// TIA Portal V17 export
// export: Created 2025-03-05T07:59:25.1832368Z, ExportSetting WithDefaults, DisplayName Totally Integrated Automation Portal, DisplayVersion V17 Update 8, DisplayName TIA Portal Openness, DisplayVersion V17 Update 8, DisplayName TIA Portal Version Control Interface, DisplayVersion V17, DisplayName SINAMICS Startdrive Advanced, DisplayVersion V17 SP2, DisplayName SINAMICS Startdrive G110M, G120, G120C, G120D, G120P, G115D, DisplayVersion V17 SP2, DisplayName SINAMICS Startdrive G130, G150, S120, S150, SINAMICS MV, S210, DisplayVersion V17 SP2, DisplayName STEP 7 Professional, DisplayVersion V17 Update 8, DisplayName SINUMERIK ONE STEP 7 Toolbox, DisplayVersion V17 Update 12, DisplayName SINUMERIK 840D sl STEP 7 Toolbox, DisplayVersion V17 Update 12, DisplayName STEP 7 Safety, DisplayVersion V17 Update 6, DisplayName WinCC Advanced, DisplayVersion V17 Update 8
FUNCTION "FC8101_MANUAL_LOADING_PART_STATUS_MANAGEMENT" : Void   // FC8101, LAD
{ S7_Optimized_Access := 'FALSE' }
VERSION : 0.1
// stored: AutoNumber false, IsIECCheckEnabled false, SetENOAutomatically false, UDAEnableTagReadback false
   VAR_TEMP
      AUX_STRING : String;
      CNT_CHARS : Int;
      CHARS_ARRAY : Array[0..63] of Char;
      ZERO : Byte;   // ZERO
      STATUS_BLKMOV : Int;   // STATUS BLKMOV
      STATUS_FILL : Int;   // STATUS FILL
   END_VAR
   VAR_TEMP   // added for the SCL form of the ladder/FBD networks
      _w1 : Bool;
      _w2 : Bool;
      _w3 : Bool;
      _w4 : Bool;
      _w5 : Bool;
      _w6 : Bool;
      _w7 : Bool;
      _w8 : Bool;
      _w9 : Bool;
      _w10 : Bool;
      _w11 : Bool;
   END_VAR
BEGIN

REGION Network 1: ZERO
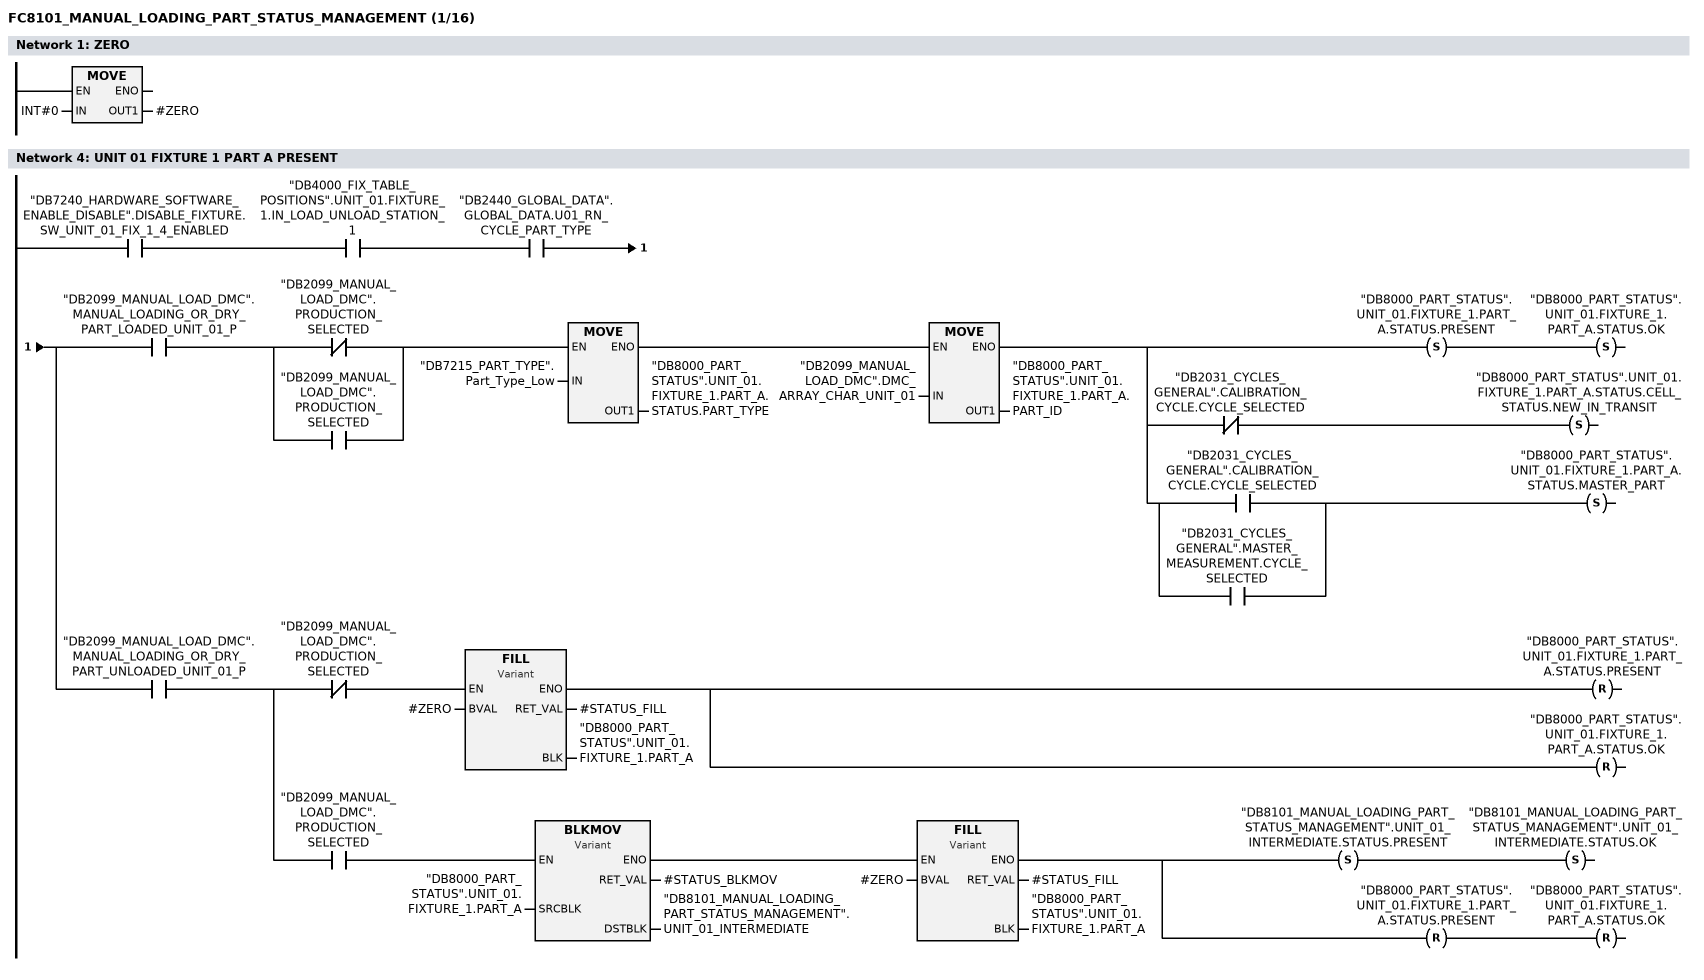
   RUNG wire#powerrail
      { S7_GenerateENO := "TRUE" } Move(in := INT#0, out1 => #ZERO)
   END_RUNG
   // the same network as SCL:
   #ZERO := INT#0;
END_REGION

REGION Network 2: <<<<<<<<<<<<<<<<<<<< RN CYCLE >>>>>>>>>>>>>>>>>>>>
END_REGION

REGION Network 3: <<<<<<<<<<<<<<<<<<<< UNIT 01 >>>>>>>>>>>>>>>>>>>>
END_REGION

REGION Network 4: UNIT 01 FIXTURE 1 PART A PRESENT
   RUNG wire#powerrail
      Contact( "DB7240_HARDWARE_SOFTWARE_ENABLE_DISABLE".DISABLE_FIXTURE.SW_UNIT_01_FIX_1_4_ENABLED )
      Contact( "DB4000_FIX_TABLE_POSITIONS".UNIT_01.FIXTURE_1.IN_LOAD_UNLOAD_STATION_1 )
      Contact( "DB2440_GLOBAL_DATA".GLOBAL_DATA.U01_RN_CYCLE_PART_TYPE )
      wire#w1
      Contact( "DB2099_MANUAL_LOAD_DMC".MANUAL_LOADING_OR_DRY_PART_LOADED_UNIT_01_P )
      wire#w2
      I_Contact( "DB2099_MANUAL_LOAD_DMC".PRODUCTION_SELECTED )
      wire#w3
      { S7_GenerateENO := "TRUE" } Move(in := "DB7215_PART_TYPE".Part_Type_Low, out1 => "DB8000_PART_STATUS".UNIT_01.FIXTURE_1.PART_A.STATUS.PART_TYPE)
      Move(in := "DB2099_MANUAL_LOAD_DMC".DMC_ARRAY_CHAR_UNIT_01, out1 => "DB8000_PART_STATUS".UNIT_01.FIXTURE_1.PART_A.PART_ID)
      wire#w4
      S_Coil( "DB8000_PART_STATUS".UNIT_01.FIXTURE_1.PART_A.STATUS.PRESENT )
      S_Coil( "DB8000_PART_STATUS".UNIT_01.FIXTURE_1.PART_A.STATUS.OK )
   END_RUNG
   RUNG wire#w2
      Contact( "DB2099_MANUAL_LOAD_DMC".PRODUCTION_SELECTED )
   END_RUNG wire#w3
   RUNG wire#w4
      I_Contact( "DB2031_CYCLES_GENERAL".CALIBRATION_CYCLE.CYCLE_SELECTED )
      S_Coil( "DB8000_PART_STATUS".UNIT_01.FIXTURE_1.PART_A.STATUS.CELL_STATUS.NEW_IN_TRANSIT )
   END_RUNG
   RUNG wire#w4
      Contact( "DB2031_CYCLES_GENERAL".CALIBRATION_CYCLE.CYCLE_SELECTED )
      wire#w5
      S_Coil( "DB8000_PART_STATUS".UNIT_01.FIXTURE_1.PART_A.STATUS.MASTER_PART )
   END_RUNG
   RUNG wire#w4
      Contact( "DB2031_CYCLES_GENERAL".MASTER_MEASUREMENT.CYCLE_SELECTED )
   END_RUNG wire#w5
   RUNG wire#w1
      Contact( "DB2099_MANUAL_LOAD_DMC".MANUAL_LOADING_OR_DRY_PART_UNLOADED_UNIT_01_P )
      wire#w6
      I_Contact( "DB2099_MANUAL_LOAD_DMC".PRODUCTION_SELECTED )
      { S7_Templates := "ptr_type := Variant" } FILL(BVAL := #ZERO, RET_VAL => #STATUS_FILL, BLK => "DB8000_PART_STATUS".UNIT_01.FIXTURE_1.PART_A)
      wire#w7
      R_Coil( "DB8000_PART_STATUS".UNIT_01.FIXTURE_1.PART_A.STATUS.PRESENT )
   END_RUNG
   RUNG wire#w7
      R_Coil( "DB8000_PART_STATUS".UNIT_01.FIXTURE_1.PART_A.STATUS.OK )
   END_RUNG
   RUNG wire#w6
      Contact( "DB2099_MANUAL_LOAD_DMC".PRODUCTION_SELECTED )
      { S7_Templates := "blk_type := Variant" } BLKMOV(SRCBLK := "DB8000_PART_STATUS".UNIT_01.FIXTURE_1.PART_A, RET_VAL => #STATUS_BLKMOV, DSTBLK => "DB8101_MANUAL_LOADING_PART_STATUS_MANAGEMENT".UNIT_01_INTERMEDIATE)
      { S7_Templates := "ptr_type := Variant" } FILL(BVAL := #ZERO, RET_VAL => #STATUS_FILL, BLK => "DB8000_PART_STATUS".UNIT_01.FIXTURE_1.PART_A)
      wire#w8
      S_Coil( "DB8101_MANUAL_LOADING_PART_STATUS_MANAGEMENT".UNIT_01_INTERMEDIATE.STATUS.PRESENT )
      S_Coil( "DB8101_MANUAL_LOADING_PART_STATUS_MANAGEMENT".UNIT_01_INTERMEDIATE.STATUS.OK )
   END_RUNG
   RUNG wire#w8
      R_Coil( "DB8000_PART_STATUS".UNIT_01.FIXTURE_1.PART_A.STATUS.PRESENT )
      R_Coil( "DB8000_PART_STATUS".UNIT_01.FIXTURE_1.PART_A.STATUS.OK )
   END_RUNG
   // the same network as SCL:
   // ENO of a box is taken as its EN; it also drops when the box reports an error
   #_w1 := "DB7240_HARDWARE_SOFTWARE_ENABLE_DISABLE".DISABLE_FIXTURE.SW_UNIT_01_FIX_1_4_ENABLED AND "DB4000_FIX_TABLE_POSITIONS".UNIT_01.FIXTURE_1.IN_LOAD_UNLOAD_STATION_1 AND "DB2440_GLOBAL_DATA".GLOBAL_DATA.U01_RN_CYCLE_PART_TYPE;
   #_w2 := #_w1 AND "DB2099_MANUAL_LOAD_DMC".MANUAL_LOADING_OR_DRY_PART_LOADED_UNIT_01_P AND (NOT "DB2099_MANUAL_LOAD_DMC".PRODUCTION_SELECTED OR "DB2099_MANUAL_LOAD_DMC".PRODUCTION_SELECTED);
   IF #_w2 THEN
       "DB8000_PART_STATUS".UNIT_01.FIXTURE_1.PART_A.STATUS.PART_TYPE := "DB7215_PART_TYPE".Part_Type_Low;
       "DB8000_PART_STATUS".UNIT_01.FIXTURE_1.PART_A.PART_ID := "DB2099_MANUAL_LOAD_DMC".DMC_ARRAY_CHAR_UNIT_01;
       "DB8000_PART_STATUS".UNIT_01.FIXTURE_1.PART_A.STATUS.PRESENT := TRUE;
       "DB8000_PART_STATUS".UNIT_01.FIXTURE_1.PART_A.STATUS.OK := TRUE;
   END_IF;
   IF #_w2 AND NOT "DB2031_CYCLES_GENERAL".CALIBRATION_CYCLE.CYCLE_SELECTED THEN
       "DB8000_PART_STATUS".UNIT_01.FIXTURE_1.PART_A.STATUS.CELL_STATUS.NEW_IN_TRANSIT := TRUE;
   END_IF;
   IF #_w2 AND ("DB2031_CYCLES_GENERAL".CALIBRATION_CYCLE.CYCLE_SELECTED OR "DB2031_CYCLES_GENERAL".MASTER_MEASUREMENT.CYCLE_SELECTED) THEN
       "DB8000_PART_STATUS".UNIT_01.FIXTURE_1.PART_A.STATUS.MASTER_PART := TRUE;
   END_IF;
   #_w3 := #_w1 AND "DB2099_MANUAL_LOAD_DMC".MANUAL_LOADING_OR_DRY_PART_UNLOADED_UNIT_01_P;
   #STATUS_FILL := FILL(EN := #_w3 AND NOT "DB2099_MANUAL_LOAD_DMC".PRODUCTION_SELECTED,
                        BVAL := #ZERO,
                        BLK => "DB8000_PART_STATUS".UNIT_01.FIXTURE_1.PART_A,
                        ENO => #_w4);
   IF #_w4 THEN
       "DB8000_PART_STATUS".UNIT_01.FIXTURE_1.PART_A.STATUS.PRESENT := FALSE;
       "DB8000_PART_STATUS".UNIT_01.FIXTURE_1.PART_A.STATUS.OK := FALSE;
   END_IF;
   #STATUS_BLKMOV := BLKMOV(EN := #_w3 AND "DB2099_MANUAL_LOAD_DMC".PRODUCTION_SELECTED,
                           SRCBLK := "DB8000_PART_STATUS".UNIT_01.FIXTURE_1.PART_A,
                           DSTBLK => "DB8101_MANUAL_LOADING_PART_STATUS_MANAGEMENT".UNIT_01_INTERMEDIATE,
                           ENO => #_w5);
   #STATUS_FILL := FILL(EN := #_w5,
                        BVAL := #ZERO,
                        BLK => "DB8000_PART_STATUS".UNIT_01.FIXTURE_1.PART_A,
                        ENO => #_w6);
   IF #_w6 THEN
       "DB8101_MANUAL_LOADING_PART_STATUS_MANAGEMENT".UNIT_01_INTERMEDIATE.STATUS.PRESENT := TRUE;
       "DB8101_MANUAL_LOADING_PART_STATUS_MANAGEMENT".UNIT_01_INTERMEDIATE.STATUS.OK := TRUE;
       "DB8000_PART_STATUS".UNIT_01.FIXTURE_1.PART_A.STATUS.PRESENT := FALSE;
       "DB8000_PART_STATUS".UNIT_01.FIXTURE_1.PART_A.STATUS.OK := FALSE;
   END_IF;
END_REGION

REGION Network 5: UNIT 01 FIXTURE 2 PART A PRESENT
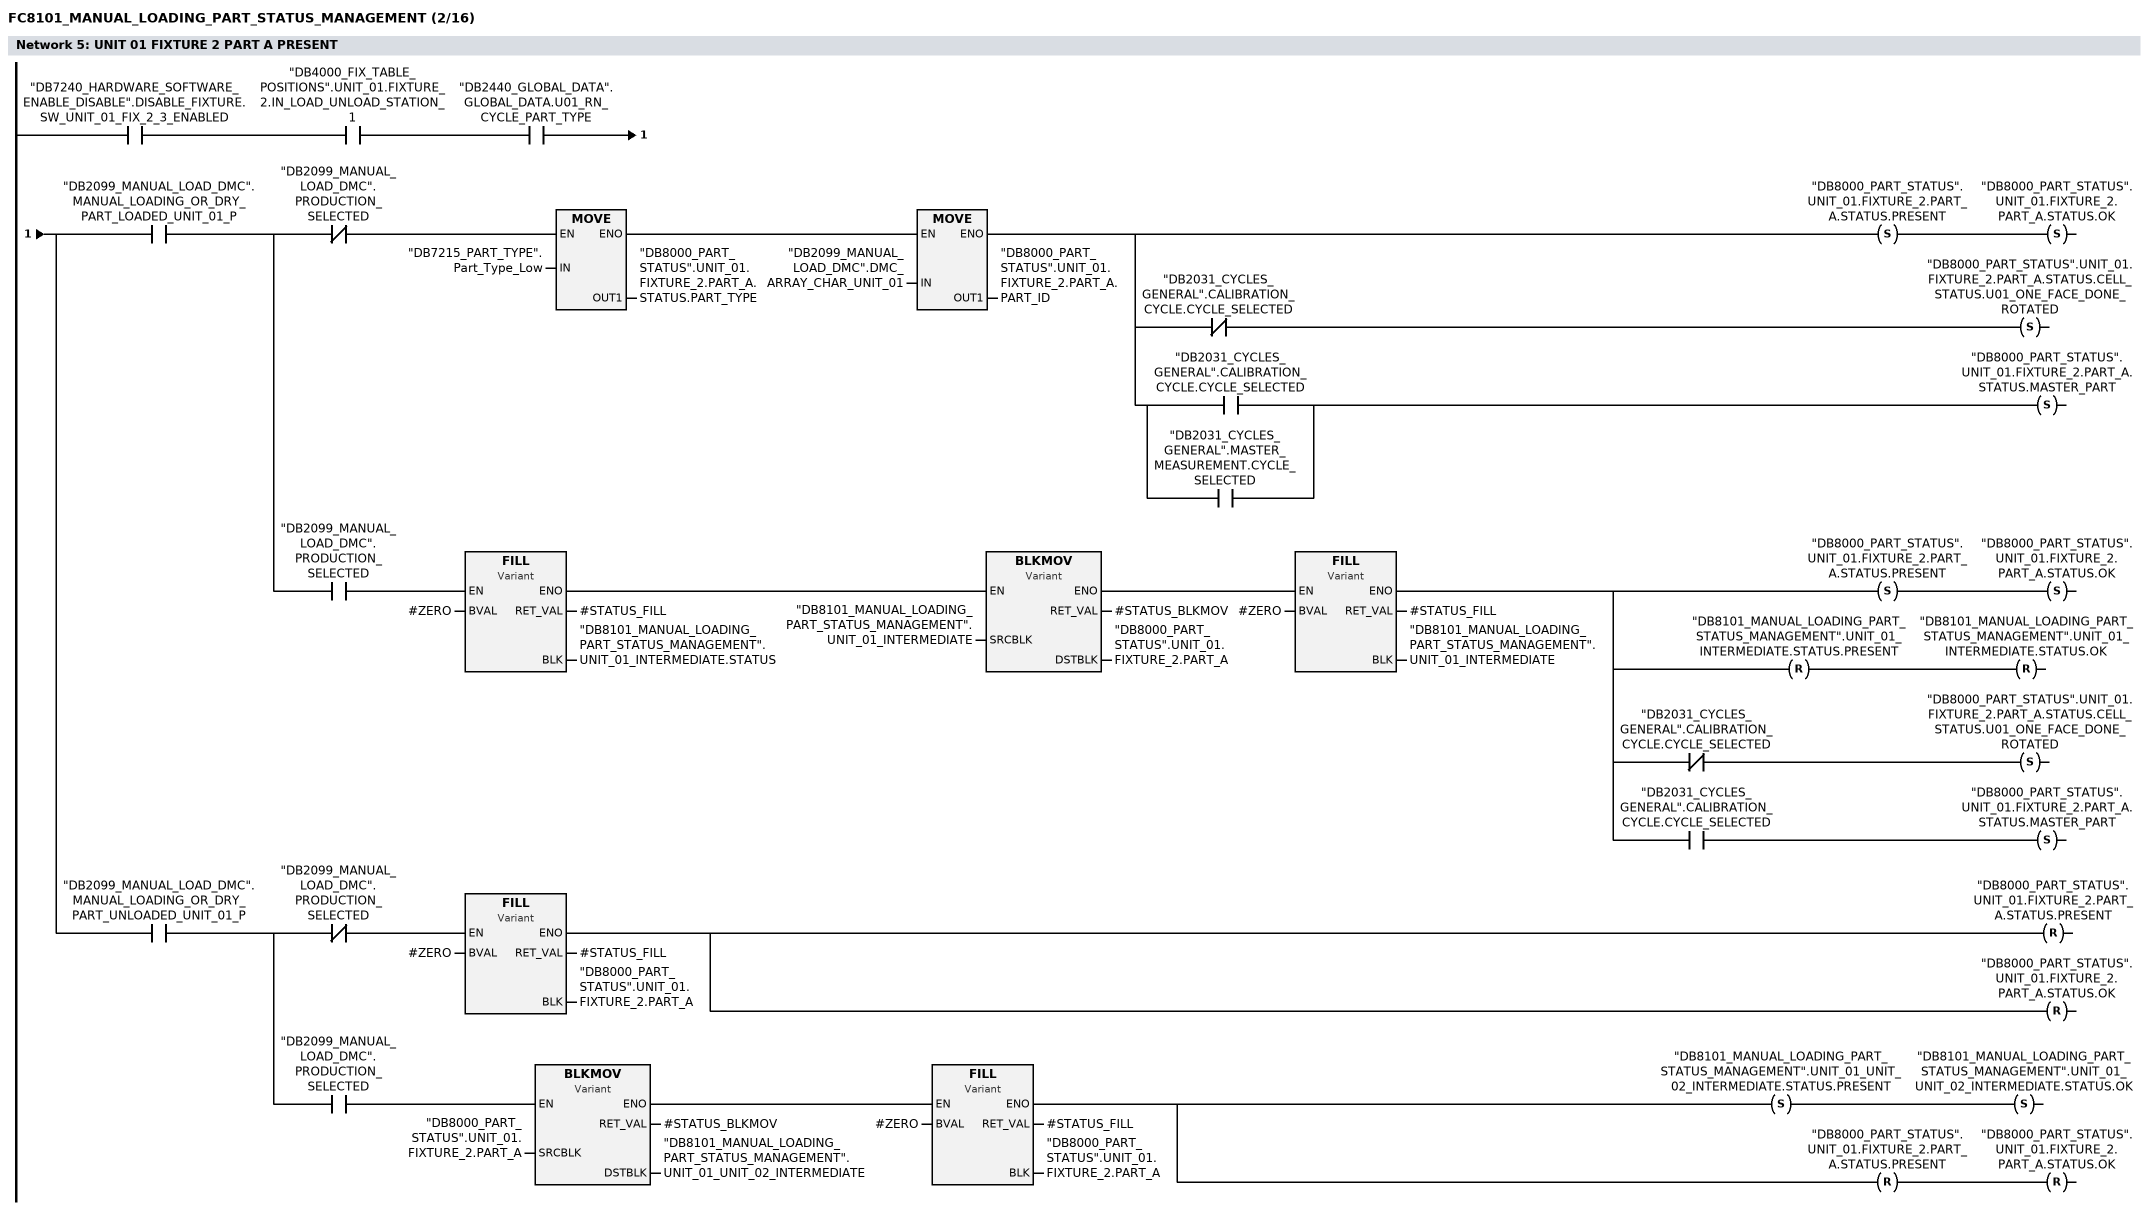
   RUNG wire#powerrail
      Contact( "DB7240_HARDWARE_SOFTWARE_ENABLE_DISABLE".DISABLE_FIXTURE.SW_UNIT_01_FIX_2_3_ENABLED )
      Contact( "DB4000_FIX_TABLE_POSITIONS".UNIT_01.FIXTURE_2.IN_LOAD_UNLOAD_STATION_1 )
      Contact( "DB2440_GLOBAL_DATA".GLOBAL_DATA.U01_RN_CYCLE_PART_TYPE )
      wire#w1
      Contact( "DB2099_MANUAL_LOAD_DMC".MANUAL_LOADING_OR_DRY_PART_LOADED_UNIT_01_P )
      wire#w2
      I_Contact( "DB2099_MANUAL_LOAD_DMC".PRODUCTION_SELECTED )
      { S7_GenerateENO := "TRUE" } Move(in := "DB7215_PART_TYPE".Part_Type_Low, out1 => "DB8000_PART_STATUS".UNIT_01.FIXTURE_2.PART_A.STATUS.PART_TYPE)
      Move(in := "DB2099_MANUAL_LOAD_DMC".DMC_ARRAY_CHAR_UNIT_01, out1 => "DB8000_PART_STATUS".UNIT_01.FIXTURE_2.PART_A.PART_ID)
      wire#w3
      S_Coil( "DB8000_PART_STATUS".UNIT_01.FIXTURE_2.PART_A.STATUS.PRESENT )
      S_Coil( "DB8000_PART_STATUS".UNIT_01.FIXTURE_2.PART_A.STATUS.OK )
   END_RUNG
   RUNG wire#w3
      I_Contact( "DB2031_CYCLES_GENERAL".CALIBRATION_CYCLE.CYCLE_SELECTED )
      S_Coil( "DB8000_PART_STATUS".UNIT_01.FIXTURE_2.PART_A.STATUS.CELL_STATUS.U01_ONE_FACE_DONE_ROTATED )
   END_RUNG
   RUNG wire#w3
      Contact( "DB2031_CYCLES_GENERAL".CALIBRATION_CYCLE.CYCLE_SELECTED )
      wire#w4
      S_Coil( "DB8000_PART_STATUS".UNIT_01.FIXTURE_2.PART_A.STATUS.MASTER_PART )
   END_RUNG
   RUNG wire#w3
      Contact( "DB2031_CYCLES_GENERAL".MASTER_MEASUREMENT.CYCLE_SELECTED )
   END_RUNG wire#w4
   RUNG wire#w2
      Contact( "DB2099_MANUAL_LOAD_DMC".PRODUCTION_SELECTED )
      { S7_Templates := "ptr_type := Variant" } FILL(BVAL := #ZERO, RET_VAL => #STATUS_FILL, BLK => "DB8101_MANUAL_LOADING_PART_STATUS_MANAGEMENT".UNIT_01_INTERMEDIATE.STATUS)
      { S7_Templates := "blk_type := Variant" } BLKMOV(SRCBLK := "DB8101_MANUAL_LOADING_PART_STATUS_MANAGEMENT".UNIT_01_INTERMEDIATE, RET_VAL => #STATUS_BLKMOV, DSTBLK => "DB8000_PART_STATUS".UNIT_01.FIXTURE_2.PART_A)
      { S7_Templates := "ptr_type := Variant" } FILL(BVAL := #ZERO, RET_VAL => #STATUS_FILL, BLK => "DB8101_MANUAL_LOADING_PART_STATUS_MANAGEMENT".UNIT_01_INTERMEDIATE)
      wire#w5
      S_Coil( "DB8000_PART_STATUS".UNIT_01.FIXTURE_2.PART_A.STATUS.PRESENT )
      S_Coil( "DB8000_PART_STATUS".UNIT_01.FIXTURE_2.PART_A.STATUS.OK )
   END_RUNG
   RUNG wire#w5
      R_Coil( "DB8101_MANUAL_LOADING_PART_STATUS_MANAGEMENT".UNIT_01_INTERMEDIATE.STATUS.PRESENT )
      R_Coil( "DB8101_MANUAL_LOADING_PART_STATUS_MANAGEMENT".UNIT_01_INTERMEDIATE.STATUS.OK )
   END_RUNG
   RUNG wire#w5
      I_Contact( "DB2031_CYCLES_GENERAL".CALIBRATION_CYCLE.CYCLE_SELECTED )
      S_Coil( "DB8000_PART_STATUS".UNIT_01.FIXTURE_2.PART_A.STATUS.CELL_STATUS.U01_ONE_FACE_DONE_ROTATED )
   END_RUNG
   RUNG wire#w5
      Contact( "DB2031_CYCLES_GENERAL".CALIBRATION_CYCLE.CYCLE_SELECTED )
      S_Coil( "DB8000_PART_STATUS".UNIT_01.FIXTURE_2.PART_A.STATUS.MASTER_PART )
   END_RUNG
   RUNG wire#w1
      Contact( "DB2099_MANUAL_LOAD_DMC".MANUAL_LOADING_OR_DRY_PART_UNLOADED_UNIT_01_P )
      wire#w6
      I_Contact( "DB2099_MANUAL_LOAD_DMC".PRODUCTION_SELECTED )
      { S7_Templates := "ptr_type := Variant" } FILL(BVAL := #ZERO, RET_VAL => #STATUS_FILL, BLK => "DB8000_PART_STATUS".UNIT_01.FIXTURE_2.PART_A)
      wire#w7
      R_Coil( "DB8000_PART_STATUS".UNIT_01.FIXTURE_2.PART_A.STATUS.PRESENT )
   END_RUNG
   RUNG wire#w7
      R_Coil( "DB8000_PART_STATUS".UNIT_01.FIXTURE_2.PART_A.STATUS.OK )
   END_RUNG
   RUNG wire#w6
      Contact( "DB2099_MANUAL_LOAD_DMC".PRODUCTION_SELECTED )
      { S7_Templates := "blk_type := Variant" } BLKMOV(SRCBLK := "DB8000_PART_STATUS".UNIT_01.FIXTURE_2.PART_A, RET_VAL => #STATUS_BLKMOV, DSTBLK => "DB8101_MANUAL_LOADING_PART_STATUS_MANAGEMENT".UNIT_01_UNIT_02_INTERMEDIATE)
      { S7_Templates := "ptr_type := Variant" } FILL(BVAL := #ZERO, RET_VAL => #STATUS_FILL, BLK => "DB8000_PART_STATUS".UNIT_01.FIXTURE_2.PART_A)
      wire#w8
      S_Coil( "DB8101_MANUAL_LOADING_PART_STATUS_MANAGEMENT".UNIT_01_UNIT_02_INTERMEDIATE.STATUS.PRESENT )
      S_Coil( "DB8101_MANUAL_LOADING_PART_STATUS_MANAGEMENT".UNIT_01_UNIT_02_INTERMEDIATE.STATUS.OK )
   END_RUNG
   RUNG wire#w8
      R_Coil( "DB8000_PART_STATUS".UNIT_01.FIXTURE_2.PART_A.STATUS.PRESENT )
      R_Coil( "DB8000_PART_STATUS".UNIT_01.FIXTURE_2.PART_A.STATUS.OK )
   END_RUNG
   // the same network as SCL:
   // ENO of a box is taken as its EN; it also drops when the box reports an error
   #_w1 := "DB7240_HARDWARE_SOFTWARE_ENABLE_DISABLE".DISABLE_FIXTURE.SW_UNIT_01_FIX_2_3_ENABLED AND "DB4000_FIX_TABLE_POSITIONS".UNIT_01.FIXTURE_2.IN_LOAD_UNLOAD_STATION_1 AND "DB2440_GLOBAL_DATA".GLOBAL_DATA.U01_RN_CYCLE_PART_TYPE;
   #_w2 := #_w1 AND "DB2099_MANUAL_LOAD_DMC".MANUAL_LOADING_OR_DRY_PART_LOADED_UNIT_01_P;
   #_w3 := #_w2 AND NOT "DB2099_MANUAL_LOAD_DMC".PRODUCTION_SELECTED;
   IF #_w3 THEN
       "DB8000_PART_STATUS".UNIT_01.FIXTURE_2.PART_A.STATUS.PART_TYPE := "DB7215_PART_TYPE".Part_Type_Low;
       "DB8000_PART_STATUS".UNIT_01.FIXTURE_2.PART_A.PART_ID := "DB2099_MANUAL_LOAD_DMC".DMC_ARRAY_CHAR_UNIT_01;
       "DB8000_PART_STATUS".UNIT_01.FIXTURE_2.PART_A.STATUS.PRESENT := TRUE;
       "DB8000_PART_STATUS".UNIT_01.FIXTURE_2.PART_A.STATUS.OK := TRUE;
   END_IF;
   IF #_w3 AND NOT "DB2031_CYCLES_GENERAL".CALIBRATION_CYCLE.CYCLE_SELECTED THEN
       "DB8000_PART_STATUS".UNIT_01.FIXTURE_2.PART_A.STATUS.CELL_STATUS.U01_ONE_FACE_DONE_ROTATED := TRUE;
   END_IF;
   IF #_w3 AND ("DB2031_CYCLES_GENERAL".CALIBRATION_CYCLE.CYCLE_SELECTED OR "DB2031_CYCLES_GENERAL".MASTER_MEASUREMENT.CYCLE_SELECTED) THEN
       "DB8000_PART_STATUS".UNIT_01.FIXTURE_2.PART_A.STATUS.MASTER_PART := TRUE;
   END_IF;
   #_w4 := #_w2 AND "DB2099_MANUAL_LOAD_DMC".PRODUCTION_SELECTED;
   #STATUS_FILL := FILL(EN := #_w4,
                        BVAL := #ZERO,
                        BLK => "DB8101_MANUAL_LOADING_PART_STATUS_MANAGEMENT".UNIT_01_INTERMEDIATE.STATUS,
                        ENO => #_w5);
   #STATUS_BLKMOV := BLKMOV(EN := #_w5,
                           SRCBLK := "DB8101_MANUAL_LOADING_PART_STATUS_MANAGEMENT".UNIT_01_INTERMEDIATE,
                           DSTBLK => "DB8000_PART_STATUS".UNIT_01.FIXTURE_2.PART_A,
                           ENO => #_w6);
   #STATUS_FILL := FILL(EN := #_w6,
                        BVAL := #ZERO,
                        BLK => "DB8101_MANUAL_LOADING_PART_STATUS_MANAGEMENT".UNIT_01_INTERMEDIATE,
                        ENO => #_w7);
   IF #_w7 THEN
       "DB8000_PART_STATUS".UNIT_01.FIXTURE_2.PART_A.STATUS.PRESENT := TRUE;
       "DB8000_PART_STATUS".UNIT_01.FIXTURE_2.PART_A.STATUS.OK := TRUE;
       "DB8101_MANUAL_LOADING_PART_STATUS_MANAGEMENT".UNIT_01_INTERMEDIATE.STATUS.PRESENT := FALSE;
       "DB8101_MANUAL_LOADING_PART_STATUS_MANAGEMENT".UNIT_01_INTERMEDIATE.STATUS.OK := FALSE;
   END_IF;
   IF #_w7 AND NOT "DB2031_CYCLES_GENERAL".CALIBRATION_CYCLE.CYCLE_SELECTED THEN
       "DB8000_PART_STATUS".UNIT_01.FIXTURE_2.PART_A.STATUS.CELL_STATUS.U01_ONE_FACE_DONE_ROTATED := TRUE;
   END_IF;
   IF #_w7 AND "DB2031_CYCLES_GENERAL".CALIBRATION_CYCLE.CYCLE_SELECTED THEN
       "DB8000_PART_STATUS".UNIT_01.FIXTURE_2.PART_A.STATUS.MASTER_PART := TRUE;
   END_IF;
   #_w8 := #_w1 AND "DB2099_MANUAL_LOAD_DMC".MANUAL_LOADING_OR_DRY_PART_UNLOADED_UNIT_01_P;
   #STATUS_FILL := FILL(EN := #_w8 AND NOT "DB2099_MANUAL_LOAD_DMC".PRODUCTION_SELECTED,
                        BVAL := #ZERO,
                        BLK => "DB8000_PART_STATUS".UNIT_01.FIXTURE_2.PART_A,
                        ENO => #_w9);
   IF #_w9 THEN
       "DB8000_PART_STATUS".UNIT_01.FIXTURE_2.PART_A.STATUS.PRESENT := FALSE;
       "DB8000_PART_STATUS".UNIT_01.FIXTURE_2.PART_A.STATUS.OK := FALSE;
   END_IF;
   #STATUS_BLKMOV := BLKMOV(EN := #_w8 AND "DB2099_MANUAL_LOAD_DMC".PRODUCTION_SELECTED,
                           SRCBLK := "DB8000_PART_STATUS".UNIT_01.FIXTURE_2.PART_A,
                           DSTBLK => "DB8101_MANUAL_LOADING_PART_STATUS_MANAGEMENT".UNIT_01_UNIT_02_INTERMEDIATE,
                           ENO => #_w10);
   #STATUS_FILL := FILL(EN := #_w10,
                        BVAL := #ZERO,
                        BLK => "DB8000_PART_STATUS".UNIT_01.FIXTURE_2.PART_A,
                        ENO => #_w11);
   IF #_w11 THEN
       "DB8101_MANUAL_LOADING_PART_STATUS_MANAGEMENT".UNIT_01_UNIT_02_INTERMEDIATE.STATUS.PRESENT := TRUE;
       "DB8101_MANUAL_LOADING_PART_STATUS_MANAGEMENT".UNIT_01_UNIT_02_INTERMEDIATE.STATUS.OK := TRUE;
       "DB8000_PART_STATUS".UNIT_01.FIXTURE_2.PART_A.STATUS.PRESENT := FALSE;
       "DB8000_PART_STATUS".UNIT_01.FIXTURE_2.PART_A.STATUS.OK := FALSE;
   END_IF;
END_REGION

REGION Network 6: UNIT 01 FIXTURE 3 PART A PRESENT
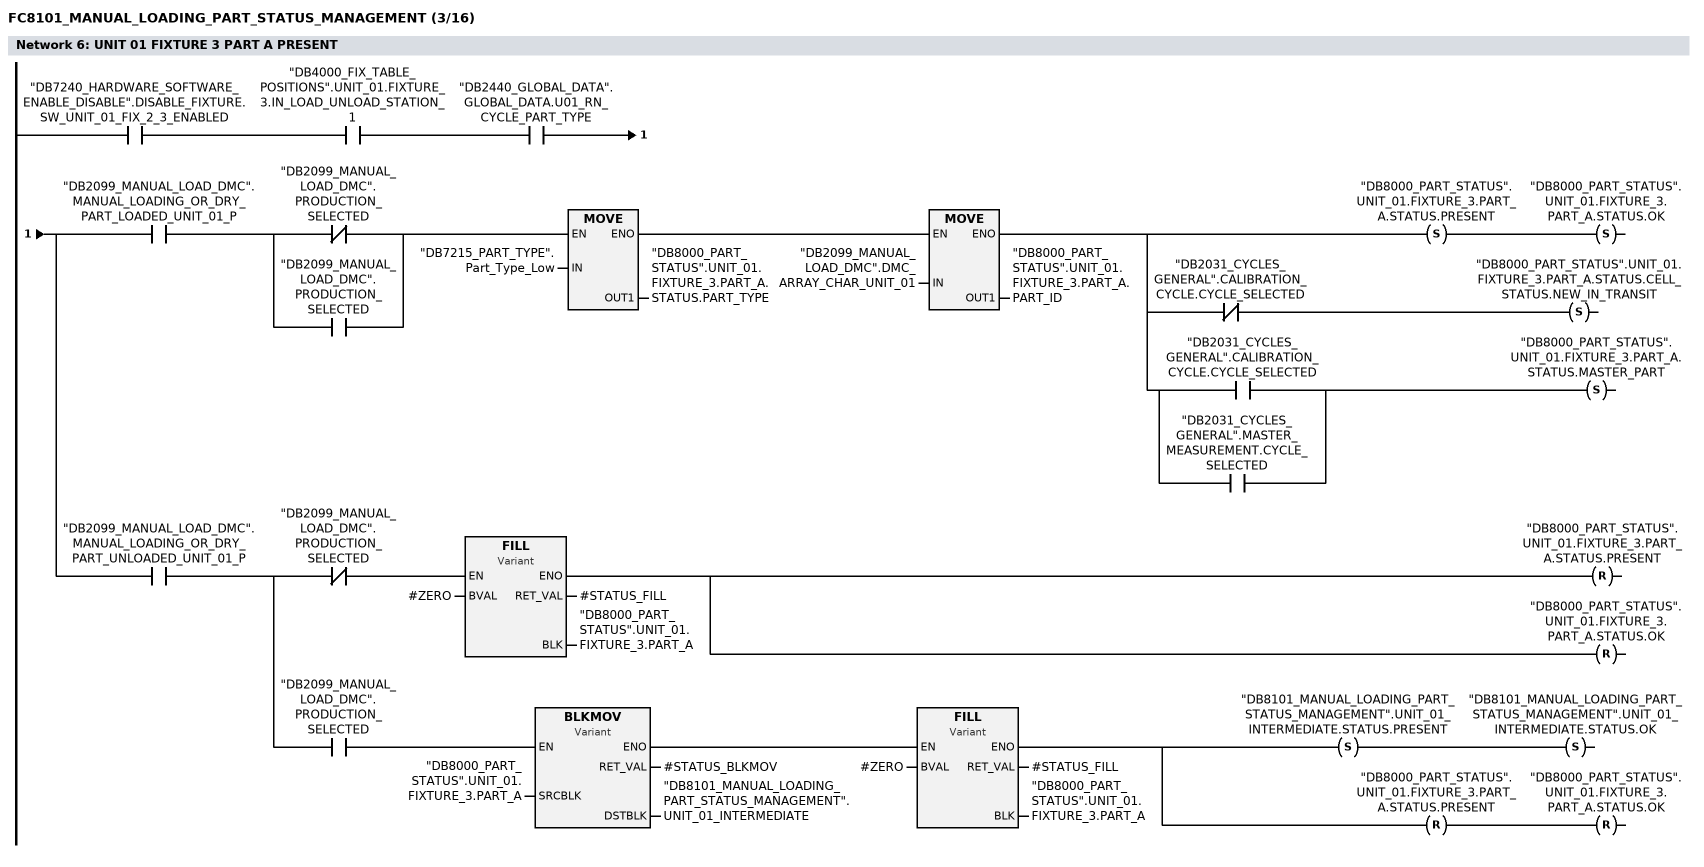
   RUNG wire#powerrail
      Contact( "DB7240_HARDWARE_SOFTWARE_ENABLE_DISABLE".DISABLE_FIXTURE.SW_UNIT_01_FIX_2_3_ENABLED )
      Contact( "DB4000_FIX_TABLE_POSITIONS".UNIT_01.FIXTURE_3.IN_LOAD_UNLOAD_STATION_1 )
      Contact( "DB2440_GLOBAL_DATA".GLOBAL_DATA.U01_RN_CYCLE_PART_TYPE )
      wire#w1
      Contact( "DB2099_MANUAL_LOAD_DMC".MANUAL_LOADING_OR_DRY_PART_LOADED_UNIT_01_P )
      wire#w2
      I_Contact( "DB2099_MANUAL_LOAD_DMC".PRODUCTION_SELECTED )
      wire#w3
      { S7_GenerateENO := "TRUE" } Move(in := "DB7215_PART_TYPE".Part_Type_Low, out1 => "DB8000_PART_STATUS".UNIT_01.FIXTURE_3.PART_A.STATUS.PART_TYPE)
      Move(in := "DB2099_MANUAL_LOAD_DMC".DMC_ARRAY_CHAR_UNIT_01, out1 => "DB8000_PART_STATUS".UNIT_01.FIXTURE_3.PART_A.PART_ID)
      wire#w4
      S_Coil( "DB8000_PART_STATUS".UNIT_01.FIXTURE_3.PART_A.STATUS.PRESENT )
      S_Coil( "DB8000_PART_STATUS".UNIT_01.FIXTURE_3.PART_A.STATUS.OK )
   END_RUNG
   RUNG wire#w2
      Contact( "DB2099_MANUAL_LOAD_DMC".PRODUCTION_SELECTED )
   END_RUNG wire#w3
   RUNG wire#w4
      I_Contact( "DB2031_CYCLES_GENERAL".CALIBRATION_CYCLE.CYCLE_SELECTED )
      S_Coil( "DB8000_PART_STATUS".UNIT_01.FIXTURE_3.PART_A.STATUS.CELL_STATUS.NEW_IN_TRANSIT )
   END_RUNG
   RUNG wire#w4
      Contact( "DB2031_CYCLES_GENERAL".CALIBRATION_CYCLE.CYCLE_SELECTED )
      wire#w5
      S_Coil( "DB8000_PART_STATUS".UNIT_01.FIXTURE_3.PART_A.STATUS.MASTER_PART )
   END_RUNG
   RUNG wire#w4
      Contact( "DB2031_CYCLES_GENERAL".MASTER_MEASUREMENT.CYCLE_SELECTED )
   END_RUNG wire#w5
   RUNG wire#w1
      Contact( "DB2099_MANUAL_LOAD_DMC".MANUAL_LOADING_OR_DRY_PART_UNLOADED_UNIT_01_P )
      wire#w6
      I_Contact( "DB2099_MANUAL_LOAD_DMC".PRODUCTION_SELECTED )
      { S7_Templates := "ptr_type := Variant" } FILL(BVAL := #ZERO, RET_VAL => #STATUS_FILL, BLK => "DB8000_PART_STATUS".UNIT_01.FIXTURE_3.PART_A)
      wire#w7
      R_Coil( "DB8000_PART_STATUS".UNIT_01.FIXTURE_3.PART_A.STATUS.PRESENT )
   END_RUNG
   RUNG wire#w7
      R_Coil( "DB8000_PART_STATUS".UNIT_01.FIXTURE_3.PART_A.STATUS.OK )
   END_RUNG
   RUNG wire#w6
      Contact( "DB2099_MANUAL_LOAD_DMC".PRODUCTION_SELECTED )
      { S7_Templates := "blk_type := Variant" } BLKMOV(SRCBLK := "DB8000_PART_STATUS".UNIT_01.FIXTURE_3.PART_A, RET_VAL => #STATUS_BLKMOV, DSTBLK => "DB8101_MANUAL_LOADING_PART_STATUS_MANAGEMENT".UNIT_01_INTERMEDIATE)
      { S7_Templates := "ptr_type := Variant" } FILL(BVAL := #ZERO, RET_VAL => #STATUS_FILL, BLK => "DB8000_PART_STATUS".UNIT_01.FIXTURE_3.PART_A)
      wire#w8
      S_Coil( "DB8101_MANUAL_LOADING_PART_STATUS_MANAGEMENT".UNIT_01_INTERMEDIATE.STATUS.PRESENT )
      S_Coil( "DB8101_MANUAL_LOADING_PART_STATUS_MANAGEMENT".UNIT_01_INTERMEDIATE.STATUS.OK )
   END_RUNG
   RUNG wire#w8
      R_Coil( "DB8000_PART_STATUS".UNIT_01.FIXTURE_3.PART_A.STATUS.PRESENT )
      R_Coil( "DB8000_PART_STATUS".UNIT_01.FIXTURE_3.PART_A.STATUS.OK )
   END_RUNG
   // the same network as SCL:
   // ENO of a box is taken as its EN; it also drops when the box reports an error
   #_w1 := "DB7240_HARDWARE_SOFTWARE_ENABLE_DISABLE".DISABLE_FIXTURE.SW_UNIT_01_FIX_2_3_ENABLED AND "DB4000_FIX_TABLE_POSITIONS".UNIT_01.FIXTURE_3.IN_LOAD_UNLOAD_STATION_1 AND "DB2440_GLOBAL_DATA".GLOBAL_DATA.U01_RN_CYCLE_PART_TYPE;
   #_w2 := #_w1 AND "DB2099_MANUAL_LOAD_DMC".MANUAL_LOADING_OR_DRY_PART_LOADED_UNIT_01_P AND (NOT "DB2099_MANUAL_LOAD_DMC".PRODUCTION_SELECTED OR "DB2099_MANUAL_LOAD_DMC".PRODUCTION_SELECTED);
   IF #_w2 THEN
       "DB8000_PART_STATUS".UNIT_01.FIXTURE_3.PART_A.STATUS.PART_TYPE := "DB7215_PART_TYPE".Part_Type_Low;
       "DB8000_PART_STATUS".UNIT_01.FIXTURE_3.PART_A.PART_ID := "DB2099_MANUAL_LOAD_DMC".DMC_ARRAY_CHAR_UNIT_01;
       "DB8000_PART_STATUS".UNIT_01.FIXTURE_3.PART_A.STATUS.PRESENT := TRUE;
       "DB8000_PART_STATUS".UNIT_01.FIXTURE_3.PART_A.STATUS.OK := TRUE;
   END_IF;
   IF #_w2 AND NOT "DB2031_CYCLES_GENERAL".CALIBRATION_CYCLE.CYCLE_SELECTED THEN
       "DB8000_PART_STATUS".UNIT_01.FIXTURE_3.PART_A.STATUS.CELL_STATUS.NEW_IN_TRANSIT := TRUE;
   END_IF;
   IF #_w2 AND ("DB2031_CYCLES_GENERAL".CALIBRATION_CYCLE.CYCLE_SELECTED OR "DB2031_CYCLES_GENERAL".MASTER_MEASUREMENT.CYCLE_SELECTED) THEN
       "DB8000_PART_STATUS".UNIT_01.FIXTURE_3.PART_A.STATUS.MASTER_PART := TRUE;
   END_IF;
   #_w3 := #_w1 AND "DB2099_MANUAL_LOAD_DMC".MANUAL_LOADING_OR_DRY_PART_UNLOADED_UNIT_01_P;
   #STATUS_FILL := FILL(EN := #_w3 AND NOT "DB2099_MANUAL_LOAD_DMC".PRODUCTION_SELECTED,
                        BVAL := #ZERO,
                        BLK => "DB8000_PART_STATUS".UNIT_01.FIXTURE_3.PART_A,
                        ENO => #_w4);
   IF #_w4 THEN
       "DB8000_PART_STATUS".UNIT_01.FIXTURE_3.PART_A.STATUS.PRESENT := FALSE;
       "DB8000_PART_STATUS".UNIT_01.FIXTURE_3.PART_A.STATUS.OK := FALSE;
   END_IF;
   #STATUS_BLKMOV := BLKMOV(EN := #_w3 AND "DB2099_MANUAL_LOAD_DMC".PRODUCTION_SELECTED,
                           SRCBLK := "DB8000_PART_STATUS".UNIT_01.FIXTURE_3.PART_A,
                           DSTBLK => "DB8101_MANUAL_LOADING_PART_STATUS_MANAGEMENT".UNIT_01_INTERMEDIATE,
                           ENO => #_w5);
   #STATUS_FILL := FILL(EN := #_w5,
                        BVAL := #ZERO,
                        BLK => "DB8000_PART_STATUS".UNIT_01.FIXTURE_3.PART_A,
                        ENO => #_w6);
   IF #_w6 THEN
       "DB8101_MANUAL_LOADING_PART_STATUS_MANAGEMENT".UNIT_01_INTERMEDIATE.STATUS.PRESENT := TRUE;
       "DB8101_MANUAL_LOADING_PART_STATUS_MANAGEMENT".UNIT_01_INTERMEDIATE.STATUS.OK := TRUE;
       "DB8000_PART_STATUS".UNIT_01.FIXTURE_3.PART_A.STATUS.PRESENT := FALSE;
       "DB8000_PART_STATUS".UNIT_01.FIXTURE_3.PART_A.STATUS.OK := FALSE;
   END_IF;
END_REGION

REGION Network 7: UNIT 01 FIXTURE 4 PART A PRESENT
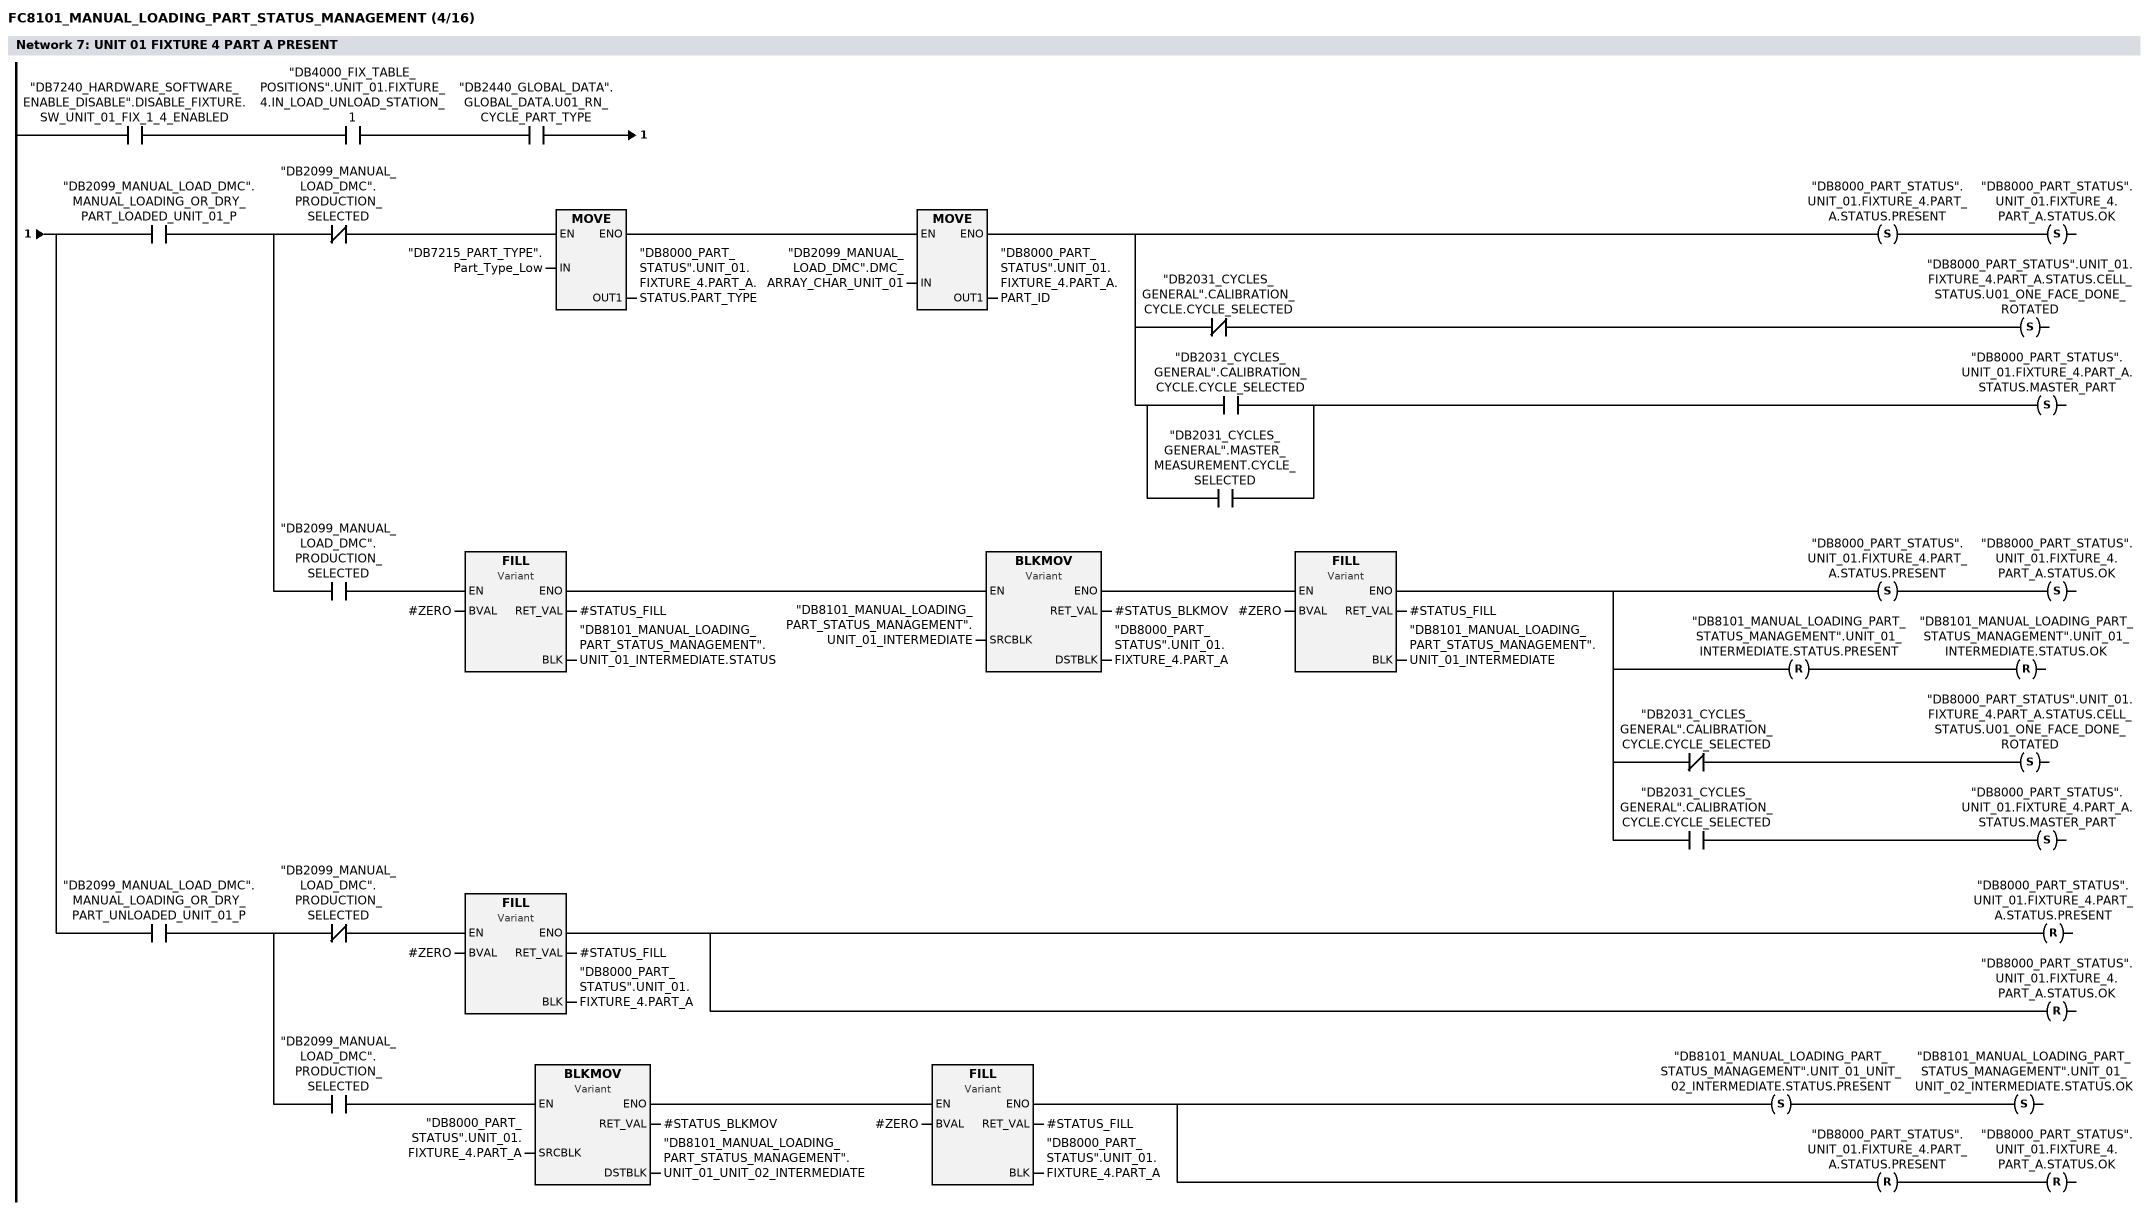
   RUNG wire#powerrail
      Contact( "DB7240_HARDWARE_SOFTWARE_ENABLE_DISABLE".DISABLE_FIXTURE.SW_UNIT_01_FIX_1_4_ENABLED )
      Contact( "DB4000_FIX_TABLE_POSITIONS".UNIT_01.FIXTURE_4.IN_LOAD_UNLOAD_STATION_1 )
      Contact( "DB2440_GLOBAL_DATA".GLOBAL_DATA.U01_RN_CYCLE_PART_TYPE )
      wire#w1
      Contact( "DB2099_MANUAL_LOAD_DMC".MANUAL_LOADING_OR_DRY_PART_LOADED_UNIT_01_P )
      wire#w2
      I_Contact( "DB2099_MANUAL_LOAD_DMC".PRODUCTION_SELECTED )
      { S7_GenerateENO := "TRUE" } Move(in := "DB7215_PART_TYPE".Part_Type_Low, out1 => "DB8000_PART_STATUS".UNIT_01.FIXTURE_4.PART_A.STATUS.PART_TYPE)
      Move(in := "DB2099_MANUAL_LOAD_DMC".DMC_ARRAY_CHAR_UNIT_01, out1 => "DB8000_PART_STATUS".UNIT_01.FIXTURE_4.PART_A.PART_ID)
      wire#w3
      S_Coil( "DB8000_PART_STATUS".UNIT_01.FIXTURE_4.PART_A.STATUS.PRESENT )
      S_Coil( "DB8000_PART_STATUS".UNIT_01.FIXTURE_4.PART_A.STATUS.OK )
   END_RUNG
   RUNG wire#w3
      I_Contact( "DB2031_CYCLES_GENERAL".CALIBRATION_CYCLE.CYCLE_SELECTED )
      S_Coil( "DB8000_PART_STATUS".UNIT_01.FIXTURE_4.PART_A.STATUS.CELL_STATUS.U01_ONE_FACE_DONE_ROTATED )
   END_RUNG
   RUNG wire#w3
      Contact( "DB2031_CYCLES_GENERAL".CALIBRATION_CYCLE.CYCLE_SELECTED )
      wire#w4
      S_Coil( "DB8000_PART_STATUS".UNIT_01.FIXTURE_4.PART_A.STATUS.MASTER_PART )
   END_RUNG
   RUNG wire#w3
      Contact( "DB2031_CYCLES_GENERAL".MASTER_MEASUREMENT.CYCLE_SELECTED )
   END_RUNG wire#w4
   RUNG wire#w2
      Contact( "DB2099_MANUAL_LOAD_DMC".PRODUCTION_SELECTED )
      { S7_Templates := "ptr_type := Variant" } FILL(BVAL := #ZERO, RET_VAL => #STATUS_FILL, BLK => "DB8101_MANUAL_LOADING_PART_STATUS_MANAGEMENT".UNIT_01_INTERMEDIATE.STATUS)
      { S7_Templates := "blk_type := Variant" } BLKMOV(SRCBLK := "DB8101_MANUAL_LOADING_PART_STATUS_MANAGEMENT".UNIT_01_INTERMEDIATE, RET_VAL => #STATUS_BLKMOV, DSTBLK => "DB8000_PART_STATUS".UNIT_01.FIXTURE_4.PART_A)
      { S7_Templates := "ptr_type := Variant" } FILL(BVAL := #ZERO, RET_VAL => #STATUS_FILL, BLK => "DB8101_MANUAL_LOADING_PART_STATUS_MANAGEMENT".UNIT_01_INTERMEDIATE)
      wire#w5
      S_Coil( "DB8000_PART_STATUS".UNIT_01.FIXTURE_4.PART_A.STATUS.PRESENT )
      S_Coil( "DB8000_PART_STATUS".UNIT_01.FIXTURE_4.PART_A.STATUS.OK )
   END_RUNG
   RUNG wire#w5
      R_Coil( "DB8101_MANUAL_LOADING_PART_STATUS_MANAGEMENT".UNIT_01_INTERMEDIATE.STATUS.PRESENT )
      R_Coil( "DB8101_MANUAL_LOADING_PART_STATUS_MANAGEMENT".UNIT_01_INTERMEDIATE.STATUS.OK )
   END_RUNG
   RUNG wire#w5
      I_Contact( "DB2031_CYCLES_GENERAL".CALIBRATION_CYCLE.CYCLE_SELECTED )
      S_Coil( "DB8000_PART_STATUS".UNIT_01.FIXTURE_4.PART_A.STATUS.CELL_STATUS.U01_ONE_FACE_DONE_ROTATED )
   END_RUNG
   RUNG wire#w5
      Contact( "DB2031_CYCLES_GENERAL".CALIBRATION_CYCLE.CYCLE_SELECTED )
      S_Coil( "DB8000_PART_STATUS".UNIT_01.FIXTURE_4.PART_A.STATUS.MASTER_PART )
   END_RUNG
   RUNG wire#w1
      Contact( "DB2099_MANUAL_LOAD_DMC".MANUAL_LOADING_OR_DRY_PART_UNLOADED_UNIT_01_P )
      wire#w6
      I_Contact( "DB2099_MANUAL_LOAD_DMC".PRODUCTION_SELECTED )
      { S7_Templates := "ptr_type := Variant" } FILL(BVAL := #ZERO, RET_VAL => #STATUS_FILL, BLK => "DB8000_PART_STATUS".UNIT_01.FIXTURE_4.PART_A)
      wire#w7
      R_Coil( "DB8000_PART_STATUS".UNIT_01.FIXTURE_4.PART_A.STATUS.PRESENT )
   END_RUNG
   RUNG wire#w7
      R_Coil( "DB8000_PART_STATUS".UNIT_01.FIXTURE_4.PART_A.STATUS.OK )
   END_RUNG
   RUNG wire#w6
      Contact( "DB2099_MANUAL_LOAD_DMC".PRODUCTION_SELECTED )
      { S7_Templates := "blk_type := Variant" } BLKMOV(SRCBLK := "DB8000_PART_STATUS".UNIT_01.FIXTURE_4.PART_A, RET_VAL => #STATUS_BLKMOV, DSTBLK => "DB8101_MANUAL_LOADING_PART_STATUS_MANAGEMENT".UNIT_01_UNIT_02_INTERMEDIATE)
      { S7_Templates := "ptr_type := Variant" } FILL(BVAL := #ZERO, RET_VAL => #STATUS_FILL, BLK => "DB8000_PART_STATUS".UNIT_01.FIXTURE_4.PART_A)
      wire#w8
      S_Coil( "DB8101_MANUAL_LOADING_PART_STATUS_MANAGEMENT".UNIT_01_UNIT_02_INTERMEDIATE.STATUS.PRESENT )
      S_Coil( "DB8101_MANUAL_LOADING_PART_STATUS_MANAGEMENT".UNIT_01_UNIT_02_INTERMEDIATE.STATUS.OK )
   END_RUNG
   RUNG wire#w8
      R_Coil( "DB8000_PART_STATUS".UNIT_01.FIXTURE_4.PART_A.STATUS.PRESENT )
      R_Coil( "DB8000_PART_STATUS".UNIT_01.FIXTURE_4.PART_A.STATUS.OK )
   END_RUNG
   // the same network as SCL:
   // ENO of a box is taken as its EN; it also drops when the box reports an error
   #_w1 := "DB7240_HARDWARE_SOFTWARE_ENABLE_DISABLE".DISABLE_FIXTURE.SW_UNIT_01_FIX_1_4_ENABLED AND "DB4000_FIX_TABLE_POSITIONS".UNIT_01.FIXTURE_4.IN_LOAD_UNLOAD_STATION_1 AND "DB2440_GLOBAL_DATA".GLOBAL_DATA.U01_RN_CYCLE_PART_TYPE;
   #_w2 := #_w1 AND "DB2099_MANUAL_LOAD_DMC".MANUAL_LOADING_OR_DRY_PART_LOADED_UNIT_01_P;
   #_w3 := #_w2 AND NOT "DB2099_MANUAL_LOAD_DMC".PRODUCTION_SELECTED;
   IF #_w3 THEN
       "DB8000_PART_STATUS".UNIT_01.FIXTURE_4.PART_A.STATUS.PART_TYPE := "DB7215_PART_TYPE".Part_Type_Low;
       "DB8000_PART_STATUS".UNIT_01.FIXTURE_4.PART_A.PART_ID := "DB2099_MANUAL_LOAD_DMC".DMC_ARRAY_CHAR_UNIT_01;
       "DB8000_PART_STATUS".UNIT_01.FIXTURE_4.PART_A.STATUS.PRESENT := TRUE;
       "DB8000_PART_STATUS".UNIT_01.FIXTURE_4.PART_A.STATUS.OK := TRUE;
   END_IF;
   IF #_w3 AND NOT "DB2031_CYCLES_GENERAL".CALIBRATION_CYCLE.CYCLE_SELECTED THEN
       "DB8000_PART_STATUS".UNIT_01.FIXTURE_4.PART_A.STATUS.CELL_STATUS.U01_ONE_FACE_DONE_ROTATED := TRUE;
   END_IF;
   IF #_w3 AND ("DB2031_CYCLES_GENERAL".CALIBRATION_CYCLE.CYCLE_SELECTED OR "DB2031_CYCLES_GENERAL".MASTER_MEASUREMENT.CYCLE_SELECTED) THEN
       "DB8000_PART_STATUS".UNIT_01.FIXTURE_4.PART_A.STATUS.MASTER_PART := TRUE;
   END_IF;
   #_w4 := #_w2 AND "DB2099_MANUAL_LOAD_DMC".PRODUCTION_SELECTED;
   #STATUS_FILL := FILL(EN := #_w4,
                        BVAL := #ZERO,
                        BLK => "DB8101_MANUAL_LOADING_PART_STATUS_MANAGEMENT".UNIT_01_INTERMEDIATE.STATUS,
                        ENO => #_w5);
   #STATUS_BLKMOV := BLKMOV(EN := #_w5,
                           SRCBLK := "DB8101_MANUAL_LOADING_PART_STATUS_MANAGEMENT".UNIT_01_INTERMEDIATE,
                           DSTBLK => "DB8000_PART_STATUS".UNIT_01.FIXTURE_4.PART_A,
                           ENO => #_w6);
   #STATUS_FILL := FILL(EN := #_w6,
                        BVAL := #ZERO,
                        BLK => "DB8101_MANUAL_LOADING_PART_STATUS_MANAGEMENT".UNIT_01_INTERMEDIATE,
                        ENO => #_w7);
   IF #_w7 THEN
       "DB8000_PART_STATUS".UNIT_01.FIXTURE_4.PART_A.STATUS.PRESENT := TRUE;
       "DB8000_PART_STATUS".UNIT_01.FIXTURE_4.PART_A.STATUS.OK := TRUE;
       "DB8101_MANUAL_LOADING_PART_STATUS_MANAGEMENT".UNIT_01_INTERMEDIATE.STATUS.PRESENT := FALSE;
       "DB8101_MANUAL_LOADING_PART_STATUS_MANAGEMENT".UNIT_01_INTERMEDIATE.STATUS.OK := FALSE;
   END_IF;
   IF #_w7 AND NOT "DB2031_CYCLES_GENERAL".CALIBRATION_CYCLE.CYCLE_SELECTED THEN
       "DB8000_PART_STATUS".UNIT_01.FIXTURE_4.PART_A.STATUS.CELL_STATUS.U01_ONE_FACE_DONE_ROTATED := TRUE;
   END_IF;
   IF #_w7 AND "DB2031_CYCLES_GENERAL".CALIBRATION_CYCLE.CYCLE_SELECTED THEN
       "DB8000_PART_STATUS".UNIT_01.FIXTURE_4.PART_A.STATUS.MASTER_PART := TRUE;
   END_IF;
   #_w8 := #_w1 AND "DB2099_MANUAL_LOAD_DMC".MANUAL_LOADING_OR_DRY_PART_UNLOADED_UNIT_01_P;
   #STATUS_FILL := FILL(EN := #_w8 AND NOT "DB2099_MANUAL_LOAD_DMC".PRODUCTION_SELECTED,
                        BVAL := #ZERO,
                        BLK => "DB8000_PART_STATUS".UNIT_01.FIXTURE_4.PART_A,
                        ENO => #_w9);
   IF #_w9 THEN
       "DB8000_PART_STATUS".UNIT_01.FIXTURE_4.PART_A.STATUS.PRESENT := FALSE;
       "DB8000_PART_STATUS".UNIT_01.FIXTURE_4.PART_A.STATUS.OK := FALSE;
   END_IF;
   #STATUS_BLKMOV := BLKMOV(EN := #_w8 AND "DB2099_MANUAL_LOAD_DMC".PRODUCTION_SELECTED,
                           SRCBLK := "DB8000_PART_STATUS".UNIT_01.FIXTURE_4.PART_A,
                           DSTBLK => "DB8101_MANUAL_LOADING_PART_STATUS_MANAGEMENT".UNIT_01_UNIT_02_INTERMEDIATE,
                           ENO => #_w10);
   #STATUS_FILL := FILL(EN := #_w10,
                        BVAL := #ZERO,
                        BLK => "DB8000_PART_STATUS".UNIT_01.FIXTURE_4.PART_A,
                        ENO => #_w11);
   IF #_w11 THEN
       "DB8101_MANUAL_LOADING_PART_STATUS_MANAGEMENT".UNIT_01_UNIT_02_INTERMEDIATE.STATUS.PRESENT := TRUE;
       "DB8101_MANUAL_LOADING_PART_STATUS_MANAGEMENT".UNIT_01_UNIT_02_INTERMEDIATE.STATUS.OK := TRUE;
       "DB8000_PART_STATUS".UNIT_01.FIXTURE_4.PART_A.STATUS.PRESENT := FALSE;
       "DB8000_PART_STATUS".UNIT_01.FIXTURE_4.PART_A.STATUS.OK := FALSE;
   END_IF;
END_REGION

REGION Network 8: <<<<<<<<<<<<<<<<<<<< UNIT 02 >>>>>>>>>>>>>>>>>>>>
END_REGION

REGION Network 9: UNIT 02 FIXTURE 1 PART A PRESENT
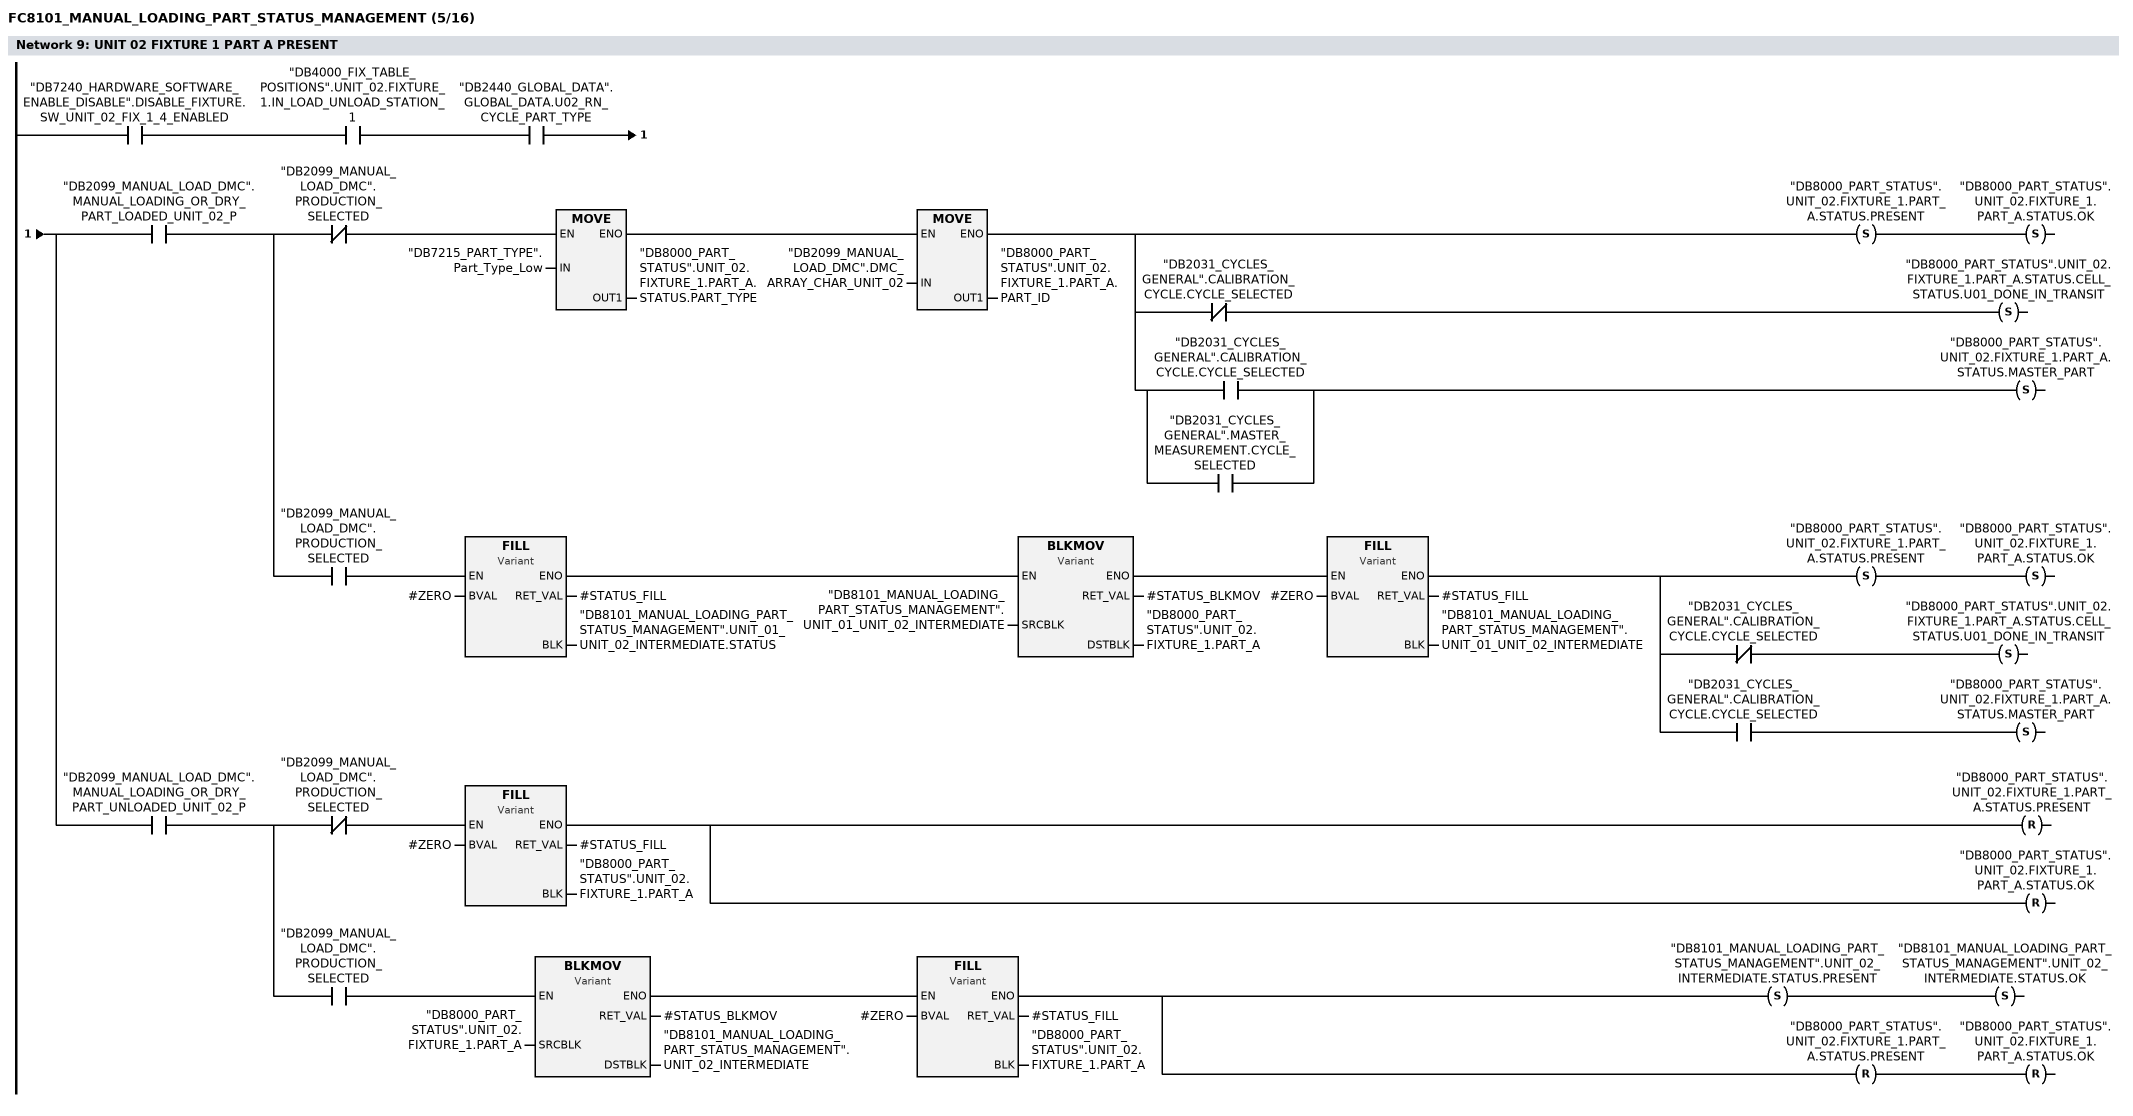
   RUNG wire#powerrail
      Contact( "DB7240_HARDWARE_SOFTWARE_ENABLE_DISABLE".DISABLE_FIXTURE.SW_UNIT_02_FIX_1_4_ENABLED )
      Contact( "DB4000_FIX_TABLE_POSITIONS".UNIT_02.FIXTURE_1.IN_LOAD_UNLOAD_STATION_1 )
      Contact( "DB2440_GLOBAL_DATA".GLOBAL_DATA.U02_RN_CYCLE_PART_TYPE )
      wire#w1
      Contact( "DB2099_MANUAL_LOAD_DMC".MANUAL_LOADING_OR_DRY_PART_LOADED_UNIT_02_P )
      wire#w2
      I_Contact( "DB2099_MANUAL_LOAD_DMC".PRODUCTION_SELECTED )
      { S7_GenerateENO := "TRUE" } Move(in := "DB7215_PART_TYPE".Part_Type_Low, out1 => "DB8000_PART_STATUS".UNIT_02.FIXTURE_1.PART_A.STATUS.PART_TYPE)
      Move(in := "DB2099_MANUAL_LOAD_DMC".DMC_ARRAY_CHAR_UNIT_02, out1 => "DB8000_PART_STATUS".UNIT_02.FIXTURE_1.PART_A.PART_ID)
      wire#w3
      S_Coil( "DB8000_PART_STATUS".UNIT_02.FIXTURE_1.PART_A.STATUS.PRESENT )
      S_Coil( "DB8000_PART_STATUS".UNIT_02.FIXTURE_1.PART_A.STATUS.OK )
   END_RUNG
   RUNG wire#w3
      I_Contact( "DB2031_CYCLES_GENERAL".CALIBRATION_CYCLE.CYCLE_SELECTED )
      S_Coil( "DB8000_PART_STATUS".UNIT_02.FIXTURE_1.PART_A.STATUS.CELL_STATUS.U01_DONE_IN_TRANSIT )
   END_RUNG
   RUNG wire#w3
      Contact( "DB2031_CYCLES_GENERAL".CALIBRATION_CYCLE.CYCLE_SELECTED )
      wire#w4
      S_Coil( "DB8000_PART_STATUS".UNIT_02.FIXTURE_1.PART_A.STATUS.MASTER_PART )
   END_RUNG
   RUNG wire#w3
      Contact( "DB2031_CYCLES_GENERAL".MASTER_MEASUREMENT.CYCLE_SELECTED )
   END_RUNG wire#w4
   RUNG wire#w2
      Contact( "DB2099_MANUAL_LOAD_DMC".PRODUCTION_SELECTED )
      { S7_Templates := "ptr_type := Variant" } FILL(BVAL := #ZERO, RET_VAL => #STATUS_FILL, BLK => "DB8101_MANUAL_LOADING_PART_STATUS_MANAGEMENT".UNIT_01_UNIT_02_INTERMEDIATE.STATUS)
      { S7_Templates := "blk_type := Variant" } BLKMOV(SRCBLK := "DB8101_MANUAL_LOADING_PART_STATUS_MANAGEMENT".UNIT_01_UNIT_02_INTERMEDIATE, RET_VAL => #STATUS_BLKMOV, DSTBLK => "DB8000_PART_STATUS".UNIT_02.FIXTURE_1.PART_A)
      { S7_Templates := "ptr_type := Variant" } FILL(BVAL := #ZERO, RET_VAL => #STATUS_FILL, BLK => "DB8101_MANUAL_LOADING_PART_STATUS_MANAGEMENT".UNIT_01_UNIT_02_INTERMEDIATE)
      wire#w5
      S_Coil( "DB8000_PART_STATUS".UNIT_02.FIXTURE_1.PART_A.STATUS.PRESENT )
      S_Coil( "DB8000_PART_STATUS".UNIT_02.FIXTURE_1.PART_A.STATUS.OK )
   END_RUNG
   RUNG wire#w5
      I_Contact( "DB2031_CYCLES_GENERAL".CALIBRATION_CYCLE.CYCLE_SELECTED )
      S_Coil( "DB8000_PART_STATUS".UNIT_02.FIXTURE_1.PART_A.STATUS.CELL_STATUS.U01_DONE_IN_TRANSIT )
   END_RUNG
   RUNG wire#w5
      Contact( "DB2031_CYCLES_GENERAL".CALIBRATION_CYCLE.CYCLE_SELECTED )
      S_Coil( "DB8000_PART_STATUS".UNIT_02.FIXTURE_1.PART_A.STATUS.MASTER_PART )
   END_RUNG
   RUNG wire#w1
      Contact( "DB2099_MANUAL_LOAD_DMC".MANUAL_LOADING_OR_DRY_PART_UNLOADED_UNIT_02_P )
      wire#w6
      I_Contact( "DB2099_MANUAL_LOAD_DMC".PRODUCTION_SELECTED )
      { S7_Templates := "ptr_type := Variant" } FILL(BVAL := #ZERO, RET_VAL => #STATUS_FILL, BLK => "DB8000_PART_STATUS".UNIT_02.FIXTURE_1.PART_A)
      wire#w7
      R_Coil( "DB8000_PART_STATUS".UNIT_02.FIXTURE_1.PART_A.STATUS.PRESENT )
   END_RUNG
   RUNG wire#w7
      R_Coil( "DB8000_PART_STATUS".UNIT_02.FIXTURE_1.PART_A.STATUS.OK )
   END_RUNG
   RUNG wire#w6
      Contact( "DB2099_MANUAL_LOAD_DMC".PRODUCTION_SELECTED )
      { S7_Templates := "blk_type := Variant" } BLKMOV(SRCBLK := "DB8000_PART_STATUS".UNIT_02.FIXTURE_1.PART_A, RET_VAL => #STATUS_BLKMOV, DSTBLK => "DB8101_MANUAL_LOADING_PART_STATUS_MANAGEMENT".UNIT_02_INTERMEDIATE)
      { S7_Templates := "ptr_type := Variant" } FILL(BVAL := #ZERO, RET_VAL => #STATUS_FILL, BLK => "DB8000_PART_STATUS".UNIT_02.FIXTURE_1.PART_A)
      wire#w8
      S_Coil( "DB8101_MANUAL_LOADING_PART_STATUS_MANAGEMENT".UNIT_02_INTERMEDIATE.STATUS.PRESENT )
      S_Coil( "DB8101_MANUAL_LOADING_PART_STATUS_MANAGEMENT".UNIT_02_INTERMEDIATE.STATUS.OK )
   END_RUNG
   RUNG wire#w8
      R_Coil( "DB8000_PART_STATUS".UNIT_02.FIXTURE_1.PART_A.STATUS.PRESENT )
      R_Coil( "DB8000_PART_STATUS".UNIT_02.FIXTURE_1.PART_A.STATUS.OK )
   END_RUNG
   // the same network as SCL:
   // ENO of a box is taken as its EN; it also drops when the box reports an error
   #_w1 := "DB7240_HARDWARE_SOFTWARE_ENABLE_DISABLE".DISABLE_FIXTURE.SW_UNIT_02_FIX_1_4_ENABLED AND "DB4000_FIX_TABLE_POSITIONS".UNIT_02.FIXTURE_1.IN_LOAD_UNLOAD_STATION_1 AND "DB2440_GLOBAL_DATA".GLOBAL_DATA.U02_RN_CYCLE_PART_TYPE;
   #_w2 := #_w1 AND "DB2099_MANUAL_LOAD_DMC".MANUAL_LOADING_OR_DRY_PART_LOADED_UNIT_02_P;
   #_w3 := #_w2 AND NOT "DB2099_MANUAL_LOAD_DMC".PRODUCTION_SELECTED;
   IF #_w3 THEN
       "DB8000_PART_STATUS".UNIT_02.FIXTURE_1.PART_A.STATUS.PART_TYPE := "DB7215_PART_TYPE".Part_Type_Low;
       "DB8000_PART_STATUS".UNIT_02.FIXTURE_1.PART_A.PART_ID := "DB2099_MANUAL_LOAD_DMC".DMC_ARRAY_CHAR_UNIT_02;
       "DB8000_PART_STATUS".UNIT_02.FIXTURE_1.PART_A.STATUS.PRESENT := TRUE;
       "DB8000_PART_STATUS".UNIT_02.FIXTURE_1.PART_A.STATUS.OK := TRUE;
   END_IF;
   IF #_w3 AND NOT "DB2031_CYCLES_GENERAL".CALIBRATION_CYCLE.CYCLE_SELECTED THEN
       "DB8000_PART_STATUS".UNIT_02.FIXTURE_1.PART_A.STATUS.CELL_STATUS.U01_DONE_IN_TRANSIT := TRUE;
   END_IF;
   IF #_w3 AND ("DB2031_CYCLES_GENERAL".CALIBRATION_CYCLE.CYCLE_SELECTED OR "DB2031_CYCLES_GENERAL".MASTER_MEASUREMENT.CYCLE_SELECTED) THEN
       "DB8000_PART_STATUS".UNIT_02.FIXTURE_1.PART_A.STATUS.MASTER_PART := TRUE;
   END_IF;
   #_w4 := #_w2 AND "DB2099_MANUAL_LOAD_DMC".PRODUCTION_SELECTED;
   #STATUS_FILL := FILL(EN := #_w4,
                        BVAL := #ZERO,
                        BLK => "DB8101_MANUAL_LOADING_PART_STATUS_MANAGEMENT".UNIT_01_UNIT_02_INTERMEDIATE.STATUS,
                        ENO => #_w5);
   #STATUS_BLKMOV := BLKMOV(EN := #_w5,
                           SRCBLK := "DB8101_MANUAL_LOADING_PART_STATUS_MANAGEMENT".UNIT_01_UNIT_02_INTERMEDIATE,
                           DSTBLK => "DB8000_PART_STATUS".UNIT_02.FIXTURE_1.PART_A,
                           ENO => #_w6);
   #STATUS_FILL := FILL(EN := #_w6,
                        BVAL := #ZERO,
                        BLK => "DB8101_MANUAL_LOADING_PART_STATUS_MANAGEMENT".UNIT_01_UNIT_02_INTERMEDIATE,
                        ENO => #_w7);
   IF #_w7 THEN
       "DB8000_PART_STATUS".UNIT_02.FIXTURE_1.PART_A.STATUS.PRESENT := TRUE;
       "DB8000_PART_STATUS".UNIT_02.FIXTURE_1.PART_A.STATUS.OK := TRUE;
   END_IF;
   IF #_w7 AND NOT "DB2031_CYCLES_GENERAL".CALIBRATION_CYCLE.CYCLE_SELECTED THEN
       "DB8000_PART_STATUS".UNIT_02.FIXTURE_1.PART_A.STATUS.CELL_STATUS.U01_DONE_IN_TRANSIT := TRUE;
   END_IF;
   IF #_w7 AND "DB2031_CYCLES_GENERAL".CALIBRATION_CYCLE.CYCLE_SELECTED THEN
       "DB8000_PART_STATUS".UNIT_02.FIXTURE_1.PART_A.STATUS.MASTER_PART := TRUE;
   END_IF;
   #_w8 := #_w1 AND "DB2099_MANUAL_LOAD_DMC".MANUAL_LOADING_OR_DRY_PART_UNLOADED_UNIT_02_P;
   #STATUS_FILL := FILL(EN := #_w8 AND NOT "DB2099_MANUAL_LOAD_DMC".PRODUCTION_SELECTED,
                        BVAL := #ZERO,
                        BLK => "DB8000_PART_STATUS".UNIT_02.FIXTURE_1.PART_A,
                        ENO => #_w9);
   IF #_w9 THEN
       "DB8000_PART_STATUS".UNIT_02.FIXTURE_1.PART_A.STATUS.PRESENT := FALSE;
       "DB8000_PART_STATUS".UNIT_02.FIXTURE_1.PART_A.STATUS.OK := FALSE;
   END_IF;
   #STATUS_BLKMOV := BLKMOV(EN := #_w8 AND "DB2099_MANUAL_LOAD_DMC".PRODUCTION_SELECTED,
                           SRCBLK := "DB8000_PART_STATUS".UNIT_02.FIXTURE_1.PART_A,
                           DSTBLK => "DB8101_MANUAL_LOADING_PART_STATUS_MANAGEMENT".UNIT_02_INTERMEDIATE,
                           ENO => #_w10);
   #STATUS_FILL := FILL(EN := #_w10,
                        BVAL := #ZERO,
                        BLK => "DB8000_PART_STATUS".UNIT_02.FIXTURE_1.PART_A,
                        ENO => #_w11);
   IF #_w11 THEN
       "DB8101_MANUAL_LOADING_PART_STATUS_MANAGEMENT".UNIT_02_INTERMEDIATE.STATUS.PRESENT := TRUE;
       "DB8101_MANUAL_LOADING_PART_STATUS_MANAGEMENT".UNIT_02_INTERMEDIATE.STATUS.OK := TRUE;
       "DB8000_PART_STATUS".UNIT_02.FIXTURE_1.PART_A.STATUS.PRESENT := FALSE;
       "DB8000_PART_STATUS".UNIT_02.FIXTURE_1.PART_A.STATUS.OK := FALSE;
   END_IF;
END_REGION

REGION Network 10: UNIT 02 FIXTURE 2 PART A PRESENT
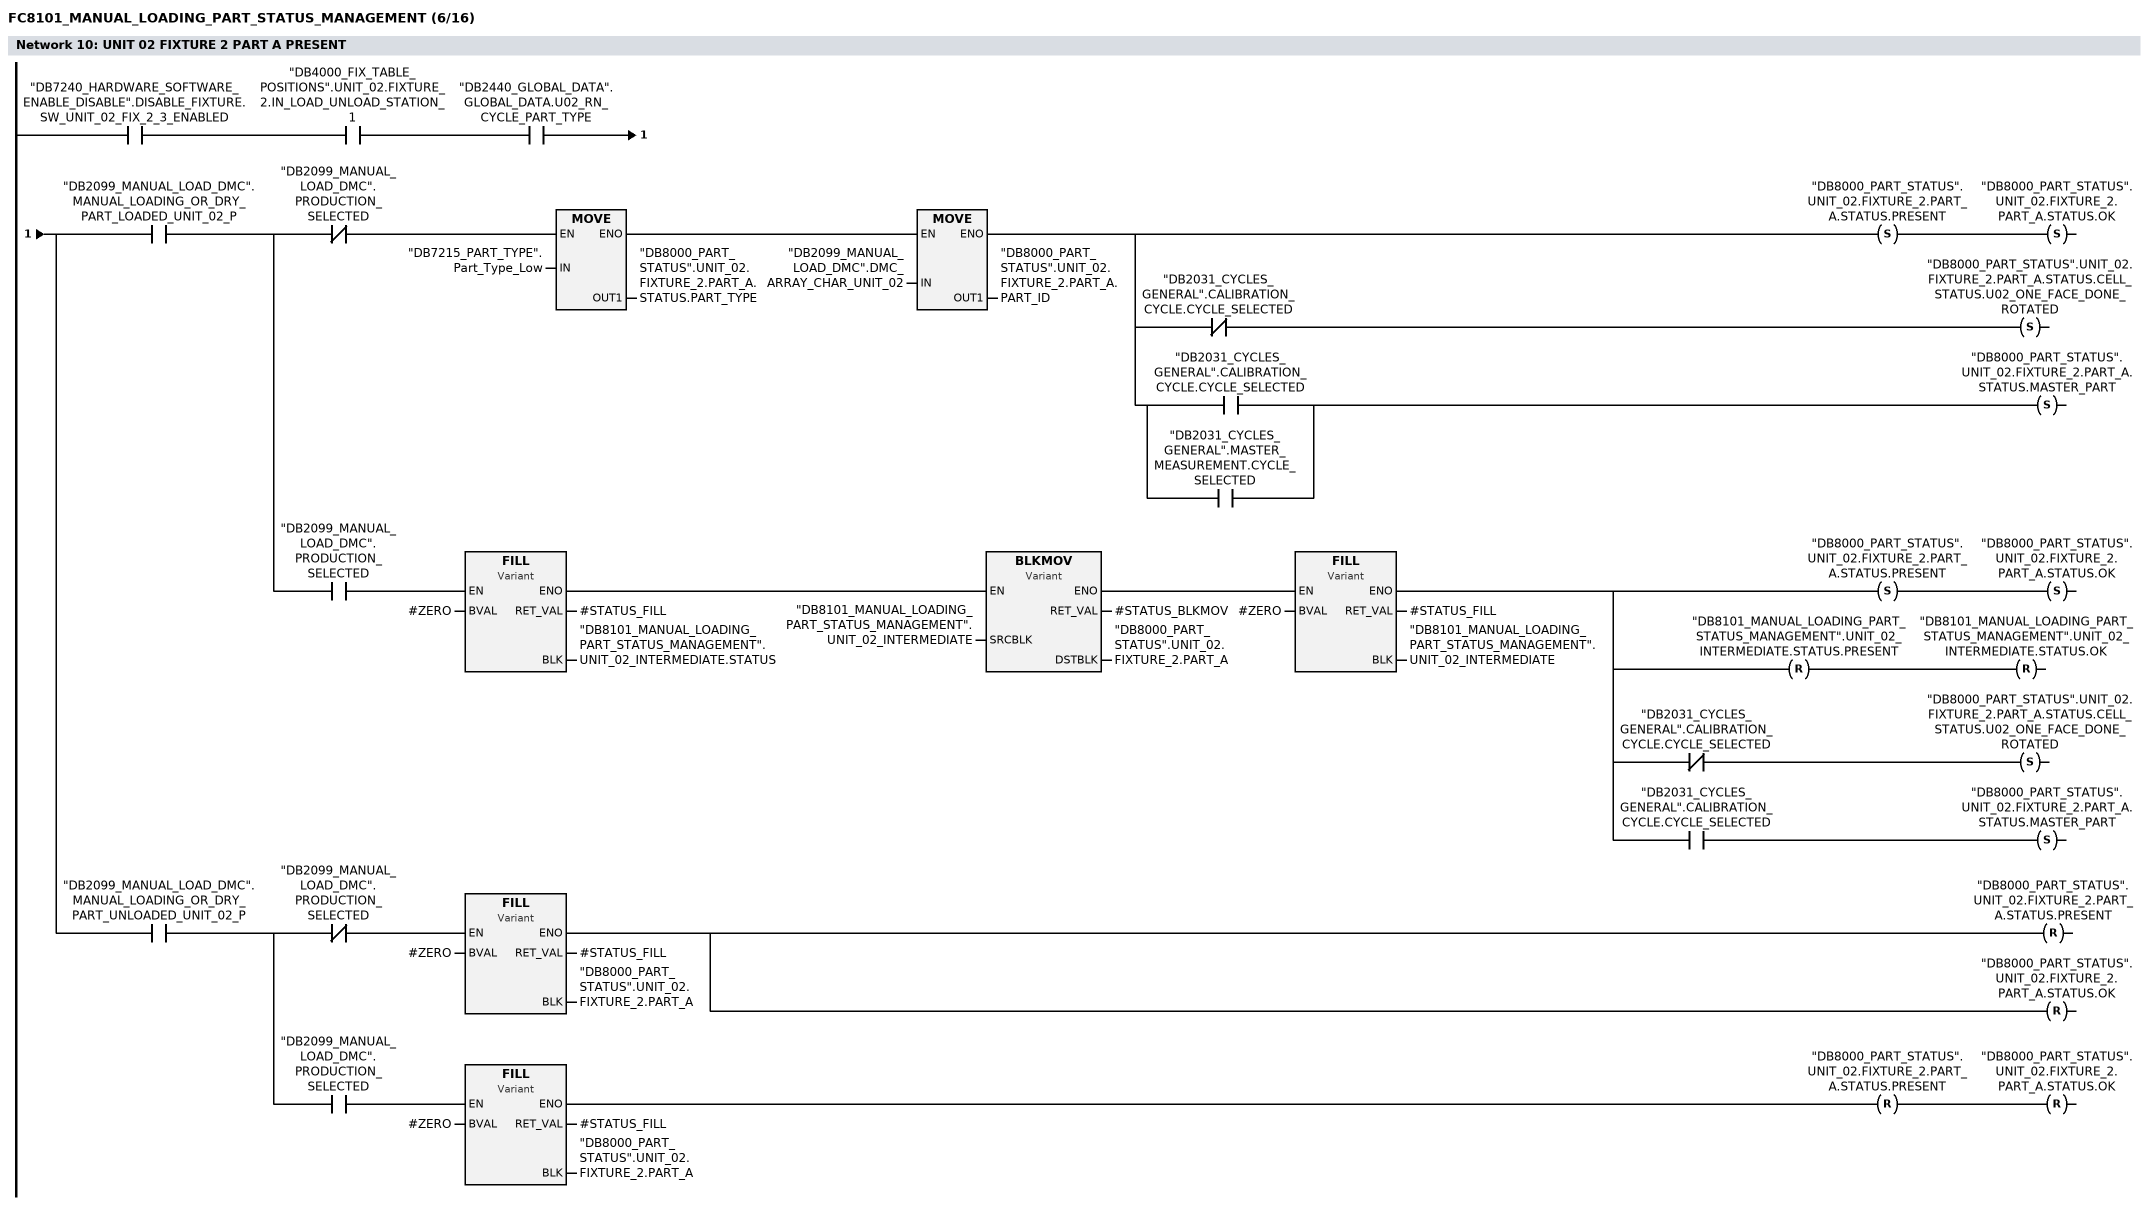
   RUNG wire#powerrail
      Contact( "DB7240_HARDWARE_SOFTWARE_ENABLE_DISABLE".DISABLE_FIXTURE.SW_UNIT_02_FIX_2_3_ENABLED )
      Contact( "DB4000_FIX_TABLE_POSITIONS".UNIT_02.FIXTURE_2.IN_LOAD_UNLOAD_STATION_1 )
      Contact( "DB2440_GLOBAL_DATA".GLOBAL_DATA.U02_RN_CYCLE_PART_TYPE )
      wire#w1
      Contact( "DB2099_MANUAL_LOAD_DMC".MANUAL_LOADING_OR_DRY_PART_LOADED_UNIT_02_P )
      wire#w2
      I_Contact( "DB2099_MANUAL_LOAD_DMC".PRODUCTION_SELECTED )
      { S7_GenerateENO := "TRUE" } Move(in := "DB7215_PART_TYPE".Part_Type_Low, out1 => "DB8000_PART_STATUS".UNIT_02.FIXTURE_2.PART_A.STATUS.PART_TYPE)
      Move(in := "DB2099_MANUAL_LOAD_DMC".DMC_ARRAY_CHAR_UNIT_02, out1 => "DB8000_PART_STATUS".UNIT_02.FIXTURE_2.PART_A.PART_ID)
      wire#w3
      S_Coil( "DB8000_PART_STATUS".UNIT_02.FIXTURE_2.PART_A.STATUS.PRESENT )
      S_Coil( "DB8000_PART_STATUS".UNIT_02.FIXTURE_2.PART_A.STATUS.OK )
   END_RUNG
   RUNG wire#w3
      I_Contact( "DB2031_CYCLES_GENERAL".CALIBRATION_CYCLE.CYCLE_SELECTED )
      S_Coil( "DB8000_PART_STATUS".UNIT_02.FIXTURE_2.PART_A.STATUS.CELL_STATUS.U02_ONE_FACE_DONE_ROTATED )
   END_RUNG
   RUNG wire#w3
      Contact( "DB2031_CYCLES_GENERAL".CALIBRATION_CYCLE.CYCLE_SELECTED )
      wire#w4
      S_Coil( "DB8000_PART_STATUS".UNIT_02.FIXTURE_2.PART_A.STATUS.MASTER_PART )
   END_RUNG
   RUNG wire#w3
      Contact( "DB2031_CYCLES_GENERAL".MASTER_MEASUREMENT.CYCLE_SELECTED )
   END_RUNG wire#w4
   RUNG wire#w2
      Contact( "DB2099_MANUAL_LOAD_DMC".PRODUCTION_SELECTED )
      { S7_Templates := "ptr_type := Variant" } FILL(BVAL := #ZERO, RET_VAL => #STATUS_FILL, BLK => "DB8101_MANUAL_LOADING_PART_STATUS_MANAGEMENT".UNIT_02_INTERMEDIATE.STATUS)
      { S7_Templates := "blk_type := Variant" } BLKMOV(SRCBLK := "DB8101_MANUAL_LOADING_PART_STATUS_MANAGEMENT".UNIT_02_INTERMEDIATE, RET_VAL => #STATUS_BLKMOV, DSTBLK => "DB8000_PART_STATUS".UNIT_02.FIXTURE_2.PART_A)
      { S7_Templates := "ptr_type := Variant" } FILL(BVAL := #ZERO, RET_VAL => #STATUS_FILL, BLK => "DB8101_MANUAL_LOADING_PART_STATUS_MANAGEMENT".UNIT_02_INTERMEDIATE)
      wire#w5
      S_Coil( "DB8000_PART_STATUS".UNIT_02.FIXTURE_2.PART_A.STATUS.PRESENT )
      S_Coil( "DB8000_PART_STATUS".UNIT_02.FIXTURE_2.PART_A.STATUS.OK )
   END_RUNG
   RUNG wire#w5
      R_Coil( "DB8101_MANUAL_LOADING_PART_STATUS_MANAGEMENT".UNIT_02_INTERMEDIATE.STATUS.PRESENT )
      R_Coil( "DB8101_MANUAL_LOADING_PART_STATUS_MANAGEMENT".UNIT_02_INTERMEDIATE.STATUS.OK )
   END_RUNG
   RUNG wire#w5
      I_Contact( "DB2031_CYCLES_GENERAL".CALIBRATION_CYCLE.CYCLE_SELECTED )
      S_Coil( "DB8000_PART_STATUS".UNIT_02.FIXTURE_2.PART_A.STATUS.CELL_STATUS.U02_ONE_FACE_DONE_ROTATED )
   END_RUNG
   RUNG wire#w5
      Contact( "DB2031_CYCLES_GENERAL".CALIBRATION_CYCLE.CYCLE_SELECTED )
      S_Coil( "DB8000_PART_STATUS".UNIT_02.FIXTURE_2.PART_A.STATUS.MASTER_PART )
   END_RUNG
   RUNG wire#w1
      Contact( "DB2099_MANUAL_LOAD_DMC".MANUAL_LOADING_OR_DRY_PART_UNLOADED_UNIT_02_P )
      wire#w6
      I_Contact( "DB2099_MANUAL_LOAD_DMC".PRODUCTION_SELECTED )
      { S7_Templates := "ptr_type := Variant" } FILL(BVAL := #ZERO, RET_VAL => #STATUS_FILL, BLK => "DB8000_PART_STATUS".UNIT_02.FIXTURE_2.PART_A)
      wire#w7
      R_Coil( "DB8000_PART_STATUS".UNIT_02.FIXTURE_2.PART_A.STATUS.PRESENT )
   END_RUNG
   RUNG wire#w7
      R_Coil( "DB8000_PART_STATUS".UNIT_02.FIXTURE_2.PART_A.STATUS.OK )
   END_RUNG
   RUNG wire#w6
      Contact( "DB2099_MANUAL_LOAD_DMC".PRODUCTION_SELECTED )
      { S7_Templates := "ptr_type := Variant" } FILL(BVAL := #ZERO, RET_VAL => #STATUS_FILL, BLK => "DB8000_PART_STATUS".UNIT_02.FIXTURE_2.PART_A)
      R_Coil( "DB8000_PART_STATUS".UNIT_02.FIXTURE_2.PART_A.STATUS.PRESENT )
      R_Coil( "DB8000_PART_STATUS".UNIT_02.FIXTURE_2.PART_A.STATUS.OK )
   END_RUNG
   // the same network as SCL:
   // ENO of a box is taken as its EN; it also drops when the box reports an error
   #_w1 := "DB7240_HARDWARE_SOFTWARE_ENABLE_DISABLE".DISABLE_FIXTURE.SW_UNIT_02_FIX_2_3_ENABLED AND "DB4000_FIX_TABLE_POSITIONS".UNIT_02.FIXTURE_2.IN_LOAD_UNLOAD_STATION_1 AND "DB2440_GLOBAL_DATA".GLOBAL_DATA.U02_RN_CYCLE_PART_TYPE;
   #_w2 := #_w1 AND "DB2099_MANUAL_LOAD_DMC".MANUAL_LOADING_OR_DRY_PART_LOADED_UNIT_02_P;
   #_w3 := #_w2 AND NOT "DB2099_MANUAL_LOAD_DMC".PRODUCTION_SELECTED;
   IF #_w3 THEN
       "DB8000_PART_STATUS".UNIT_02.FIXTURE_2.PART_A.STATUS.PART_TYPE := "DB7215_PART_TYPE".Part_Type_Low;
       "DB8000_PART_STATUS".UNIT_02.FIXTURE_2.PART_A.PART_ID := "DB2099_MANUAL_LOAD_DMC".DMC_ARRAY_CHAR_UNIT_02;
       "DB8000_PART_STATUS".UNIT_02.FIXTURE_2.PART_A.STATUS.PRESENT := TRUE;
       "DB8000_PART_STATUS".UNIT_02.FIXTURE_2.PART_A.STATUS.OK := TRUE;
   END_IF;
   IF #_w3 AND NOT "DB2031_CYCLES_GENERAL".CALIBRATION_CYCLE.CYCLE_SELECTED THEN
       "DB8000_PART_STATUS".UNIT_02.FIXTURE_2.PART_A.STATUS.CELL_STATUS.U02_ONE_FACE_DONE_ROTATED := TRUE;
   END_IF;
   IF #_w3 AND ("DB2031_CYCLES_GENERAL".CALIBRATION_CYCLE.CYCLE_SELECTED OR "DB2031_CYCLES_GENERAL".MASTER_MEASUREMENT.CYCLE_SELECTED) THEN
       "DB8000_PART_STATUS".UNIT_02.FIXTURE_2.PART_A.STATUS.MASTER_PART := TRUE;
   END_IF;
   #_w4 := #_w2 AND "DB2099_MANUAL_LOAD_DMC".PRODUCTION_SELECTED;
   #STATUS_FILL := FILL(EN := #_w4,
                        BVAL := #ZERO,
                        BLK => "DB8101_MANUAL_LOADING_PART_STATUS_MANAGEMENT".UNIT_02_INTERMEDIATE.STATUS,
                        ENO => #_w5);
   #STATUS_BLKMOV := BLKMOV(EN := #_w5,
                           SRCBLK := "DB8101_MANUAL_LOADING_PART_STATUS_MANAGEMENT".UNIT_02_INTERMEDIATE,
                           DSTBLK => "DB8000_PART_STATUS".UNIT_02.FIXTURE_2.PART_A,
                           ENO => #_w6);
   #STATUS_FILL := FILL(EN := #_w6,
                        BVAL := #ZERO,
                        BLK => "DB8101_MANUAL_LOADING_PART_STATUS_MANAGEMENT".UNIT_02_INTERMEDIATE,
                        ENO => #_w7);
   IF #_w7 THEN
       "DB8000_PART_STATUS".UNIT_02.FIXTURE_2.PART_A.STATUS.PRESENT := TRUE;
       "DB8000_PART_STATUS".UNIT_02.FIXTURE_2.PART_A.STATUS.OK := TRUE;
       "DB8101_MANUAL_LOADING_PART_STATUS_MANAGEMENT".UNIT_02_INTERMEDIATE.STATUS.PRESENT := FALSE;
       "DB8101_MANUAL_LOADING_PART_STATUS_MANAGEMENT".UNIT_02_INTERMEDIATE.STATUS.OK := FALSE;
   END_IF;
   IF #_w7 AND NOT "DB2031_CYCLES_GENERAL".CALIBRATION_CYCLE.CYCLE_SELECTED THEN
       "DB8000_PART_STATUS".UNIT_02.FIXTURE_2.PART_A.STATUS.CELL_STATUS.U02_ONE_FACE_DONE_ROTATED := TRUE;
   END_IF;
   IF #_w7 AND "DB2031_CYCLES_GENERAL".CALIBRATION_CYCLE.CYCLE_SELECTED THEN
       "DB8000_PART_STATUS".UNIT_02.FIXTURE_2.PART_A.STATUS.MASTER_PART := TRUE;
   END_IF;
   #_w8 := #_w1 AND "DB2099_MANUAL_LOAD_DMC".MANUAL_LOADING_OR_DRY_PART_UNLOADED_UNIT_02_P;
   #STATUS_FILL := FILL(EN := #_w8 AND NOT "DB2099_MANUAL_LOAD_DMC".PRODUCTION_SELECTED,
                        BVAL := #ZERO,
                        BLK => "DB8000_PART_STATUS".UNIT_02.FIXTURE_2.PART_A,
                        ENO => #_w9);
   IF #_w9 THEN
       "DB8000_PART_STATUS".UNIT_02.FIXTURE_2.PART_A.STATUS.PRESENT := FALSE;
       "DB8000_PART_STATUS".UNIT_02.FIXTURE_2.PART_A.STATUS.OK := FALSE;
   END_IF;
   #STATUS_FILL := FILL(EN := #_w8 AND "DB2099_MANUAL_LOAD_DMC".PRODUCTION_SELECTED,
                        BVAL := #ZERO,
                        BLK => "DB8000_PART_STATUS".UNIT_02.FIXTURE_2.PART_A,
                        ENO => #_w10);
   IF #_w10 THEN
       "DB8000_PART_STATUS".UNIT_02.FIXTURE_2.PART_A.STATUS.PRESENT := FALSE;
       "DB8000_PART_STATUS".UNIT_02.FIXTURE_2.PART_A.STATUS.OK := FALSE;
   END_IF;
END_REGION

REGION Network 11: UNIT 02 FIXTURE 3 PART A PRESENT
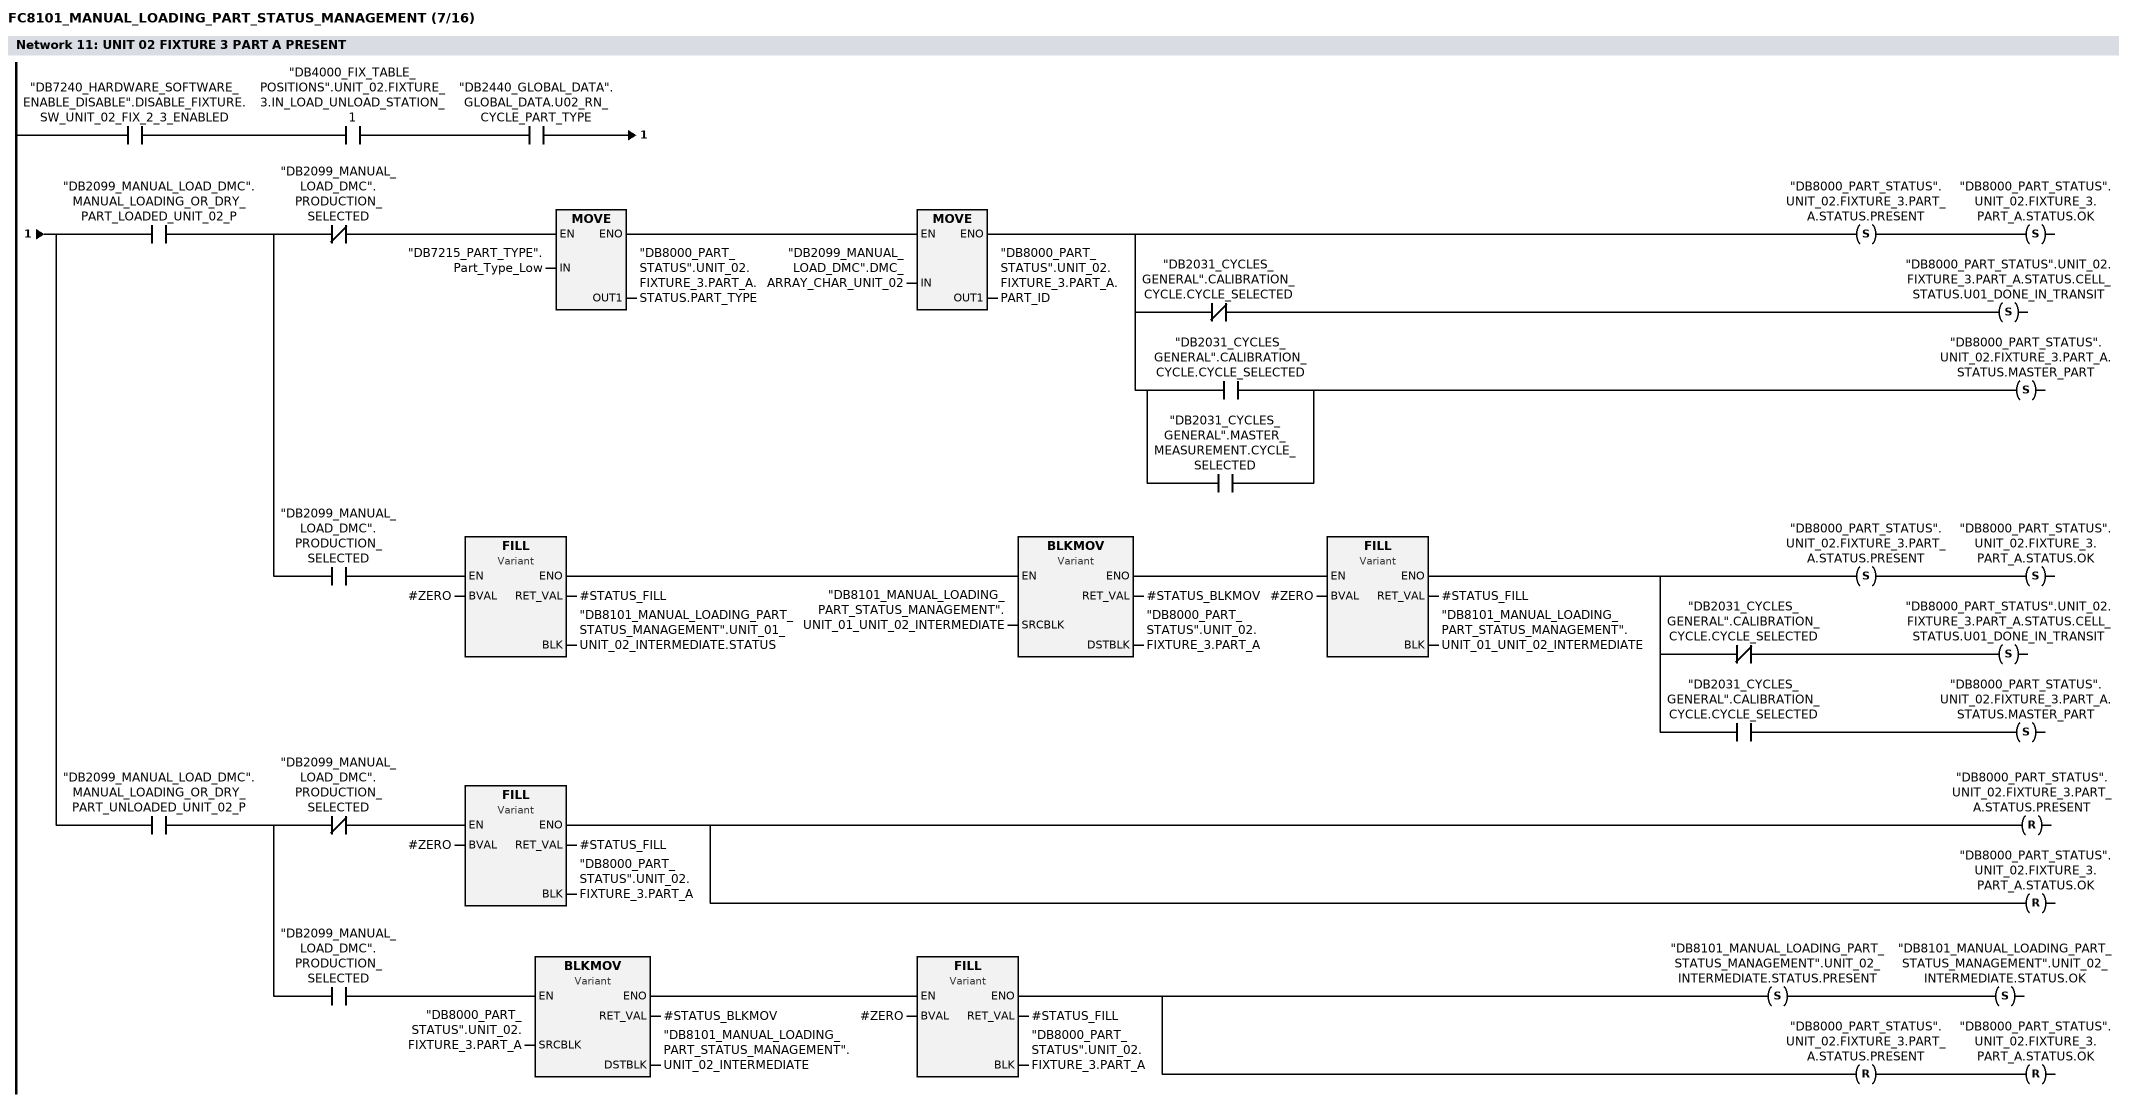
   RUNG wire#powerrail
      Contact( "DB7240_HARDWARE_SOFTWARE_ENABLE_DISABLE".DISABLE_FIXTURE.SW_UNIT_02_FIX_2_3_ENABLED )
      Contact( "DB4000_FIX_TABLE_POSITIONS".UNIT_02.FIXTURE_3.IN_LOAD_UNLOAD_STATION_1 )
      Contact( "DB2440_GLOBAL_DATA".GLOBAL_DATA.U02_RN_CYCLE_PART_TYPE )
      wire#w1
      Contact( "DB2099_MANUAL_LOAD_DMC".MANUAL_LOADING_OR_DRY_PART_LOADED_UNIT_02_P )
      wire#w2
      I_Contact( "DB2099_MANUAL_LOAD_DMC".PRODUCTION_SELECTED )
      { S7_GenerateENO := "TRUE" } Move(in := "DB7215_PART_TYPE".Part_Type_Low, out1 => "DB8000_PART_STATUS".UNIT_02.FIXTURE_3.PART_A.STATUS.PART_TYPE)
      Move(in := "DB2099_MANUAL_LOAD_DMC".DMC_ARRAY_CHAR_UNIT_02, out1 => "DB8000_PART_STATUS".UNIT_02.FIXTURE_3.PART_A.PART_ID)
      wire#w3
      S_Coil( "DB8000_PART_STATUS".UNIT_02.FIXTURE_3.PART_A.STATUS.PRESENT )
      S_Coil( "DB8000_PART_STATUS".UNIT_02.FIXTURE_3.PART_A.STATUS.OK )
   END_RUNG
   RUNG wire#w3
      I_Contact( "DB2031_CYCLES_GENERAL".CALIBRATION_CYCLE.CYCLE_SELECTED )
      S_Coil( "DB8000_PART_STATUS".UNIT_02.FIXTURE_3.PART_A.STATUS.CELL_STATUS.U01_DONE_IN_TRANSIT )
   END_RUNG
   RUNG wire#w3
      Contact( "DB2031_CYCLES_GENERAL".CALIBRATION_CYCLE.CYCLE_SELECTED )
      wire#w4
      S_Coil( "DB8000_PART_STATUS".UNIT_02.FIXTURE_3.PART_A.STATUS.MASTER_PART )
   END_RUNG
   RUNG wire#w3
      Contact( "DB2031_CYCLES_GENERAL".MASTER_MEASUREMENT.CYCLE_SELECTED )
   END_RUNG wire#w4
   RUNG wire#w2
      Contact( "DB2099_MANUAL_LOAD_DMC".PRODUCTION_SELECTED )
      { S7_Templates := "ptr_type := Variant" } FILL(BVAL := #ZERO, RET_VAL => #STATUS_FILL, BLK => "DB8101_MANUAL_LOADING_PART_STATUS_MANAGEMENT".UNIT_01_UNIT_02_INTERMEDIATE.STATUS)
      { S7_Templates := "blk_type := Variant" } BLKMOV(SRCBLK := "DB8101_MANUAL_LOADING_PART_STATUS_MANAGEMENT".UNIT_01_UNIT_02_INTERMEDIATE, RET_VAL => #STATUS_BLKMOV, DSTBLK => "DB8000_PART_STATUS".UNIT_02.FIXTURE_3.PART_A)
      { S7_Templates := "ptr_type := Variant" } FILL(BVAL := #ZERO, RET_VAL => #STATUS_FILL, BLK => "DB8101_MANUAL_LOADING_PART_STATUS_MANAGEMENT".UNIT_01_UNIT_02_INTERMEDIATE)
      wire#w5
      S_Coil( "DB8000_PART_STATUS".UNIT_02.FIXTURE_3.PART_A.STATUS.PRESENT )
      S_Coil( "DB8000_PART_STATUS".UNIT_02.FIXTURE_3.PART_A.STATUS.OK )
   END_RUNG
   RUNG wire#w5
      I_Contact( "DB2031_CYCLES_GENERAL".CALIBRATION_CYCLE.CYCLE_SELECTED )
      S_Coil( "DB8000_PART_STATUS".UNIT_02.FIXTURE_3.PART_A.STATUS.CELL_STATUS.U01_DONE_IN_TRANSIT )
   END_RUNG
   RUNG wire#w5
      Contact( "DB2031_CYCLES_GENERAL".CALIBRATION_CYCLE.CYCLE_SELECTED )
      S_Coil( "DB8000_PART_STATUS".UNIT_02.FIXTURE_3.PART_A.STATUS.MASTER_PART )
   END_RUNG
   RUNG wire#w1
      Contact( "DB2099_MANUAL_LOAD_DMC".MANUAL_LOADING_OR_DRY_PART_UNLOADED_UNIT_02_P )
      wire#w6
      I_Contact( "DB2099_MANUAL_LOAD_DMC".PRODUCTION_SELECTED )
      { S7_Templates := "ptr_type := Variant" } FILL(BVAL := #ZERO, RET_VAL => #STATUS_FILL, BLK => "DB8000_PART_STATUS".UNIT_02.FIXTURE_3.PART_A)
      wire#w7
      R_Coil( "DB8000_PART_STATUS".UNIT_02.FIXTURE_3.PART_A.STATUS.PRESENT )
   END_RUNG
   RUNG wire#w7
      R_Coil( "DB8000_PART_STATUS".UNIT_02.FIXTURE_3.PART_A.STATUS.OK )
   END_RUNG
   RUNG wire#w6
      Contact( "DB2099_MANUAL_LOAD_DMC".PRODUCTION_SELECTED )
      { S7_Templates := "blk_type := Variant" } BLKMOV(SRCBLK := "DB8000_PART_STATUS".UNIT_02.FIXTURE_3.PART_A, RET_VAL => #STATUS_BLKMOV, DSTBLK => "DB8101_MANUAL_LOADING_PART_STATUS_MANAGEMENT".UNIT_02_INTERMEDIATE)
      { S7_Templates := "ptr_type := Variant" } FILL(BVAL := #ZERO, RET_VAL => #STATUS_FILL, BLK => "DB8000_PART_STATUS".UNIT_02.FIXTURE_3.PART_A)
      wire#w8
      S_Coil( "DB8101_MANUAL_LOADING_PART_STATUS_MANAGEMENT".UNIT_02_INTERMEDIATE.STATUS.PRESENT )
      S_Coil( "DB8101_MANUAL_LOADING_PART_STATUS_MANAGEMENT".UNIT_02_INTERMEDIATE.STATUS.OK )
   END_RUNG
   RUNG wire#w8
      R_Coil( "DB8000_PART_STATUS".UNIT_02.FIXTURE_3.PART_A.STATUS.PRESENT )
      R_Coil( "DB8000_PART_STATUS".UNIT_02.FIXTURE_3.PART_A.STATUS.OK )
   END_RUNG
   // the same network as SCL:
   // ENO of a box is taken as its EN; it also drops when the box reports an error
   #_w1 := "DB7240_HARDWARE_SOFTWARE_ENABLE_DISABLE".DISABLE_FIXTURE.SW_UNIT_02_FIX_2_3_ENABLED AND "DB4000_FIX_TABLE_POSITIONS".UNIT_02.FIXTURE_3.IN_LOAD_UNLOAD_STATION_1 AND "DB2440_GLOBAL_DATA".GLOBAL_DATA.U02_RN_CYCLE_PART_TYPE;
   #_w2 := #_w1 AND "DB2099_MANUAL_LOAD_DMC".MANUAL_LOADING_OR_DRY_PART_LOADED_UNIT_02_P;
   #_w3 := #_w2 AND NOT "DB2099_MANUAL_LOAD_DMC".PRODUCTION_SELECTED;
   IF #_w3 THEN
       "DB8000_PART_STATUS".UNIT_02.FIXTURE_3.PART_A.STATUS.PART_TYPE := "DB7215_PART_TYPE".Part_Type_Low;
       "DB8000_PART_STATUS".UNIT_02.FIXTURE_3.PART_A.PART_ID := "DB2099_MANUAL_LOAD_DMC".DMC_ARRAY_CHAR_UNIT_02;
       "DB8000_PART_STATUS".UNIT_02.FIXTURE_3.PART_A.STATUS.PRESENT := TRUE;
       "DB8000_PART_STATUS".UNIT_02.FIXTURE_3.PART_A.STATUS.OK := TRUE;
   END_IF;
   IF #_w3 AND NOT "DB2031_CYCLES_GENERAL".CALIBRATION_CYCLE.CYCLE_SELECTED THEN
       "DB8000_PART_STATUS".UNIT_02.FIXTURE_3.PART_A.STATUS.CELL_STATUS.U01_DONE_IN_TRANSIT := TRUE;
   END_IF;
   IF #_w3 AND ("DB2031_CYCLES_GENERAL".CALIBRATION_CYCLE.CYCLE_SELECTED OR "DB2031_CYCLES_GENERAL".MASTER_MEASUREMENT.CYCLE_SELECTED) THEN
       "DB8000_PART_STATUS".UNIT_02.FIXTURE_3.PART_A.STATUS.MASTER_PART := TRUE;
   END_IF;
   #_w4 := #_w2 AND "DB2099_MANUAL_LOAD_DMC".PRODUCTION_SELECTED;
   #STATUS_FILL := FILL(EN := #_w4,
                        BVAL := #ZERO,
                        BLK => "DB8101_MANUAL_LOADING_PART_STATUS_MANAGEMENT".UNIT_01_UNIT_02_INTERMEDIATE.STATUS,
                        ENO => #_w5);
   #STATUS_BLKMOV := BLKMOV(EN := #_w5,
                           SRCBLK := "DB8101_MANUAL_LOADING_PART_STATUS_MANAGEMENT".UNIT_01_UNIT_02_INTERMEDIATE,
                           DSTBLK => "DB8000_PART_STATUS".UNIT_02.FIXTURE_3.PART_A,
                           ENO => #_w6);
   #STATUS_FILL := FILL(EN := #_w6,
                        BVAL := #ZERO,
                        BLK => "DB8101_MANUAL_LOADING_PART_STATUS_MANAGEMENT".UNIT_01_UNIT_02_INTERMEDIATE,
                        ENO => #_w7);
   IF #_w7 THEN
       "DB8000_PART_STATUS".UNIT_02.FIXTURE_3.PART_A.STATUS.PRESENT := TRUE;
       "DB8000_PART_STATUS".UNIT_02.FIXTURE_3.PART_A.STATUS.OK := TRUE;
   END_IF;
   IF #_w7 AND NOT "DB2031_CYCLES_GENERAL".CALIBRATION_CYCLE.CYCLE_SELECTED THEN
       "DB8000_PART_STATUS".UNIT_02.FIXTURE_3.PART_A.STATUS.CELL_STATUS.U01_DONE_IN_TRANSIT := TRUE;
   END_IF;
   IF #_w7 AND "DB2031_CYCLES_GENERAL".CALIBRATION_CYCLE.CYCLE_SELECTED THEN
       "DB8000_PART_STATUS".UNIT_02.FIXTURE_3.PART_A.STATUS.MASTER_PART := TRUE;
   END_IF;
   #_w8 := #_w1 AND "DB2099_MANUAL_LOAD_DMC".MANUAL_LOADING_OR_DRY_PART_UNLOADED_UNIT_02_P;
   #STATUS_FILL := FILL(EN := #_w8 AND NOT "DB2099_MANUAL_LOAD_DMC".PRODUCTION_SELECTED,
                        BVAL := #ZERO,
                        BLK => "DB8000_PART_STATUS".UNIT_02.FIXTURE_3.PART_A,
                        ENO => #_w9);
   IF #_w9 THEN
       "DB8000_PART_STATUS".UNIT_02.FIXTURE_3.PART_A.STATUS.PRESENT := FALSE;
       "DB8000_PART_STATUS".UNIT_02.FIXTURE_3.PART_A.STATUS.OK := FALSE;
   END_IF;
   #STATUS_BLKMOV := BLKMOV(EN := #_w8 AND "DB2099_MANUAL_LOAD_DMC".PRODUCTION_SELECTED,
                           SRCBLK := "DB8000_PART_STATUS".UNIT_02.FIXTURE_3.PART_A,
                           DSTBLK => "DB8101_MANUAL_LOADING_PART_STATUS_MANAGEMENT".UNIT_02_INTERMEDIATE,
                           ENO => #_w10);
   #STATUS_FILL := FILL(EN := #_w10,
                        BVAL := #ZERO,
                        BLK => "DB8000_PART_STATUS".UNIT_02.FIXTURE_3.PART_A,
                        ENO => #_w11);
   IF #_w11 THEN
       "DB8101_MANUAL_LOADING_PART_STATUS_MANAGEMENT".UNIT_02_INTERMEDIATE.STATUS.PRESENT := TRUE;
       "DB8101_MANUAL_LOADING_PART_STATUS_MANAGEMENT".UNIT_02_INTERMEDIATE.STATUS.OK := TRUE;
       "DB8000_PART_STATUS".UNIT_02.FIXTURE_3.PART_A.STATUS.PRESENT := FALSE;
       "DB8000_PART_STATUS".UNIT_02.FIXTURE_3.PART_A.STATUS.OK := FALSE;
   END_IF;
END_REGION

REGION Network 12: UNIT 02 FIXTURE 4 PART A PRESENT
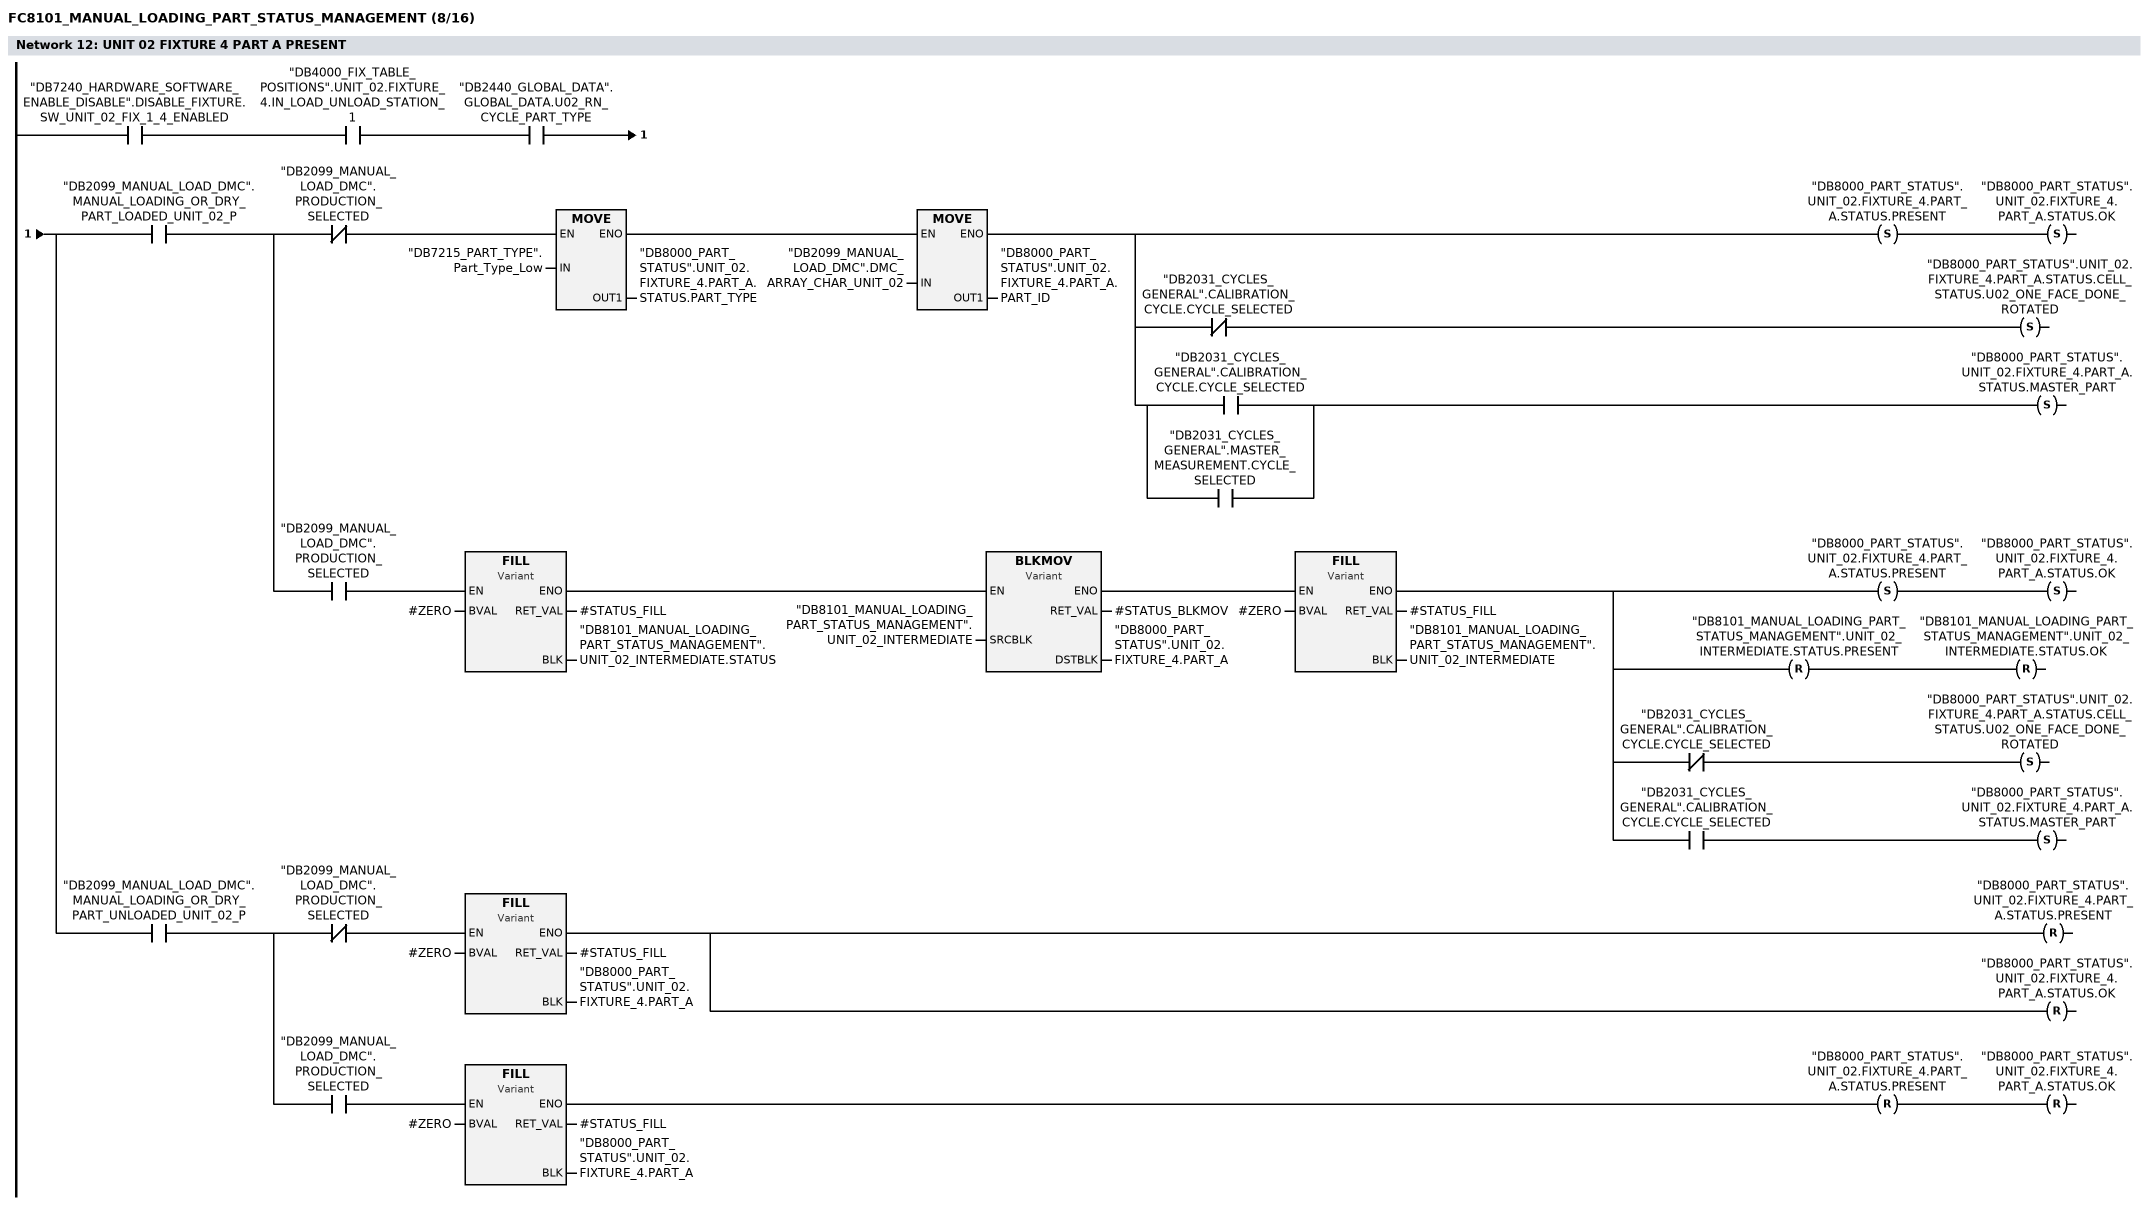
   RUNG wire#powerrail
      Contact( "DB7240_HARDWARE_SOFTWARE_ENABLE_DISABLE".DISABLE_FIXTURE.SW_UNIT_02_FIX_1_4_ENABLED )
      Contact( "DB4000_FIX_TABLE_POSITIONS".UNIT_02.FIXTURE_4.IN_LOAD_UNLOAD_STATION_1 )
      Contact( "DB2440_GLOBAL_DATA".GLOBAL_DATA.U02_RN_CYCLE_PART_TYPE )
      wire#w1
      Contact( "DB2099_MANUAL_LOAD_DMC".MANUAL_LOADING_OR_DRY_PART_LOADED_UNIT_02_P )
      wire#w2
      I_Contact( "DB2099_MANUAL_LOAD_DMC".PRODUCTION_SELECTED )
      { S7_GenerateENO := "TRUE" } Move(in := "DB7215_PART_TYPE".Part_Type_Low, out1 => "DB8000_PART_STATUS".UNIT_02.FIXTURE_4.PART_A.STATUS.PART_TYPE)
      Move(in := "DB2099_MANUAL_LOAD_DMC".DMC_ARRAY_CHAR_UNIT_02, out1 => "DB8000_PART_STATUS".UNIT_02.FIXTURE_4.PART_A.PART_ID)
      wire#w3
      S_Coil( "DB8000_PART_STATUS".UNIT_02.FIXTURE_4.PART_A.STATUS.PRESENT )
      S_Coil( "DB8000_PART_STATUS".UNIT_02.FIXTURE_4.PART_A.STATUS.OK )
   END_RUNG
   RUNG wire#w3
      I_Contact( "DB2031_CYCLES_GENERAL".CALIBRATION_CYCLE.CYCLE_SELECTED )
      S_Coil( "DB8000_PART_STATUS".UNIT_02.FIXTURE_4.PART_A.STATUS.CELL_STATUS.U02_ONE_FACE_DONE_ROTATED )
   END_RUNG
   RUNG wire#w3
      Contact( "DB2031_CYCLES_GENERAL".CALIBRATION_CYCLE.CYCLE_SELECTED )
      wire#w4
      S_Coil( "DB8000_PART_STATUS".UNIT_02.FIXTURE_4.PART_A.STATUS.MASTER_PART )
   END_RUNG
   RUNG wire#w3
      Contact( "DB2031_CYCLES_GENERAL".MASTER_MEASUREMENT.CYCLE_SELECTED )
   END_RUNG wire#w4
   RUNG wire#w2
      Contact( "DB2099_MANUAL_LOAD_DMC".PRODUCTION_SELECTED )
      { S7_Templates := "ptr_type := Variant" } FILL(BVAL := #ZERO, RET_VAL => #STATUS_FILL, BLK => "DB8101_MANUAL_LOADING_PART_STATUS_MANAGEMENT".UNIT_02_INTERMEDIATE.STATUS)
      { S7_Templates := "blk_type := Variant" } BLKMOV(SRCBLK := "DB8101_MANUAL_LOADING_PART_STATUS_MANAGEMENT".UNIT_02_INTERMEDIATE, RET_VAL => #STATUS_BLKMOV, DSTBLK => "DB8000_PART_STATUS".UNIT_02.FIXTURE_4.PART_A)
      { S7_Templates := "ptr_type := Variant" } FILL(BVAL := #ZERO, RET_VAL => #STATUS_FILL, BLK => "DB8101_MANUAL_LOADING_PART_STATUS_MANAGEMENT".UNIT_02_INTERMEDIATE)
      wire#w5
      S_Coil( "DB8000_PART_STATUS".UNIT_02.FIXTURE_4.PART_A.STATUS.PRESENT )
      S_Coil( "DB8000_PART_STATUS".UNIT_02.FIXTURE_4.PART_A.STATUS.OK )
   END_RUNG
   RUNG wire#w5
      R_Coil( "DB8101_MANUAL_LOADING_PART_STATUS_MANAGEMENT".UNIT_02_INTERMEDIATE.STATUS.PRESENT )
      R_Coil( "DB8101_MANUAL_LOADING_PART_STATUS_MANAGEMENT".UNIT_02_INTERMEDIATE.STATUS.OK )
   END_RUNG
   RUNG wire#w5
      I_Contact( "DB2031_CYCLES_GENERAL".CALIBRATION_CYCLE.CYCLE_SELECTED )
      S_Coil( "DB8000_PART_STATUS".UNIT_02.FIXTURE_4.PART_A.STATUS.CELL_STATUS.U02_ONE_FACE_DONE_ROTATED )
   END_RUNG
   RUNG wire#w5
      Contact( "DB2031_CYCLES_GENERAL".CALIBRATION_CYCLE.CYCLE_SELECTED )
      S_Coil( "DB8000_PART_STATUS".UNIT_02.FIXTURE_4.PART_A.STATUS.MASTER_PART )
   END_RUNG
   RUNG wire#w1
      Contact( "DB2099_MANUAL_LOAD_DMC".MANUAL_LOADING_OR_DRY_PART_UNLOADED_UNIT_02_P )
      wire#w6
      I_Contact( "DB2099_MANUAL_LOAD_DMC".PRODUCTION_SELECTED )
      { S7_Templates := "ptr_type := Variant" } FILL(BVAL := #ZERO, RET_VAL => #STATUS_FILL, BLK => "DB8000_PART_STATUS".UNIT_02.FIXTURE_4.PART_A)
      wire#w7
      R_Coil( "DB8000_PART_STATUS".UNIT_02.FIXTURE_4.PART_A.STATUS.PRESENT )
   END_RUNG
   RUNG wire#w7
      R_Coil( "DB8000_PART_STATUS".UNIT_02.FIXTURE_4.PART_A.STATUS.OK )
   END_RUNG
   RUNG wire#w6
      Contact( "DB2099_MANUAL_LOAD_DMC".PRODUCTION_SELECTED )
      { S7_Templates := "ptr_type := Variant" } FILL(BVAL := #ZERO, RET_VAL => #STATUS_FILL, BLK => "DB8000_PART_STATUS".UNIT_02.FIXTURE_4.PART_A)
      R_Coil( "DB8000_PART_STATUS".UNIT_02.FIXTURE_4.PART_A.STATUS.PRESENT )
      R_Coil( "DB8000_PART_STATUS".UNIT_02.FIXTURE_4.PART_A.STATUS.OK )
   END_RUNG
   // the same network as SCL:
   // ENO of a box is taken as its EN; it also drops when the box reports an error
   #_w1 := "DB7240_HARDWARE_SOFTWARE_ENABLE_DISABLE".DISABLE_FIXTURE.SW_UNIT_02_FIX_1_4_ENABLED AND "DB4000_FIX_TABLE_POSITIONS".UNIT_02.FIXTURE_4.IN_LOAD_UNLOAD_STATION_1 AND "DB2440_GLOBAL_DATA".GLOBAL_DATA.U02_RN_CYCLE_PART_TYPE;
   #_w2 := #_w1 AND "DB2099_MANUAL_LOAD_DMC".MANUAL_LOADING_OR_DRY_PART_LOADED_UNIT_02_P;
   #_w3 := #_w2 AND NOT "DB2099_MANUAL_LOAD_DMC".PRODUCTION_SELECTED;
   IF #_w3 THEN
       "DB8000_PART_STATUS".UNIT_02.FIXTURE_4.PART_A.STATUS.PART_TYPE := "DB7215_PART_TYPE".Part_Type_Low;
       "DB8000_PART_STATUS".UNIT_02.FIXTURE_4.PART_A.PART_ID := "DB2099_MANUAL_LOAD_DMC".DMC_ARRAY_CHAR_UNIT_02;
       "DB8000_PART_STATUS".UNIT_02.FIXTURE_4.PART_A.STATUS.PRESENT := TRUE;
       "DB8000_PART_STATUS".UNIT_02.FIXTURE_4.PART_A.STATUS.OK := TRUE;
   END_IF;
   IF #_w3 AND NOT "DB2031_CYCLES_GENERAL".CALIBRATION_CYCLE.CYCLE_SELECTED THEN
       "DB8000_PART_STATUS".UNIT_02.FIXTURE_4.PART_A.STATUS.CELL_STATUS.U02_ONE_FACE_DONE_ROTATED := TRUE;
   END_IF;
   IF #_w3 AND ("DB2031_CYCLES_GENERAL".CALIBRATION_CYCLE.CYCLE_SELECTED OR "DB2031_CYCLES_GENERAL".MASTER_MEASUREMENT.CYCLE_SELECTED) THEN
       "DB8000_PART_STATUS".UNIT_02.FIXTURE_4.PART_A.STATUS.MASTER_PART := TRUE;
   END_IF;
   #_w4 := #_w2 AND "DB2099_MANUAL_LOAD_DMC".PRODUCTION_SELECTED;
   #STATUS_FILL := FILL(EN := #_w4,
                        BVAL := #ZERO,
                        BLK => "DB8101_MANUAL_LOADING_PART_STATUS_MANAGEMENT".UNIT_02_INTERMEDIATE.STATUS,
                        ENO => #_w5);
   #STATUS_BLKMOV := BLKMOV(EN := #_w5,
                           SRCBLK := "DB8101_MANUAL_LOADING_PART_STATUS_MANAGEMENT".UNIT_02_INTERMEDIATE,
                           DSTBLK => "DB8000_PART_STATUS".UNIT_02.FIXTURE_4.PART_A,
                           ENO => #_w6);
   #STATUS_FILL := FILL(EN := #_w6,
                        BVAL := #ZERO,
                        BLK => "DB8101_MANUAL_LOADING_PART_STATUS_MANAGEMENT".UNIT_02_INTERMEDIATE,
                        ENO => #_w7);
   IF #_w7 THEN
       "DB8000_PART_STATUS".UNIT_02.FIXTURE_4.PART_A.STATUS.PRESENT := TRUE;
       "DB8000_PART_STATUS".UNIT_02.FIXTURE_4.PART_A.STATUS.OK := TRUE;
       "DB8101_MANUAL_LOADING_PART_STATUS_MANAGEMENT".UNIT_02_INTERMEDIATE.STATUS.PRESENT := FALSE;
       "DB8101_MANUAL_LOADING_PART_STATUS_MANAGEMENT".UNIT_02_INTERMEDIATE.STATUS.OK := FALSE;
   END_IF;
   IF #_w7 AND NOT "DB2031_CYCLES_GENERAL".CALIBRATION_CYCLE.CYCLE_SELECTED THEN
       "DB8000_PART_STATUS".UNIT_02.FIXTURE_4.PART_A.STATUS.CELL_STATUS.U02_ONE_FACE_DONE_ROTATED := TRUE;
   END_IF;
   IF #_w7 AND "DB2031_CYCLES_GENERAL".CALIBRATION_CYCLE.CYCLE_SELECTED THEN
       "DB8000_PART_STATUS".UNIT_02.FIXTURE_4.PART_A.STATUS.MASTER_PART := TRUE;
   END_IF;
   #_w8 := #_w1 AND "DB2099_MANUAL_LOAD_DMC".MANUAL_LOADING_OR_DRY_PART_UNLOADED_UNIT_02_P;
   #STATUS_FILL := FILL(EN := #_w8 AND NOT "DB2099_MANUAL_LOAD_DMC".PRODUCTION_SELECTED,
                        BVAL := #ZERO,
                        BLK => "DB8000_PART_STATUS".UNIT_02.FIXTURE_4.PART_A,
                        ENO => #_w9);
   IF #_w9 THEN
       "DB8000_PART_STATUS".UNIT_02.FIXTURE_4.PART_A.STATUS.PRESENT := FALSE;
       "DB8000_PART_STATUS".UNIT_02.FIXTURE_4.PART_A.STATUS.OK := FALSE;
   END_IF;
   #STATUS_FILL := FILL(EN := #_w8 AND "DB2099_MANUAL_LOAD_DMC".PRODUCTION_SELECTED,
                        BVAL := #ZERO,
                        BLK => "DB8000_PART_STATUS".UNIT_02.FIXTURE_4.PART_A,
                        ENO => #_w10);
   IF #_w10 THEN
       "DB8000_PART_STATUS".UNIT_02.FIXTURE_4.PART_A.STATUS.PRESENT := FALSE;
       "DB8000_PART_STATUS".UNIT_02.FIXTURE_4.PART_A.STATUS.OK := FALSE;
   END_IF;
END_REGION

REGION Network 13: <<<<<<<<<<<<<<<<<<<< NR CYCLE >>>>>>>>>>>>>>>>>>>>
END_REGION

REGION Network 14: <<<<<<<<<<<<<<<<<<<< UNIT 01 >>>>>>>>>>>>>>>>>>>>
END_REGION

REGION Network 15: UNIT 01 FIXTURE 1 PART A PRESENT
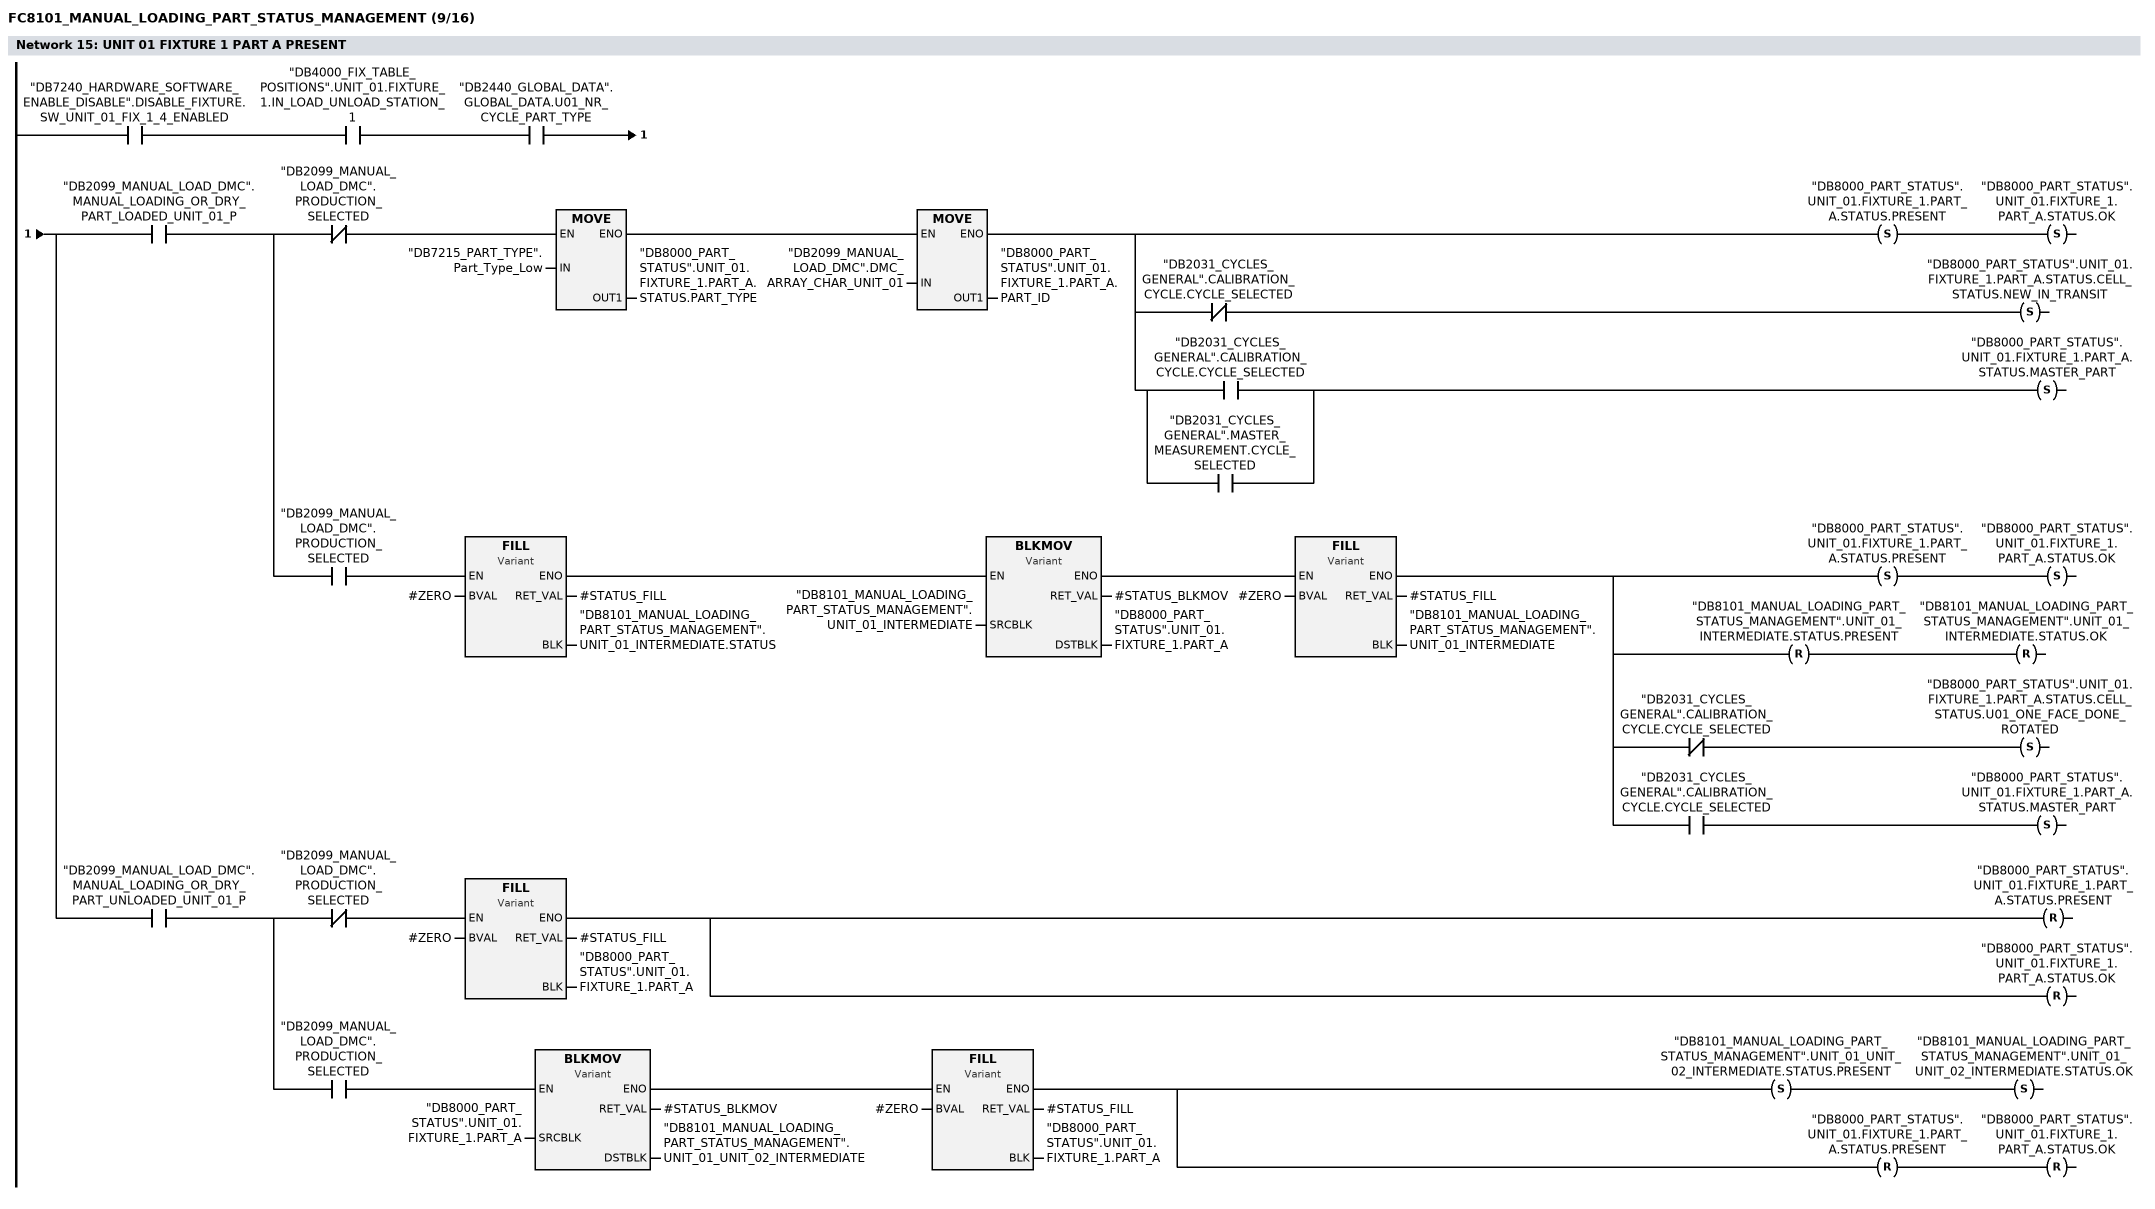
   RUNG wire#powerrail
      Contact( "DB7240_HARDWARE_SOFTWARE_ENABLE_DISABLE".DISABLE_FIXTURE.SW_UNIT_01_FIX_1_4_ENABLED )
      Contact( "DB4000_FIX_TABLE_POSITIONS".UNIT_01.FIXTURE_1.IN_LOAD_UNLOAD_STATION_1 )
      Contact( "DB2440_GLOBAL_DATA".GLOBAL_DATA.U01_NR_CYCLE_PART_TYPE )
      wire#w1
      Contact( "DB2099_MANUAL_LOAD_DMC".MANUAL_LOADING_OR_DRY_PART_LOADED_UNIT_01_P )
      wire#w2
      I_Contact( "DB2099_MANUAL_LOAD_DMC".PRODUCTION_SELECTED )
      { S7_GenerateENO := "TRUE" } Move(in := "DB7215_PART_TYPE".Part_Type_Low, out1 => "DB8000_PART_STATUS".UNIT_01.FIXTURE_1.PART_A.STATUS.PART_TYPE)
      Move(in := "DB2099_MANUAL_LOAD_DMC".DMC_ARRAY_CHAR_UNIT_01, out1 => "DB8000_PART_STATUS".UNIT_01.FIXTURE_1.PART_A.PART_ID)
      wire#w3
      S_Coil( "DB8000_PART_STATUS".UNIT_01.FIXTURE_1.PART_A.STATUS.PRESENT )
      S_Coil( "DB8000_PART_STATUS".UNIT_01.FIXTURE_1.PART_A.STATUS.OK )
   END_RUNG
   RUNG wire#w3
      I_Contact( "DB2031_CYCLES_GENERAL".CALIBRATION_CYCLE.CYCLE_SELECTED )
      S_Coil( "DB8000_PART_STATUS".UNIT_01.FIXTURE_1.PART_A.STATUS.CELL_STATUS.NEW_IN_TRANSIT )
   END_RUNG
   RUNG wire#w3
      Contact( "DB2031_CYCLES_GENERAL".CALIBRATION_CYCLE.CYCLE_SELECTED )
      wire#w4
      S_Coil( "DB8000_PART_STATUS".UNIT_01.FIXTURE_1.PART_A.STATUS.MASTER_PART )
   END_RUNG
   RUNG wire#w3
      Contact( "DB2031_CYCLES_GENERAL".MASTER_MEASUREMENT.CYCLE_SELECTED )
   END_RUNG wire#w4
   RUNG wire#w2
      Contact( "DB2099_MANUAL_LOAD_DMC".PRODUCTION_SELECTED )
      { S7_Templates := "ptr_type := Variant" } FILL(BVAL := #ZERO, RET_VAL => #STATUS_FILL, BLK => "DB8101_MANUAL_LOADING_PART_STATUS_MANAGEMENT".UNIT_01_INTERMEDIATE.STATUS)
      { S7_Templates := "blk_type := Variant" } BLKMOV(SRCBLK := "DB8101_MANUAL_LOADING_PART_STATUS_MANAGEMENT".UNIT_01_INTERMEDIATE, RET_VAL => #STATUS_BLKMOV, DSTBLK => "DB8000_PART_STATUS".UNIT_01.FIXTURE_1.PART_A)
      { S7_Templates := "ptr_type := Variant" } FILL(BVAL := #ZERO, RET_VAL => #STATUS_FILL, BLK => "DB8101_MANUAL_LOADING_PART_STATUS_MANAGEMENT".UNIT_01_INTERMEDIATE)
      wire#w5
      S_Coil( "DB8000_PART_STATUS".UNIT_01.FIXTURE_1.PART_A.STATUS.PRESENT )
      S_Coil( "DB8000_PART_STATUS".UNIT_01.FIXTURE_1.PART_A.STATUS.OK )
   END_RUNG
   RUNG wire#w5
      R_Coil( "DB8101_MANUAL_LOADING_PART_STATUS_MANAGEMENT".UNIT_01_INTERMEDIATE.STATUS.PRESENT )
      R_Coil( "DB8101_MANUAL_LOADING_PART_STATUS_MANAGEMENT".UNIT_01_INTERMEDIATE.STATUS.OK )
   END_RUNG
   RUNG wire#w5
      I_Contact( "DB2031_CYCLES_GENERAL".CALIBRATION_CYCLE.CYCLE_SELECTED )
      S_Coil( "DB8000_PART_STATUS".UNIT_01.FIXTURE_1.PART_A.STATUS.CELL_STATUS.U01_ONE_FACE_DONE_ROTATED )
   END_RUNG
   RUNG wire#w5
      Contact( "DB2031_CYCLES_GENERAL".CALIBRATION_CYCLE.CYCLE_SELECTED )
      S_Coil( "DB8000_PART_STATUS".UNIT_01.FIXTURE_1.PART_A.STATUS.MASTER_PART )
   END_RUNG
   RUNG wire#w1
      Contact( "DB2099_MANUAL_LOAD_DMC".MANUAL_LOADING_OR_DRY_PART_UNLOADED_UNIT_01_P )
      wire#w6
      I_Contact( "DB2099_MANUAL_LOAD_DMC".PRODUCTION_SELECTED )
      { S7_Templates := "ptr_type := Variant" } FILL(BVAL := #ZERO, RET_VAL => #STATUS_FILL, BLK => "DB8000_PART_STATUS".UNIT_01.FIXTURE_1.PART_A)
      wire#w7
      R_Coil( "DB8000_PART_STATUS".UNIT_01.FIXTURE_1.PART_A.STATUS.PRESENT )
   END_RUNG
   RUNG wire#w7
      R_Coil( "DB8000_PART_STATUS".UNIT_01.FIXTURE_1.PART_A.STATUS.OK )
   END_RUNG
   RUNG wire#w6
      Contact( "DB2099_MANUAL_LOAD_DMC".PRODUCTION_SELECTED )
      { S7_Templates := "blk_type := Variant" } BLKMOV(SRCBLK := "DB8000_PART_STATUS".UNIT_01.FIXTURE_1.PART_A, RET_VAL => #STATUS_BLKMOV, DSTBLK => "DB8101_MANUAL_LOADING_PART_STATUS_MANAGEMENT".UNIT_01_UNIT_02_INTERMEDIATE)
      { S7_Templates := "ptr_type := Variant" } FILL(BVAL := #ZERO, RET_VAL => #STATUS_FILL, BLK => "DB8000_PART_STATUS".UNIT_01.FIXTURE_1.PART_A)
      wire#w8
      S_Coil( "DB8101_MANUAL_LOADING_PART_STATUS_MANAGEMENT".UNIT_01_UNIT_02_INTERMEDIATE.STATUS.PRESENT )
      S_Coil( "DB8101_MANUAL_LOADING_PART_STATUS_MANAGEMENT".UNIT_01_UNIT_02_INTERMEDIATE.STATUS.OK )
   END_RUNG
   RUNG wire#w8
      R_Coil( "DB8000_PART_STATUS".UNIT_01.FIXTURE_1.PART_A.STATUS.PRESENT )
      R_Coil( "DB8000_PART_STATUS".UNIT_01.FIXTURE_1.PART_A.STATUS.OK )
   END_RUNG
   // the same network as SCL:
   // ENO of a box is taken as its EN; it also drops when the box reports an error
   #_w1 := "DB7240_HARDWARE_SOFTWARE_ENABLE_DISABLE".DISABLE_FIXTURE.SW_UNIT_01_FIX_1_4_ENABLED AND "DB4000_FIX_TABLE_POSITIONS".UNIT_01.FIXTURE_1.IN_LOAD_UNLOAD_STATION_1 AND "DB2440_GLOBAL_DATA".GLOBAL_DATA.U01_NR_CYCLE_PART_TYPE;
   #_w2 := #_w1 AND "DB2099_MANUAL_LOAD_DMC".MANUAL_LOADING_OR_DRY_PART_LOADED_UNIT_01_P;
   #_w3 := #_w2 AND NOT "DB2099_MANUAL_LOAD_DMC".PRODUCTION_SELECTED;
   IF #_w3 THEN
       "DB8000_PART_STATUS".UNIT_01.FIXTURE_1.PART_A.STATUS.PART_TYPE := "DB7215_PART_TYPE".Part_Type_Low;
       "DB8000_PART_STATUS".UNIT_01.FIXTURE_1.PART_A.PART_ID := "DB2099_MANUAL_LOAD_DMC".DMC_ARRAY_CHAR_UNIT_01;
       "DB8000_PART_STATUS".UNIT_01.FIXTURE_1.PART_A.STATUS.PRESENT := TRUE;
       "DB8000_PART_STATUS".UNIT_01.FIXTURE_1.PART_A.STATUS.OK := TRUE;
   END_IF;
   IF #_w3 AND NOT "DB2031_CYCLES_GENERAL".CALIBRATION_CYCLE.CYCLE_SELECTED THEN
       "DB8000_PART_STATUS".UNIT_01.FIXTURE_1.PART_A.STATUS.CELL_STATUS.NEW_IN_TRANSIT := TRUE;
   END_IF;
   IF #_w3 AND ("DB2031_CYCLES_GENERAL".CALIBRATION_CYCLE.CYCLE_SELECTED OR "DB2031_CYCLES_GENERAL".MASTER_MEASUREMENT.CYCLE_SELECTED) THEN
       "DB8000_PART_STATUS".UNIT_01.FIXTURE_1.PART_A.STATUS.MASTER_PART := TRUE;
   END_IF;
   #_w4 := #_w2 AND "DB2099_MANUAL_LOAD_DMC".PRODUCTION_SELECTED;
   #STATUS_FILL := FILL(EN := #_w4,
                        BVAL := #ZERO,
                        BLK => "DB8101_MANUAL_LOADING_PART_STATUS_MANAGEMENT".UNIT_01_INTERMEDIATE.STATUS,
                        ENO => #_w5);
   #STATUS_BLKMOV := BLKMOV(EN := #_w5,
                           SRCBLK := "DB8101_MANUAL_LOADING_PART_STATUS_MANAGEMENT".UNIT_01_INTERMEDIATE,
                           DSTBLK => "DB8000_PART_STATUS".UNIT_01.FIXTURE_1.PART_A,
                           ENO => #_w6);
   #STATUS_FILL := FILL(EN := #_w6,
                        BVAL := #ZERO,
                        BLK => "DB8101_MANUAL_LOADING_PART_STATUS_MANAGEMENT".UNIT_01_INTERMEDIATE,
                        ENO => #_w7);
   IF #_w7 THEN
       "DB8000_PART_STATUS".UNIT_01.FIXTURE_1.PART_A.STATUS.PRESENT := TRUE;
       "DB8000_PART_STATUS".UNIT_01.FIXTURE_1.PART_A.STATUS.OK := TRUE;
       "DB8101_MANUAL_LOADING_PART_STATUS_MANAGEMENT".UNIT_01_INTERMEDIATE.STATUS.PRESENT := FALSE;
       "DB8101_MANUAL_LOADING_PART_STATUS_MANAGEMENT".UNIT_01_INTERMEDIATE.STATUS.OK := FALSE;
   END_IF;
   IF #_w7 AND NOT "DB2031_CYCLES_GENERAL".CALIBRATION_CYCLE.CYCLE_SELECTED THEN
       "DB8000_PART_STATUS".UNIT_01.FIXTURE_1.PART_A.STATUS.CELL_STATUS.U01_ONE_FACE_DONE_ROTATED := TRUE;
   END_IF;
   IF #_w7 AND "DB2031_CYCLES_GENERAL".CALIBRATION_CYCLE.CYCLE_SELECTED THEN
       "DB8000_PART_STATUS".UNIT_01.FIXTURE_1.PART_A.STATUS.MASTER_PART := TRUE;
   END_IF;
   #_w8 := #_w1 AND "DB2099_MANUAL_LOAD_DMC".MANUAL_LOADING_OR_DRY_PART_UNLOADED_UNIT_01_P;
   #STATUS_FILL := FILL(EN := #_w8 AND NOT "DB2099_MANUAL_LOAD_DMC".PRODUCTION_SELECTED,
                        BVAL := #ZERO,
                        BLK => "DB8000_PART_STATUS".UNIT_01.FIXTURE_1.PART_A,
                        ENO => #_w9);
   IF #_w9 THEN
       "DB8000_PART_STATUS".UNIT_01.FIXTURE_1.PART_A.STATUS.PRESENT := FALSE;
       "DB8000_PART_STATUS".UNIT_01.FIXTURE_1.PART_A.STATUS.OK := FALSE;
   END_IF;
   #STATUS_BLKMOV := BLKMOV(EN := #_w8 AND "DB2099_MANUAL_LOAD_DMC".PRODUCTION_SELECTED,
                           SRCBLK := "DB8000_PART_STATUS".UNIT_01.FIXTURE_1.PART_A,
                           DSTBLK => "DB8101_MANUAL_LOADING_PART_STATUS_MANAGEMENT".UNIT_01_UNIT_02_INTERMEDIATE,
                           ENO => #_w10);
   #STATUS_FILL := FILL(EN := #_w10,
                        BVAL := #ZERO,
                        BLK => "DB8000_PART_STATUS".UNIT_01.FIXTURE_1.PART_A,
                        ENO => #_w11);
   IF #_w11 THEN
       "DB8101_MANUAL_LOADING_PART_STATUS_MANAGEMENT".UNIT_01_UNIT_02_INTERMEDIATE.STATUS.PRESENT := TRUE;
       "DB8101_MANUAL_LOADING_PART_STATUS_MANAGEMENT".UNIT_01_UNIT_02_INTERMEDIATE.STATUS.OK := TRUE;
       "DB8000_PART_STATUS".UNIT_01.FIXTURE_1.PART_A.STATUS.PRESENT := FALSE;
       "DB8000_PART_STATUS".UNIT_01.FIXTURE_1.PART_A.STATUS.OK := FALSE;
   END_IF;
END_REGION

REGION Network 16: UNIT 01 FIXTURE 2 PART A PRESENT
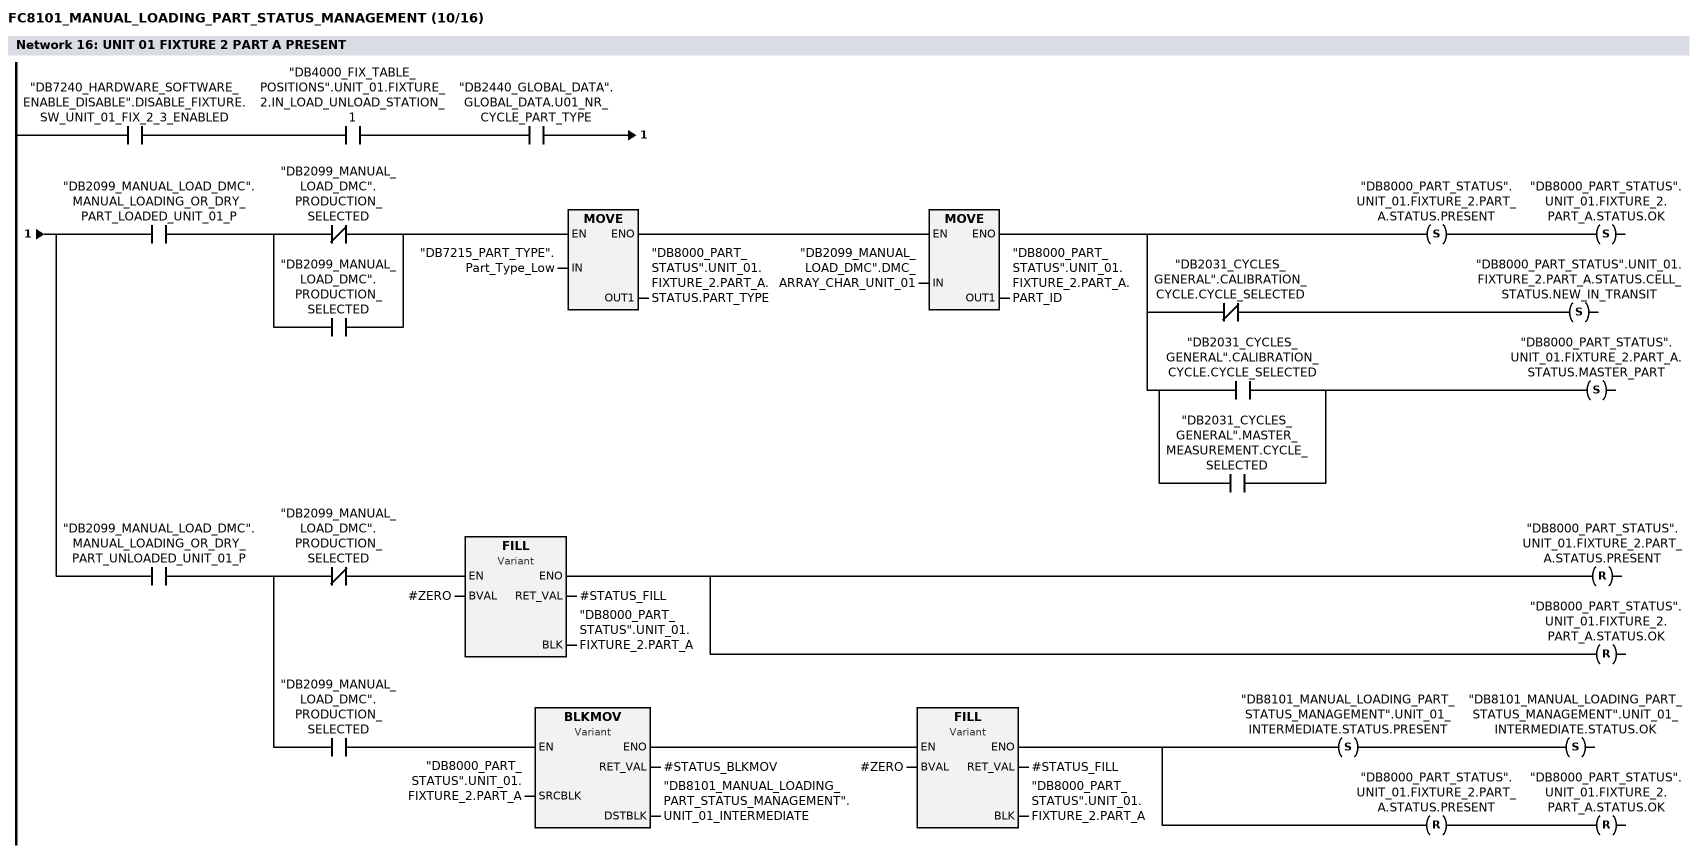
   RUNG wire#powerrail
      Contact( "DB7240_HARDWARE_SOFTWARE_ENABLE_DISABLE".DISABLE_FIXTURE.SW_UNIT_01_FIX_2_3_ENABLED )
      Contact( "DB4000_FIX_TABLE_POSITIONS".UNIT_01.FIXTURE_2.IN_LOAD_UNLOAD_STATION_1 )
      Contact( "DB2440_GLOBAL_DATA".GLOBAL_DATA.U01_NR_CYCLE_PART_TYPE )
      wire#w1
      Contact( "DB2099_MANUAL_LOAD_DMC".MANUAL_LOADING_OR_DRY_PART_LOADED_UNIT_01_P )
      wire#w2
      I_Contact( "DB2099_MANUAL_LOAD_DMC".PRODUCTION_SELECTED )
      wire#w3
      { S7_GenerateENO := "TRUE" } Move(in := "DB7215_PART_TYPE".Part_Type_Low, out1 => "DB8000_PART_STATUS".UNIT_01.FIXTURE_2.PART_A.STATUS.PART_TYPE)
      Move(in := "DB2099_MANUAL_LOAD_DMC".DMC_ARRAY_CHAR_UNIT_01, out1 => "DB8000_PART_STATUS".UNIT_01.FIXTURE_2.PART_A.PART_ID)
      wire#w4
      S_Coil( "DB8000_PART_STATUS".UNIT_01.FIXTURE_2.PART_A.STATUS.PRESENT )
      S_Coil( "DB8000_PART_STATUS".UNIT_01.FIXTURE_2.PART_A.STATUS.OK )
   END_RUNG
   RUNG wire#w2
      Contact( "DB2099_MANUAL_LOAD_DMC".PRODUCTION_SELECTED )
   END_RUNG wire#w3
   RUNG wire#w4
      I_Contact( "DB2031_CYCLES_GENERAL".CALIBRATION_CYCLE.CYCLE_SELECTED )
      S_Coil( "DB8000_PART_STATUS".UNIT_01.FIXTURE_2.PART_A.STATUS.CELL_STATUS.NEW_IN_TRANSIT )
   END_RUNG
   RUNG wire#w4
      Contact( "DB2031_CYCLES_GENERAL".CALIBRATION_CYCLE.CYCLE_SELECTED )
      wire#w5
      S_Coil( "DB8000_PART_STATUS".UNIT_01.FIXTURE_2.PART_A.STATUS.MASTER_PART )
   END_RUNG
   RUNG wire#w4
      Contact( "DB2031_CYCLES_GENERAL".MASTER_MEASUREMENT.CYCLE_SELECTED )
   END_RUNG wire#w5
   RUNG wire#w1
      Contact( "DB2099_MANUAL_LOAD_DMC".MANUAL_LOADING_OR_DRY_PART_UNLOADED_UNIT_01_P )
      wire#w6
      I_Contact( "DB2099_MANUAL_LOAD_DMC".PRODUCTION_SELECTED )
      { S7_Templates := "ptr_type := Variant" } FILL(BVAL := #ZERO, RET_VAL => #STATUS_FILL, BLK => "DB8000_PART_STATUS".UNIT_01.FIXTURE_2.PART_A)
      wire#w7
      R_Coil( "DB8000_PART_STATUS".UNIT_01.FIXTURE_2.PART_A.STATUS.PRESENT )
   END_RUNG
   RUNG wire#w7
      R_Coil( "DB8000_PART_STATUS".UNIT_01.FIXTURE_2.PART_A.STATUS.OK )
   END_RUNG
   RUNG wire#w6
      Contact( "DB2099_MANUAL_LOAD_DMC".PRODUCTION_SELECTED )
      { S7_Templates := "blk_type := Variant" } BLKMOV(SRCBLK := "DB8000_PART_STATUS".UNIT_01.FIXTURE_2.PART_A, RET_VAL => #STATUS_BLKMOV, DSTBLK => "DB8101_MANUAL_LOADING_PART_STATUS_MANAGEMENT".UNIT_01_INTERMEDIATE)
      { S7_Templates := "ptr_type := Variant" } FILL(BVAL := #ZERO, RET_VAL => #STATUS_FILL, BLK => "DB8000_PART_STATUS".UNIT_01.FIXTURE_2.PART_A)
      wire#w8
      S_Coil( "DB8101_MANUAL_LOADING_PART_STATUS_MANAGEMENT".UNIT_01_INTERMEDIATE.STATUS.PRESENT )
      S_Coil( "DB8101_MANUAL_LOADING_PART_STATUS_MANAGEMENT".UNIT_01_INTERMEDIATE.STATUS.OK )
   END_RUNG
   RUNG wire#w8
      R_Coil( "DB8000_PART_STATUS".UNIT_01.FIXTURE_2.PART_A.STATUS.PRESENT )
      R_Coil( "DB8000_PART_STATUS".UNIT_01.FIXTURE_2.PART_A.STATUS.OK )
   END_RUNG
   // the same network as SCL:
   // ENO of a box is taken as its EN; it also drops when the box reports an error
   #_w1 := "DB7240_HARDWARE_SOFTWARE_ENABLE_DISABLE".DISABLE_FIXTURE.SW_UNIT_01_FIX_2_3_ENABLED AND "DB4000_FIX_TABLE_POSITIONS".UNIT_01.FIXTURE_2.IN_LOAD_UNLOAD_STATION_1 AND "DB2440_GLOBAL_DATA".GLOBAL_DATA.U01_NR_CYCLE_PART_TYPE;
   #_w2 := #_w1 AND "DB2099_MANUAL_LOAD_DMC".MANUAL_LOADING_OR_DRY_PART_LOADED_UNIT_01_P AND (NOT "DB2099_MANUAL_LOAD_DMC".PRODUCTION_SELECTED OR "DB2099_MANUAL_LOAD_DMC".PRODUCTION_SELECTED);
   IF #_w2 THEN
       "DB8000_PART_STATUS".UNIT_01.FIXTURE_2.PART_A.STATUS.PART_TYPE := "DB7215_PART_TYPE".Part_Type_Low;
       "DB8000_PART_STATUS".UNIT_01.FIXTURE_2.PART_A.PART_ID := "DB2099_MANUAL_LOAD_DMC".DMC_ARRAY_CHAR_UNIT_01;
       "DB8000_PART_STATUS".UNIT_01.FIXTURE_2.PART_A.STATUS.PRESENT := TRUE;
       "DB8000_PART_STATUS".UNIT_01.FIXTURE_2.PART_A.STATUS.OK := TRUE;
   END_IF;
   IF #_w2 AND NOT "DB2031_CYCLES_GENERAL".CALIBRATION_CYCLE.CYCLE_SELECTED THEN
       "DB8000_PART_STATUS".UNIT_01.FIXTURE_2.PART_A.STATUS.CELL_STATUS.NEW_IN_TRANSIT := TRUE;
   END_IF;
   IF #_w2 AND ("DB2031_CYCLES_GENERAL".CALIBRATION_CYCLE.CYCLE_SELECTED OR "DB2031_CYCLES_GENERAL".MASTER_MEASUREMENT.CYCLE_SELECTED) THEN
       "DB8000_PART_STATUS".UNIT_01.FIXTURE_2.PART_A.STATUS.MASTER_PART := TRUE;
   END_IF;
   #_w3 := #_w1 AND "DB2099_MANUAL_LOAD_DMC".MANUAL_LOADING_OR_DRY_PART_UNLOADED_UNIT_01_P;
   #STATUS_FILL := FILL(EN := #_w3 AND NOT "DB2099_MANUAL_LOAD_DMC".PRODUCTION_SELECTED,
                        BVAL := #ZERO,
                        BLK => "DB8000_PART_STATUS".UNIT_01.FIXTURE_2.PART_A,
                        ENO => #_w4);
   IF #_w4 THEN
       "DB8000_PART_STATUS".UNIT_01.FIXTURE_2.PART_A.STATUS.PRESENT := FALSE;
       "DB8000_PART_STATUS".UNIT_01.FIXTURE_2.PART_A.STATUS.OK := FALSE;
   END_IF;
   #STATUS_BLKMOV := BLKMOV(EN := #_w3 AND "DB2099_MANUAL_LOAD_DMC".PRODUCTION_SELECTED,
                           SRCBLK := "DB8000_PART_STATUS".UNIT_01.FIXTURE_2.PART_A,
                           DSTBLK => "DB8101_MANUAL_LOADING_PART_STATUS_MANAGEMENT".UNIT_01_INTERMEDIATE,
                           ENO => #_w5);
   #STATUS_FILL := FILL(EN := #_w5,
                        BVAL := #ZERO,
                        BLK => "DB8000_PART_STATUS".UNIT_01.FIXTURE_2.PART_A,
                        ENO => #_w6);
   IF #_w6 THEN
       "DB8101_MANUAL_LOADING_PART_STATUS_MANAGEMENT".UNIT_01_INTERMEDIATE.STATUS.PRESENT := TRUE;
       "DB8101_MANUAL_LOADING_PART_STATUS_MANAGEMENT".UNIT_01_INTERMEDIATE.STATUS.OK := TRUE;
       "DB8000_PART_STATUS".UNIT_01.FIXTURE_2.PART_A.STATUS.PRESENT := FALSE;
       "DB8000_PART_STATUS".UNIT_01.FIXTURE_2.PART_A.STATUS.OK := FALSE;
   END_IF;
END_REGION

REGION Network 17: UNIT 01 FIXTURE 3 PART A PRESENT
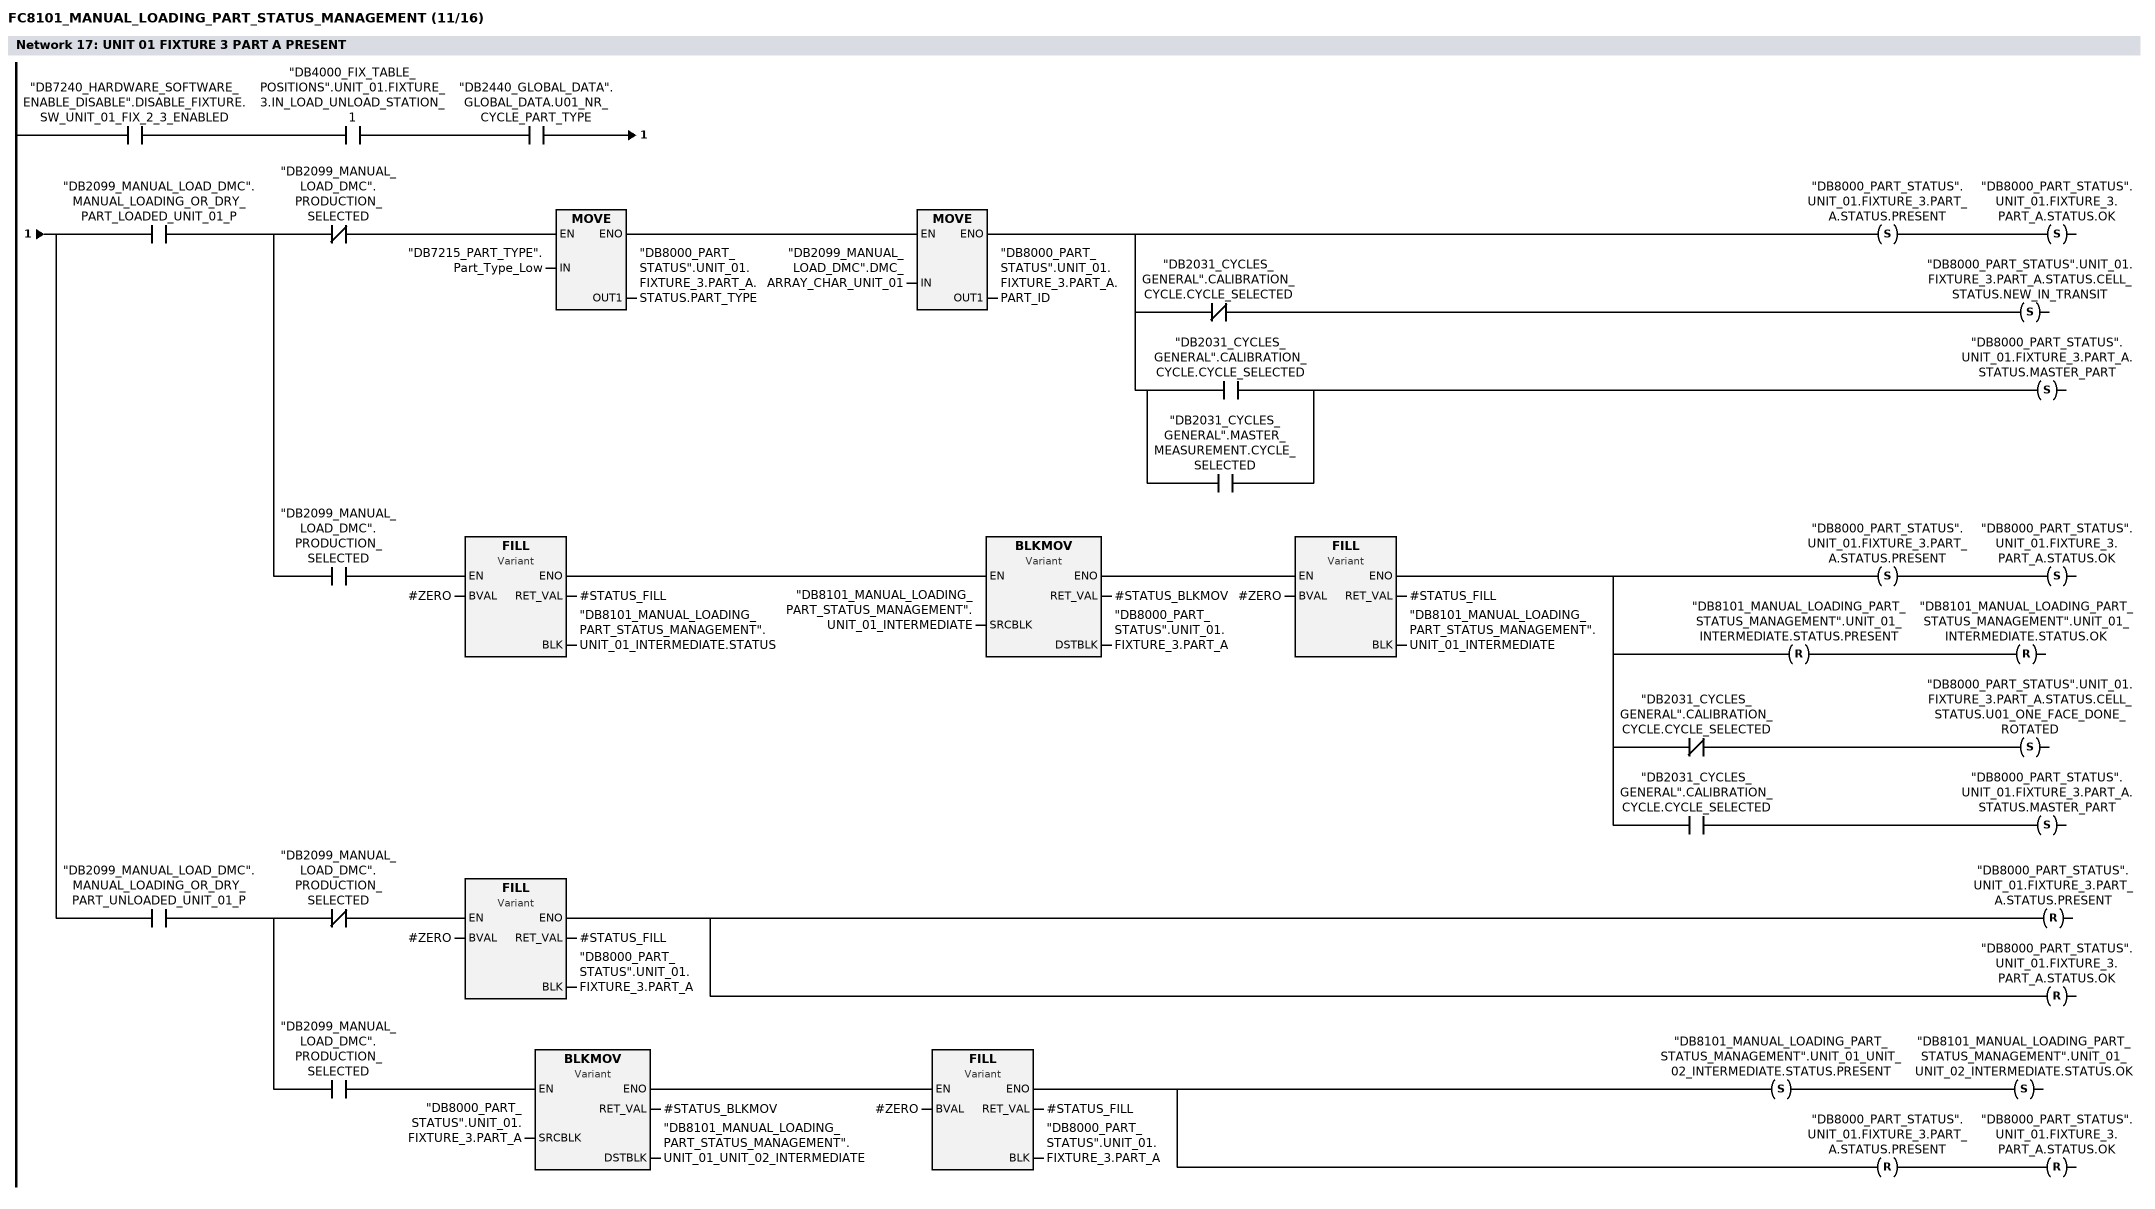
   RUNG wire#powerrail
      Contact( "DB7240_HARDWARE_SOFTWARE_ENABLE_DISABLE".DISABLE_FIXTURE.SW_UNIT_01_FIX_2_3_ENABLED )
      Contact( "DB4000_FIX_TABLE_POSITIONS".UNIT_01.FIXTURE_3.IN_LOAD_UNLOAD_STATION_1 )
      Contact( "DB2440_GLOBAL_DATA".GLOBAL_DATA.U01_NR_CYCLE_PART_TYPE )
      wire#w1
      Contact( "DB2099_MANUAL_LOAD_DMC".MANUAL_LOADING_OR_DRY_PART_LOADED_UNIT_01_P )
      wire#w2
      I_Contact( "DB2099_MANUAL_LOAD_DMC".PRODUCTION_SELECTED )
      { S7_GenerateENO := "TRUE" } Move(in := "DB7215_PART_TYPE".Part_Type_Low, out1 => "DB8000_PART_STATUS".UNIT_01.FIXTURE_3.PART_A.STATUS.PART_TYPE)
      Move(in := "DB2099_MANUAL_LOAD_DMC".DMC_ARRAY_CHAR_UNIT_01, out1 => "DB8000_PART_STATUS".UNIT_01.FIXTURE_3.PART_A.PART_ID)
      wire#w3
      S_Coil( "DB8000_PART_STATUS".UNIT_01.FIXTURE_3.PART_A.STATUS.PRESENT )
      S_Coil( "DB8000_PART_STATUS".UNIT_01.FIXTURE_3.PART_A.STATUS.OK )
   END_RUNG
   RUNG wire#w3
      I_Contact( "DB2031_CYCLES_GENERAL".CALIBRATION_CYCLE.CYCLE_SELECTED )
      S_Coil( "DB8000_PART_STATUS".UNIT_01.FIXTURE_3.PART_A.STATUS.CELL_STATUS.NEW_IN_TRANSIT )
   END_RUNG
   RUNG wire#w3
      Contact( "DB2031_CYCLES_GENERAL".CALIBRATION_CYCLE.CYCLE_SELECTED )
      wire#w4
      S_Coil( "DB8000_PART_STATUS".UNIT_01.FIXTURE_3.PART_A.STATUS.MASTER_PART )
   END_RUNG
   RUNG wire#w3
      Contact( "DB2031_CYCLES_GENERAL".MASTER_MEASUREMENT.CYCLE_SELECTED )
   END_RUNG wire#w4
   RUNG wire#w2
      Contact( "DB2099_MANUAL_LOAD_DMC".PRODUCTION_SELECTED )
      { S7_Templates := "ptr_type := Variant" } FILL(BVAL := #ZERO, RET_VAL => #STATUS_FILL, BLK => "DB8101_MANUAL_LOADING_PART_STATUS_MANAGEMENT".UNIT_01_INTERMEDIATE.STATUS)
      { S7_Templates := "blk_type := Variant" } BLKMOV(SRCBLK := "DB8101_MANUAL_LOADING_PART_STATUS_MANAGEMENT".UNIT_01_INTERMEDIATE, RET_VAL => #STATUS_BLKMOV, DSTBLK => "DB8000_PART_STATUS".UNIT_01.FIXTURE_3.PART_A)
      { S7_Templates := "ptr_type := Variant" } FILL(BVAL := #ZERO, RET_VAL => #STATUS_FILL, BLK => "DB8101_MANUAL_LOADING_PART_STATUS_MANAGEMENT".UNIT_01_INTERMEDIATE)
      wire#w5
      S_Coil( "DB8000_PART_STATUS".UNIT_01.FIXTURE_3.PART_A.STATUS.PRESENT )
      S_Coil( "DB8000_PART_STATUS".UNIT_01.FIXTURE_3.PART_A.STATUS.OK )
   END_RUNG
   RUNG wire#w5
      R_Coil( "DB8101_MANUAL_LOADING_PART_STATUS_MANAGEMENT".UNIT_01_INTERMEDIATE.STATUS.PRESENT )
      R_Coil( "DB8101_MANUAL_LOADING_PART_STATUS_MANAGEMENT".UNIT_01_INTERMEDIATE.STATUS.OK )
   END_RUNG
   RUNG wire#w5
      I_Contact( "DB2031_CYCLES_GENERAL".CALIBRATION_CYCLE.CYCLE_SELECTED )
      S_Coil( "DB8000_PART_STATUS".UNIT_01.FIXTURE_3.PART_A.STATUS.CELL_STATUS.U01_ONE_FACE_DONE_ROTATED )
   END_RUNG
   RUNG wire#w5
      Contact( "DB2031_CYCLES_GENERAL".CALIBRATION_CYCLE.CYCLE_SELECTED )
      S_Coil( "DB8000_PART_STATUS".UNIT_01.FIXTURE_3.PART_A.STATUS.MASTER_PART )
   END_RUNG
   RUNG wire#w1
      Contact( "DB2099_MANUAL_LOAD_DMC".MANUAL_LOADING_OR_DRY_PART_UNLOADED_UNIT_01_P )
      wire#w6
      I_Contact( "DB2099_MANUAL_LOAD_DMC".PRODUCTION_SELECTED )
      { S7_Templates := "ptr_type := Variant" } FILL(BVAL := #ZERO, RET_VAL => #STATUS_FILL, BLK => "DB8000_PART_STATUS".UNIT_01.FIXTURE_3.PART_A)
      wire#w7
      R_Coil( "DB8000_PART_STATUS".UNIT_01.FIXTURE_3.PART_A.STATUS.PRESENT )
   END_RUNG
   RUNG wire#w7
      R_Coil( "DB8000_PART_STATUS".UNIT_01.FIXTURE_3.PART_A.STATUS.OK )
   END_RUNG
   RUNG wire#w6
      Contact( "DB2099_MANUAL_LOAD_DMC".PRODUCTION_SELECTED )
      { S7_Templates := "blk_type := Variant" } BLKMOV(SRCBLK := "DB8000_PART_STATUS".UNIT_01.FIXTURE_3.PART_A, RET_VAL => #STATUS_BLKMOV, DSTBLK => "DB8101_MANUAL_LOADING_PART_STATUS_MANAGEMENT".UNIT_01_UNIT_02_INTERMEDIATE)
      { S7_Templates := "ptr_type := Variant" } FILL(BVAL := #ZERO, RET_VAL => #STATUS_FILL, BLK => "DB8000_PART_STATUS".UNIT_01.FIXTURE_3.PART_A)
      wire#w8
      S_Coil( "DB8101_MANUAL_LOADING_PART_STATUS_MANAGEMENT".UNIT_01_UNIT_02_INTERMEDIATE.STATUS.PRESENT )
      S_Coil( "DB8101_MANUAL_LOADING_PART_STATUS_MANAGEMENT".UNIT_01_UNIT_02_INTERMEDIATE.STATUS.OK )
   END_RUNG
   RUNG wire#w8
      R_Coil( "DB8000_PART_STATUS".UNIT_01.FIXTURE_3.PART_A.STATUS.PRESENT )
      R_Coil( "DB8000_PART_STATUS".UNIT_01.FIXTURE_3.PART_A.STATUS.OK )
   END_RUNG
   // the same network as SCL:
   // ENO of a box is taken as its EN; it also drops when the box reports an error
   #_w1 := "DB7240_HARDWARE_SOFTWARE_ENABLE_DISABLE".DISABLE_FIXTURE.SW_UNIT_01_FIX_2_3_ENABLED AND "DB4000_FIX_TABLE_POSITIONS".UNIT_01.FIXTURE_3.IN_LOAD_UNLOAD_STATION_1 AND "DB2440_GLOBAL_DATA".GLOBAL_DATA.U01_NR_CYCLE_PART_TYPE;
   #_w2 := #_w1 AND "DB2099_MANUAL_LOAD_DMC".MANUAL_LOADING_OR_DRY_PART_LOADED_UNIT_01_P;
   #_w3 := #_w2 AND NOT "DB2099_MANUAL_LOAD_DMC".PRODUCTION_SELECTED;
   IF #_w3 THEN
       "DB8000_PART_STATUS".UNIT_01.FIXTURE_3.PART_A.STATUS.PART_TYPE := "DB7215_PART_TYPE".Part_Type_Low;
       "DB8000_PART_STATUS".UNIT_01.FIXTURE_3.PART_A.PART_ID := "DB2099_MANUAL_LOAD_DMC".DMC_ARRAY_CHAR_UNIT_01;
       "DB8000_PART_STATUS".UNIT_01.FIXTURE_3.PART_A.STATUS.PRESENT := TRUE;
       "DB8000_PART_STATUS".UNIT_01.FIXTURE_3.PART_A.STATUS.OK := TRUE;
   END_IF;
   IF #_w3 AND NOT "DB2031_CYCLES_GENERAL".CALIBRATION_CYCLE.CYCLE_SELECTED THEN
       "DB8000_PART_STATUS".UNIT_01.FIXTURE_3.PART_A.STATUS.CELL_STATUS.NEW_IN_TRANSIT := TRUE;
   END_IF;
   IF #_w3 AND ("DB2031_CYCLES_GENERAL".CALIBRATION_CYCLE.CYCLE_SELECTED OR "DB2031_CYCLES_GENERAL".MASTER_MEASUREMENT.CYCLE_SELECTED) THEN
       "DB8000_PART_STATUS".UNIT_01.FIXTURE_3.PART_A.STATUS.MASTER_PART := TRUE;
   END_IF;
   #_w4 := #_w2 AND "DB2099_MANUAL_LOAD_DMC".PRODUCTION_SELECTED;
   #STATUS_FILL := FILL(EN := #_w4,
                        BVAL := #ZERO,
                        BLK => "DB8101_MANUAL_LOADING_PART_STATUS_MANAGEMENT".UNIT_01_INTERMEDIATE.STATUS,
                        ENO => #_w5);
   #STATUS_BLKMOV := BLKMOV(EN := #_w5,
                           SRCBLK := "DB8101_MANUAL_LOADING_PART_STATUS_MANAGEMENT".UNIT_01_INTERMEDIATE,
                           DSTBLK => "DB8000_PART_STATUS".UNIT_01.FIXTURE_3.PART_A,
                           ENO => #_w6);
   #STATUS_FILL := FILL(EN := #_w6,
                        BVAL := #ZERO,
                        BLK => "DB8101_MANUAL_LOADING_PART_STATUS_MANAGEMENT".UNIT_01_INTERMEDIATE,
                        ENO => #_w7);
   IF #_w7 THEN
       "DB8000_PART_STATUS".UNIT_01.FIXTURE_3.PART_A.STATUS.PRESENT := TRUE;
       "DB8000_PART_STATUS".UNIT_01.FIXTURE_3.PART_A.STATUS.OK := TRUE;
       "DB8101_MANUAL_LOADING_PART_STATUS_MANAGEMENT".UNIT_01_INTERMEDIATE.STATUS.PRESENT := FALSE;
       "DB8101_MANUAL_LOADING_PART_STATUS_MANAGEMENT".UNIT_01_INTERMEDIATE.STATUS.OK := FALSE;
   END_IF;
   IF #_w7 AND NOT "DB2031_CYCLES_GENERAL".CALIBRATION_CYCLE.CYCLE_SELECTED THEN
       "DB8000_PART_STATUS".UNIT_01.FIXTURE_3.PART_A.STATUS.CELL_STATUS.U01_ONE_FACE_DONE_ROTATED := TRUE;
   END_IF;
   IF #_w7 AND "DB2031_CYCLES_GENERAL".CALIBRATION_CYCLE.CYCLE_SELECTED THEN
       "DB8000_PART_STATUS".UNIT_01.FIXTURE_3.PART_A.STATUS.MASTER_PART := TRUE;
   END_IF;
   #_w8 := #_w1 AND "DB2099_MANUAL_LOAD_DMC".MANUAL_LOADING_OR_DRY_PART_UNLOADED_UNIT_01_P;
   #STATUS_FILL := FILL(EN := #_w8 AND NOT "DB2099_MANUAL_LOAD_DMC".PRODUCTION_SELECTED,
                        BVAL := #ZERO,
                        BLK => "DB8000_PART_STATUS".UNIT_01.FIXTURE_3.PART_A,
                        ENO => #_w9);
   IF #_w9 THEN
       "DB8000_PART_STATUS".UNIT_01.FIXTURE_3.PART_A.STATUS.PRESENT := FALSE;
       "DB8000_PART_STATUS".UNIT_01.FIXTURE_3.PART_A.STATUS.OK := FALSE;
   END_IF;
   #STATUS_BLKMOV := BLKMOV(EN := #_w8 AND "DB2099_MANUAL_LOAD_DMC".PRODUCTION_SELECTED,
                           SRCBLK := "DB8000_PART_STATUS".UNIT_01.FIXTURE_3.PART_A,
                           DSTBLK => "DB8101_MANUAL_LOADING_PART_STATUS_MANAGEMENT".UNIT_01_UNIT_02_INTERMEDIATE,
                           ENO => #_w10);
   #STATUS_FILL := FILL(EN := #_w10,
                        BVAL := #ZERO,
                        BLK => "DB8000_PART_STATUS".UNIT_01.FIXTURE_3.PART_A,
                        ENO => #_w11);
   IF #_w11 THEN
       "DB8101_MANUAL_LOADING_PART_STATUS_MANAGEMENT".UNIT_01_UNIT_02_INTERMEDIATE.STATUS.PRESENT := TRUE;
       "DB8101_MANUAL_LOADING_PART_STATUS_MANAGEMENT".UNIT_01_UNIT_02_INTERMEDIATE.STATUS.OK := TRUE;
       "DB8000_PART_STATUS".UNIT_01.FIXTURE_3.PART_A.STATUS.PRESENT := FALSE;
       "DB8000_PART_STATUS".UNIT_01.FIXTURE_3.PART_A.STATUS.OK := FALSE;
   END_IF;
END_REGION

REGION Network 18: UNIT 01 FIXTURE 4 PART A PRESENT
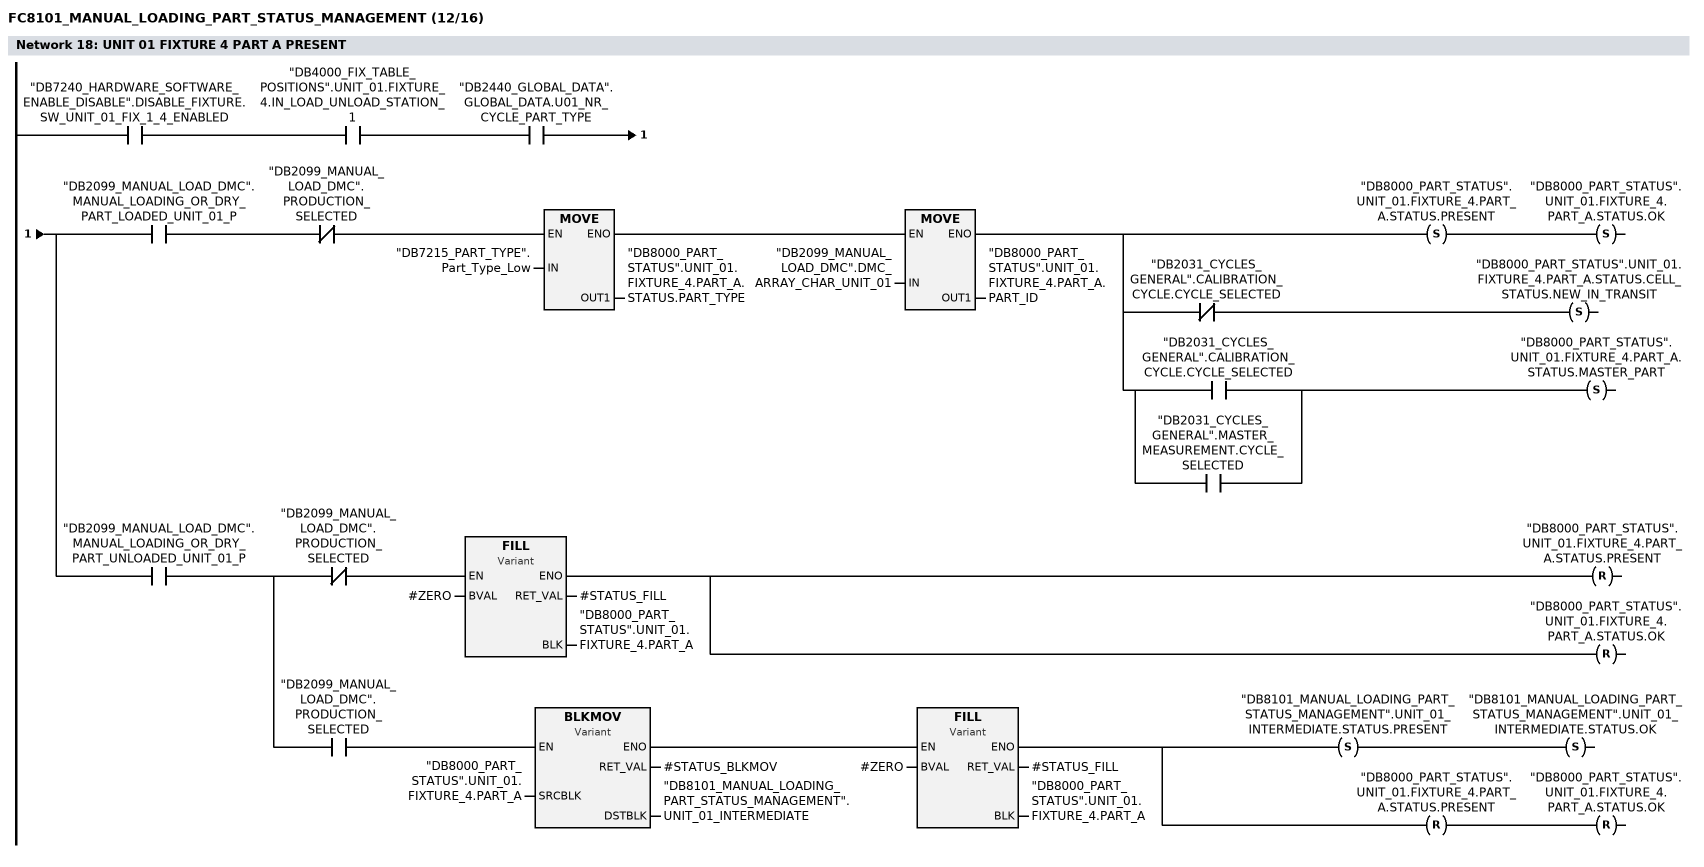
   RUNG wire#powerrail
      Contact( "DB7240_HARDWARE_SOFTWARE_ENABLE_DISABLE".DISABLE_FIXTURE.SW_UNIT_01_FIX_1_4_ENABLED )
      Contact( "DB4000_FIX_TABLE_POSITIONS".UNIT_01.FIXTURE_4.IN_LOAD_UNLOAD_STATION_1 )
      Contact( "DB2440_GLOBAL_DATA".GLOBAL_DATA.U01_NR_CYCLE_PART_TYPE )
      wire#w1
      Contact( "DB2099_MANUAL_LOAD_DMC".MANUAL_LOADING_OR_DRY_PART_LOADED_UNIT_01_P )
      I_Contact( "DB2099_MANUAL_LOAD_DMC".PRODUCTION_SELECTED )
      { S7_GenerateENO := "TRUE" } Move(in := "DB7215_PART_TYPE".Part_Type_Low, out1 => "DB8000_PART_STATUS".UNIT_01.FIXTURE_4.PART_A.STATUS.PART_TYPE)
      Move(in := "DB2099_MANUAL_LOAD_DMC".DMC_ARRAY_CHAR_UNIT_01, out1 => "DB8000_PART_STATUS".UNIT_01.FIXTURE_4.PART_A.PART_ID)
      wire#w2
      S_Coil( "DB8000_PART_STATUS".UNIT_01.FIXTURE_4.PART_A.STATUS.PRESENT )
      S_Coil( "DB8000_PART_STATUS".UNIT_01.FIXTURE_4.PART_A.STATUS.OK )
   END_RUNG
   RUNG wire#w2
      I_Contact( "DB2031_CYCLES_GENERAL".CALIBRATION_CYCLE.CYCLE_SELECTED )
      S_Coil( "DB8000_PART_STATUS".UNIT_01.FIXTURE_4.PART_A.STATUS.CELL_STATUS.NEW_IN_TRANSIT )
   END_RUNG
   RUNG wire#w2
      Contact( "DB2031_CYCLES_GENERAL".CALIBRATION_CYCLE.CYCLE_SELECTED )
      wire#w3
      S_Coil( "DB8000_PART_STATUS".UNIT_01.FIXTURE_4.PART_A.STATUS.MASTER_PART )
   END_RUNG
   RUNG wire#w2
      Contact( "DB2031_CYCLES_GENERAL".MASTER_MEASUREMENT.CYCLE_SELECTED )
   END_RUNG wire#w3
   RUNG wire#w1
      Contact( "DB2099_MANUAL_LOAD_DMC".MANUAL_LOADING_OR_DRY_PART_UNLOADED_UNIT_01_P )
      wire#w4
      I_Contact( "DB2099_MANUAL_LOAD_DMC".PRODUCTION_SELECTED )
      { S7_Templates := "ptr_type := Variant" } FILL(BVAL := #ZERO, RET_VAL => #STATUS_FILL, BLK => "DB8000_PART_STATUS".UNIT_01.FIXTURE_4.PART_A)
      wire#w5
      R_Coil( "DB8000_PART_STATUS".UNIT_01.FIXTURE_4.PART_A.STATUS.PRESENT )
   END_RUNG
   RUNG wire#w5
      R_Coil( "DB8000_PART_STATUS".UNIT_01.FIXTURE_4.PART_A.STATUS.OK )
   END_RUNG
   RUNG wire#w4
      Contact( "DB2099_MANUAL_LOAD_DMC".PRODUCTION_SELECTED )
      { S7_Templates := "blk_type := Variant" } BLKMOV(SRCBLK := "DB8000_PART_STATUS".UNIT_01.FIXTURE_4.PART_A, RET_VAL => #STATUS_BLKMOV, DSTBLK => "DB8101_MANUAL_LOADING_PART_STATUS_MANAGEMENT".UNIT_01_INTERMEDIATE)
      { S7_Templates := "ptr_type := Variant" } FILL(BVAL := #ZERO, RET_VAL => #STATUS_FILL, BLK => "DB8000_PART_STATUS".UNIT_01.FIXTURE_4.PART_A)
      wire#w6
      S_Coil( "DB8101_MANUAL_LOADING_PART_STATUS_MANAGEMENT".UNIT_01_INTERMEDIATE.STATUS.PRESENT )
      S_Coil( "DB8101_MANUAL_LOADING_PART_STATUS_MANAGEMENT".UNIT_01_INTERMEDIATE.STATUS.OK )
   END_RUNG
   RUNG wire#w6
      R_Coil( "DB8000_PART_STATUS".UNIT_01.FIXTURE_4.PART_A.STATUS.PRESENT )
      R_Coil( "DB8000_PART_STATUS".UNIT_01.FIXTURE_4.PART_A.STATUS.OK )
   END_RUNG
   // the same network as SCL:
   // ENO of a box is taken as its EN; it also drops when the box reports an error
   #_w1 := "DB7240_HARDWARE_SOFTWARE_ENABLE_DISABLE".DISABLE_FIXTURE.SW_UNIT_01_FIX_1_4_ENABLED AND "DB4000_FIX_TABLE_POSITIONS".UNIT_01.FIXTURE_4.IN_LOAD_UNLOAD_STATION_1 AND "DB2440_GLOBAL_DATA".GLOBAL_DATA.U01_NR_CYCLE_PART_TYPE;
   #_w2 := #_w1 AND "DB2099_MANUAL_LOAD_DMC".MANUAL_LOADING_OR_DRY_PART_LOADED_UNIT_01_P AND NOT "DB2099_MANUAL_LOAD_DMC".PRODUCTION_SELECTED;
   IF #_w2 THEN
       "DB8000_PART_STATUS".UNIT_01.FIXTURE_4.PART_A.STATUS.PART_TYPE := "DB7215_PART_TYPE".Part_Type_Low;
       "DB8000_PART_STATUS".UNIT_01.FIXTURE_4.PART_A.PART_ID := "DB2099_MANUAL_LOAD_DMC".DMC_ARRAY_CHAR_UNIT_01;
       "DB8000_PART_STATUS".UNIT_01.FIXTURE_4.PART_A.STATUS.PRESENT := TRUE;
       "DB8000_PART_STATUS".UNIT_01.FIXTURE_4.PART_A.STATUS.OK := TRUE;
   END_IF;
   IF #_w2 AND NOT "DB2031_CYCLES_GENERAL".CALIBRATION_CYCLE.CYCLE_SELECTED THEN
       "DB8000_PART_STATUS".UNIT_01.FIXTURE_4.PART_A.STATUS.CELL_STATUS.NEW_IN_TRANSIT := TRUE;
   END_IF;
   IF #_w2 AND ("DB2031_CYCLES_GENERAL".CALIBRATION_CYCLE.CYCLE_SELECTED OR "DB2031_CYCLES_GENERAL".MASTER_MEASUREMENT.CYCLE_SELECTED) THEN
       "DB8000_PART_STATUS".UNIT_01.FIXTURE_4.PART_A.STATUS.MASTER_PART := TRUE;
   END_IF;
   #_w3 := #_w1 AND "DB2099_MANUAL_LOAD_DMC".MANUAL_LOADING_OR_DRY_PART_UNLOADED_UNIT_01_P;
   #STATUS_FILL := FILL(EN := #_w3 AND NOT "DB2099_MANUAL_LOAD_DMC".PRODUCTION_SELECTED,
                        BVAL := #ZERO,
                        BLK => "DB8000_PART_STATUS".UNIT_01.FIXTURE_4.PART_A,
                        ENO => #_w4);
   IF #_w4 THEN
       "DB8000_PART_STATUS".UNIT_01.FIXTURE_4.PART_A.STATUS.PRESENT := FALSE;
       "DB8000_PART_STATUS".UNIT_01.FIXTURE_4.PART_A.STATUS.OK := FALSE;
   END_IF;
   #STATUS_BLKMOV := BLKMOV(EN := #_w3 AND "DB2099_MANUAL_LOAD_DMC".PRODUCTION_SELECTED,
                           SRCBLK := "DB8000_PART_STATUS".UNIT_01.FIXTURE_4.PART_A,
                           DSTBLK => "DB8101_MANUAL_LOADING_PART_STATUS_MANAGEMENT".UNIT_01_INTERMEDIATE,
                           ENO => #_w5);
   #STATUS_FILL := FILL(EN := #_w5,
                        BVAL := #ZERO,
                        BLK => "DB8000_PART_STATUS".UNIT_01.FIXTURE_4.PART_A,
                        ENO => #_w6);
   IF #_w6 THEN
       "DB8101_MANUAL_LOADING_PART_STATUS_MANAGEMENT".UNIT_01_INTERMEDIATE.STATUS.PRESENT := TRUE;
       "DB8101_MANUAL_LOADING_PART_STATUS_MANAGEMENT".UNIT_01_INTERMEDIATE.STATUS.OK := TRUE;
       "DB8000_PART_STATUS".UNIT_01.FIXTURE_4.PART_A.STATUS.PRESENT := FALSE;
       "DB8000_PART_STATUS".UNIT_01.FIXTURE_4.PART_A.STATUS.OK := FALSE;
   END_IF;
END_REGION

REGION Network 19: <<<<<<<<<<<<<<<<<<<< UNIT 02 >>>>>>>>>>>>>>>>>>>>
END_REGION

REGION Network 20: UNIT 02 FIXTURE 1 PART A PRESENT
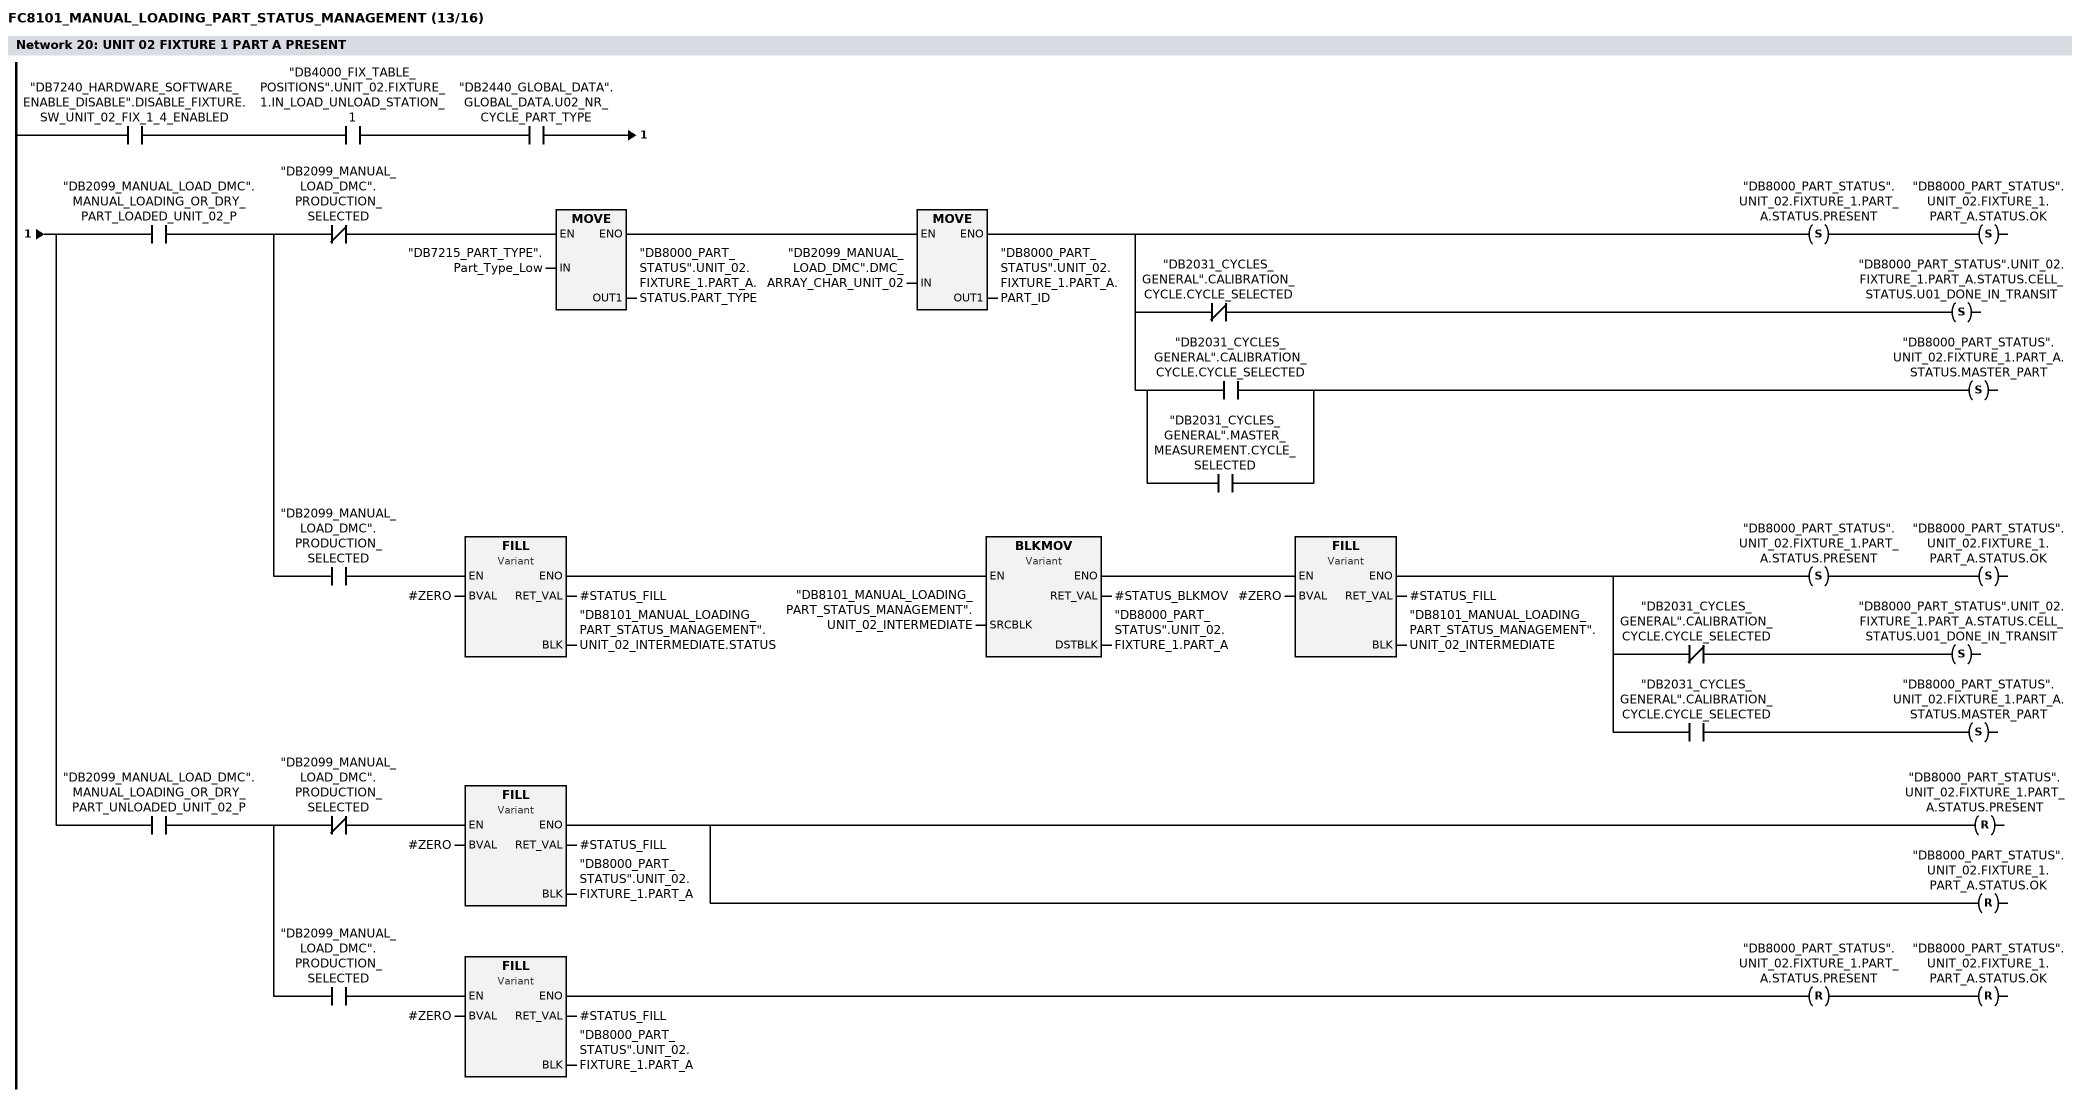
   RUNG wire#powerrail
      Contact( "DB7240_HARDWARE_SOFTWARE_ENABLE_DISABLE".DISABLE_FIXTURE.SW_UNIT_02_FIX_1_4_ENABLED )
      Contact( "DB4000_FIX_TABLE_POSITIONS".UNIT_02.FIXTURE_1.IN_LOAD_UNLOAD_STATION_1 )
      Contact( "DB2440_GLOBAL_DATA".GLOBAL_DATA.U02_NR_CYCLE_PART_TYPE )
      wire#w1
      Contact( "DB2099_MANUAL_LOAD_DMC".MANUAL_LOADING_OR_DRY_PART_LOADED_UNIT_02_P )
      wire#w2
      I_Contact( "DB2099_MANUAL_LOAD_DMC".PRODUCTION_SELECTED )
      { S7_GenerateENO := "TRUE" } Move(in := "DB7215_PART_TYPE".Part_Type_Low, out1 => "DB8000_PART_STATUS".UNIT_02.FIXTURE_1.PART_A.STATUS.PART_TYPE)
      Move(in := "DB2099_MANUAL_LOAD_DMC".DMC_ARRAY_CHAR_UNIT_02, out1 => "DB8000_PART_STATUS".UNIT_02.FIXTURE_1.PART_A.PART_ID)
      wire#w3
      S_Coil( "DB8000_PART_STATUS".UNIT_02.FIXTURE_1.PART_A.STATUS.PRESENT )
      S_Coil( "DB8000_PART_STATUS".UNIT_02.FIXTURE_1.PART_A.STATUS.OK )
   END_RUNG
   RUNG wire#w3
      I_Contact( "DB2031_CYCLES_GENERAL".CALIBRATION_CYCLE.CYCLE_SELECTED )
      S_Coil( "DB8000_PART_STATUS".UNIT_02.FIXTURE_1.PART_A.STATUS.CELL_STATUS.U01_DONE_IN_TRANSIT )
   END_RUNG
   RUNG wire#w3
      Contact( "DB2031_CYCLES_GENERAL".CALIBRATION_CYCLE.CYCLE_SELECTED )
      wire#w4
      S_Coil( "DB8000_PART_STATUS".UNIT_02.FIXTURE_1.PART_A.STATUS.MASTER_PART )
   END_RUNG
   RUNG wire#w3
      Contact( "DB2031_CYCLES_GENERAL".MASTER_MEASUREMENT.CYCLE_SELECTED )
   END_RUNG wire#w4
   RUNG wire#w2
      Contact( "DB2099_MANUAL_LOAD_DMC".PRODUCTION_SELECTED )
      { S7_Templates := "ptr_type := Variant" } FILL(BVAL := #ZERO, RET_VAL => #STATUS_FILL, BLK => "DB8101_MANUAL_LOADING_PART_STATUS_MANAGEMENT".UNIT_02_INTERMEDIATE.STATUS)
      { S7_Templates := "blk_type := Variant" } BLKMOV(SRCBLK := "DB8101_MANUAL_LOADING_PART_STATUS_MANAGEMENT".UNIT_02_INTERMEDIATE, RET_VAL => #STATUS_BLKMOV, DSTBLK => "DB8000_PART_STATUS".UNIT_02.FIXTURE_1.PART_A)
      { S7_Templates := "ptr_type := Variant" } FILL(BVAL := #ZERO, RET_VAL => #STATUS_FILL, BLK => "DB8101_MANUAL_LOADING_PART_STATUS_MANAGEMENT".UNIT_02_INTERMEDIATE)
      wire#w5
      S_Coil( "DB8000_PART_STATUS".UNIT_02.FIXTURE_1.PART_A.STATUS.PRESENT )
      S_Coil( "DB8000_PART_STATUS".UNIT_02.FIXTURE_1.PART_A.STATUS.OK )
   END_RUNG
   RUNG wire#w5
      I_Contact( "DB2031_CYCLES_GENERAL".CALIBRATION_CYCLE.CYCLE_SELECTED )
      S_Coil( "DB8000_PART_STATUS".UNIT_02.FIXTURE_1.PART_A.STATUS.CELL_STATUS.U01_DONE_IN_TRANSIT )
   END_RUNG
   RUNG wire#w5
      Contact( "DB2031_CYCLES_GENERAL".CALIBRATION_CYCLE.CYCLE_SELECTED )
      S_Coil( "DB8000_PART_STATUS".UNIT_02.FIXTURE_1.PART_A.STATUS.MASTER_PART )
   END_RUNG
   RUNG wire#w1
      Contact( "DB2099_MANUAL_LOAD_DMC".MANUAL_LOADING_OR_DRY_PART_UNLOADED_UNIT_02_P )
      wire#w6
      I_Contact( "DB2099_MANUAL_LOAD_DMC".PRODUCTION_SELECTED )
      { S7_Templates := "ptr_type := Variant" } FILL(BVAL := #ZERO, RET_VAL => #STATUS_FILL, BLK => "DB8000_PART_STATUS".UNIT_02.FIXTURE_1.PART_A)
      wire#w7
      R_Coil( "DB8000_PART_STATUS".UNIT_02.FIXTURE_1.PART_A.STATUS.PRESENT )
   END_RUNG
   RUNG wire#w7
      R_Coil( "DB8000_PART_STATUS".UNIT_02.FIXTURE_1.PART_A.STATUS.OK )
   END_RUNG
   RUNG wire#w6
      Contact( "DB2099_MANUAL_LOAD_DMC".PRODUCTION_SELECTED )
      { S7_Templates := "ptr_type := Variant" } FILL(BVAL := #ZERO, RET_VAL => #STATUS_FILL, BLK => "DB8000_PART_STATUS".UNIT_02.FIXTURE_1.PART_A)
      R_Coil( "DB8000_PART_STATUS".UNIT_02.FIXTURE_1.PART_A.STATUS.PRESENT )
      R_Coil( "DB8000_PART_STATUS".UNIT_02.FIXTURE_1.PART_A.STATUS.OK )
   END_RUNG
   // the same network as SCL:
   // ENO of a box is taken as its EN; it also drops when the box reports an error
   #_w1 := "DB7240_HARDWARE_SOFTWARE_ENABLE_DISABLE".DISABLE_FIXTURE.SW_UNIT_02_FIX_1_4_ENABLED AND "DB4000_FIX_TABLE_POSITIONS".UNIT_02.FIXTURE_1.IN_LOAD_UNLOAD_STATION_1 AND "DB2440_GLOBAL_DATA".GLOBAL_DATA.U02_NR_CYCLE_PART_TYPE;
   #_w2 := #_w1 AND "DB2099_MANUAL_LOAD_DMC".MANUAL_LOADING_OR_DRY_PART_LOADED_UNIT_02_P;
   #_w3 := #_w2 AND NOT "DB2099_MANUAL_LOAD_DMC".PRODUCTION_SELECTED;
   IF #_w3 THEN
       "DB8000_PART_STATUS".UNIT_02.FIXTURE_1.PART_A.STATUS.PART_TYPE := "DB7215_PART_TYPE".Part_Type_Low;
       "DB8000_PART_STATUS".UNIT_02.FIXTURE_1.PART_A.PART_ID := "DB2099_MANUAL_LOAD_DMC".DMC_ARRAY_CHAR_UNIT_02;
       "DB8000_PART_STATUS".UNIT_02.FIXTURE_1.PART_A.STATUS.PRESENT := TRUE;
       "DB8000_PART_STATUS".UNIT_02.FIXTURE_1.PART_A.STATUS.OK := TRUE;
   END_IF;
   IF #_w3 AND NOT "DB2031_CYCLES_GENERAL".CALIBRATION_CYCLE.CYCLE_SELECTED THEN
       "DB8000_PART_STATUS".UNIT_02.FIXTURE_1.PART_A.STATUS.CELL_STATUS.U01_DONE_IN_TRANSIT := TRUE;
   END_IF;
   IF #_w3 AND ("DB2031_CYCLES_GENERAL".CALIBRATION_CYCLE.CYCLE_SELECTED OR "DB2031_CYCLES_GENERAL".MASTER_MEASUREMENT.CYCLE_SELECTED) THEN
       "DB8000_PART_STATUS".UNIT_02.FIXTURE_1.PART_A.STATUS.MASTER_PART := TRUE;
   END_IF;
   #_w4 := #_w2 AND "DB2099_MANUAL_LOAD_DMC".PRODUCTION_SELECTED;
   #STATUS_FILL := FILL(EN := #_w4,
                        BVAL := #ZERO,
                        BLK => "DB8101_MANUAL_LOADING_PART_STATUS_MANAGEMENT".UNIT_02_INTERMEDIATE.STATUS,
                        ENO => #_w5);
   #STATUS_BLKMOV := BLKMOV(EN := #_w5,
                           SRCBLK := "DB8101_MANUAL_LOADING_PART_STATUS_MANAGEMENT".UNIT_02_INTERMEDIATE,
                           DSTBLK => "DB8000_PART_STATUS".UNIT_02.FIXTURE_1.PART_A,
                           ENO => #_w6);
   #STATUS_FILL := FILL(EN := #_w6,
                        BVAL := #ZERO,
                        BLK => "DB8101_MANUAL_LOADING_PART_STATUS_MANAGEMENT".UNIT_02_INTERMEDIATE,
                        ENO => #_w7);
   IF #_w7 THEN
       "DB8000_PART_STATUS".UNIT_02.FIXTURE_1.PART_A.STATUS.PRESENT := TRUE;
       "DB8000_PART_STATUS".UNIT_02.FIXTURE_1.PART_A.STATUS.OK := TRUE;
   END_IF;
   IF #_w7 AND NOT "DB2031_CYCLES_GENERAL".CALIBRATION_CYCLE.CYCLE_SELECTED THEN
       "DB8000_PART_STATUS".UNIT_02.FIXTURE_1.PART_A.STATUS.CELL_STATUS.U01_DONE_IN_TRANSIT := TRUE;
   END_IF;
   IF #_w7 AND "DB2031_CYCLES_GENERAL".CALIBRATION_CYCLE.CYCLE_SELECTED THEN
       "DB8000_PART_STATUS".UNIT_02.FIXTURE_1.PART_A.STATUS.MASTER_PART := TRUE;
   END_IF;
   #_w8 := #_w1 AND "DB2099_MANUAL_LOAD_DMC".MANUAL_LOADING_OR_DRY_PART_UNLOADED_UNIT_02_P;
   #STATUS_FILL := FILL(EN := #_w8 AND NOT "DB2099_MANUAL_LOAD_DMC".PRODUCTION_SELECTED,
                        BVAL := #ZERO,
                        BLK => "DB8000_PART_STATUS".UNIT_02.FIXTURE_1.PART_A,
                        ENO => #_w9);
   IF #_w9 THEN
       "DB8000_PART_STATUS".UNIT_02.FIXTURE_1.PART_A.STATUS.PRESENT := FALSE;
       "DB8000_PART_STATUS".UNIT_02.FIXTURE_1.PART_A.STATUS.OK := FALSE;
   END_IF;
   #STATUS_FILL := FILL(EN := #_w8 AND "DB2099_MANUAL_LOAD_DMC".PRODUCTION_SELECTED,
                        BVAL := #ZERO,
                        BLK => "DB8000_PART_STATUS".UNIT_02.FIXTURE_1.PART_A,
                        ENO => #_w10);
   IF #_w10 THEN
       "DB8000_PART_STATUS".UNIT_02.FIXTURE_1.PART_A.STATUS.PRESENT := FALSE;
       "DB8000_PART_STATUS".UNIT_02.FIXTURE_1.PART_A.STATUS.OK := FALSE;
   END_IF;
END_REGION

